REGION Network 1: Cân độc lập AGG5 Full
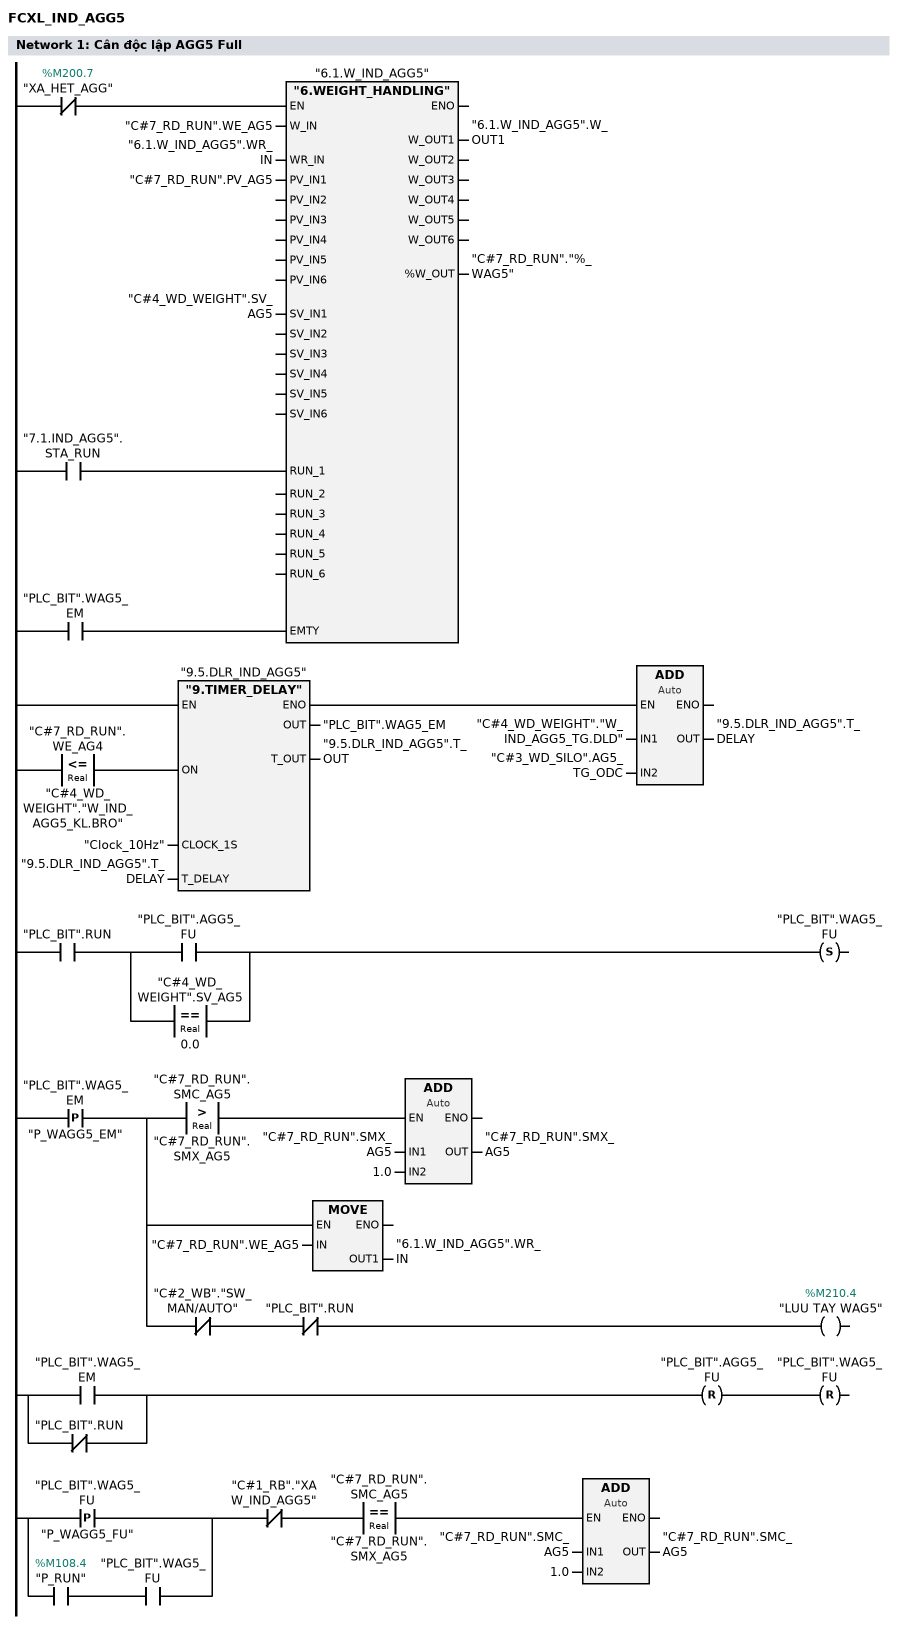
   RUNG wire#powerrail
      I_Contact( "XA_HET_AGG" )
      "6.1.W_IND_AGG5"(RUN_1 := wire#w1, EMTY := wire#w2, W_IN := "C#7_RD_RUN".WE_AG5, WR_IN := "6.1.W_IND_AGG5".WR_IN, PV_IN1 := "C#7_RD_RUN".PV_AG5, PV_IN2 :=, PV_IN3 :=, PV_IN4 :=, PV_IN5 :=, PV_IN6 :=, SV_IN1 := "C#4_WD_WEIGHT".SV_AG5, SV_IN2 :=, SV_IN3 :=, SV_IN4 :=, SV_IN5 :=, SV_IN6 :=, RUN_2 :=, RUN_3 :=, RUN_4 :=, RUN_5 :=, RUN_6 :=, W_OUT1 => "6.1.W_IND_AGG5".W_OUT1, W_OUT2 =>, W_OUT3 =>, W_OUT4 =>, W_OUT5 =>, W_OUT6 =>, "%W_OUT" => "C#7_RD_RUN"."%_WAG5")
   END_RUNG
   RUNG wire#powerrail
      Contact( "7.1.IND_AGG5".STA_RUN )
   END_RUNG wire#w1
   RUNG wire#powerrail
      Contact( "PLC_BIT".WAG5_EM )
   END_RUNG wire#w2
   RUNG wire#powerrail
      "9.5.DLR_IND_AGG5"(ON := wire#w3, CLOCK_1S := "Clock_10Hz", T_DELAY := "9.5.DLR_IND_AGG5".T_DELAY, OUT => "PLC_BIT".WAG5_EM, T_OUT => "9.5.DLR_IND_AGG5".T_OUT)
      Add(in1 := "C#4_WD_WEIGHT"."W_IND_AGG5_TG.DLD", in2 := "C#3_WD_SILO".AG5_TG_ODC, out => "9.5.DLR_IND_AGG5".T_DELAY)
   END_RUNG
   RUNG wire#powerrail
      { S7_Templates := "SrcType := Real" } LE_Contact(in1 := "C#7_RD_RUN".WE_AG4, in2 := "C#4_WD_WEIGHT"."W_IND_AGG5_KL.BRO")
   END_RUNG wire#w3
   RUNG wire#powerrail
      Contact( "PLC_BIT".RUN )
      wire#w4
      Contact( "PLC_BIT".AGG5_FU )
      wire#w5
      S_Coil( "PLC_BIT".WAG5_FU )
   END_RUNG
   RUNG wire#w4
      { S7_Templates := "SrcType := Real" } EQ_Contact(in1 := "C#4_WD_WEIGHT".SV_AG5, in2 := 0.0)
   END_RUNG wire#w5
   RUNG wire#powerrail
      P_Contact(operand := "PLC_BIT".WAG5_EM, bit := "P_WAGG5_EM")
      wire#w6
      { S7_Templates := "SrcType := Real" } GT_Contact(in1 := "C#7_RD_RUN".SMC_AG5, in2 := "C#7_RD_RUN".SMX_AG5)
      Add(in1 := "C#7_RD_RUN".SMX_AG5, in2 := 1.0, out => "C#7_RD_RUN".SMX_AG5)
   END_RUNG
   RUNG wire#w6
      Move(in := "C#7_RD_RUN".WE_AG5, out1 => "6.1.W_IND_AGG5".WR_IN)
   END_RUNG
   RUNG wire#w6
      I_Contact( "C#2_WB"."SW_MAN/AUTO" )
      I_Contact( "PLC_BIT".RUN )
      Coil( "LUU TAY WAG5" )
   END_RUNG
   RUNG wire#powerrail
      Contact( "PLC_BIT".WAG5_EM )
      wire#w7
      R_Coil( "PLC_BIT".AGG5_FU )
      R_Coil( "PLC_BIT".WAG5_FU )
   END_RUNG
   RUNG wire#powerrail
      I_Contact( "PLC_BIT".RUN )
   END_RUNG wire#w7
   RUNG wire#powerrail
      P_Contact(operand := "PLC_BIT".WAG5_FU, bit := "P_WAGG5_FU")
      wire#w8
      I_Contact( "C#1_RB"."XA W_IND_AGG5" )
      { S7_Templates := "SrcType := Real" } EQ_Contact(in1 := "C#7_RD_RUN".SMC_AG5, in2 := "C#7_RD_RUN".SMX_AG5)
      Add(in1 := "C#7_RD_RUN".SMC_AG5, in2 := 1.0, out => "C#7_RD_RUN".SMC_AG5)
   END_RUNG
   RUNG wire#powerrail
      Contact( "P_RUN" )
      Contact( "PLC_BIT".WAG5_FU )
   END_RUNG wire#w8
   // the same network as SCL:
   IF NOT "XA_HET_AGG" THEN
       "6.1.W_IND_AGG5"(W_IN := "C#7_RD_RUN".WE_AG5,   // "6.WEIGHT_HANDLING"
                        WR_IN := "6.1.W_IND_AGG5".WR_IN,
                        PV_IN1 := "C#7_RD_RUN".PV_AG5,
                        SV_IN1 := "C#4_WD_WEIGHT".SV_AG5,
                        RUN_1 := "7.1.IND_AGG5".STA_RUN,
                        EMTY := "PLC_BIT".WAG5_EM,
                        W_OUT1 => "6.1.W_IND_AGG5".W_OUT1,
                        "%W_OUT" => "C#7_RD_RUN"."%_WAG5");
   END_IF;
   "9.5.DLR_IND_AGG5"(ON := "C#7_RD_RUN".WE_AG4 <= "C#4_WD_WEIGHT"."W_IND_AGG5_KL.BRO",   // "9.TIMER_DELAY"
                      CLOCK_1S := "Clock_10Hz",
                      T_DELAY := "9.5.DLR_IND_AGG5".T_DELAY,
                      OUT => "PLC_BIT".WAG5_EM,
                      T_OUT => "9.5.DLR_IND_AGG5".T_OUT,
                      ENO => #_w1);
   IF #_w1 THEN
       "9.5.DLR_IND_AGG5".T_DELAY := "C#4_WD_WEIGHT"."W_IND_AGG5_TG.DLD" + "C#3_WD_SILO".AG5_TG_ODC;
   END_IF;
   IF "PLC_BIT".RUN AND ("PLC_BIT".AGG5_FU OR ("C#4_WD_WEIGHT".SV_AG5 = 0.0)) THEN
       "PLC_BIT".WAG5_FU := TRUE;
   END_IF;
   #_w2 := "PLC_BIT".WAG5_EM AND NOT "P_WAGG5_EM";   // rising edge of "PLC_BIT".WAG5_EM
   "P_WAGG5_EM" := "PLC_BIT".WAG5_EM;
   IF #_w2 AND ("C#7_RD_RUN".SMC_AG5 > "C#7_RD_RUN".SMX_AG5) THEN
       "C#7_RD_RUN".SMX_AG5 := "C#7_RD_RUN".SMX_AG5 + 1.0;
   END_IF;
   IF #_w2 THEN "6.1.W_IND_AGG5".WR_IN := "C#7_RD_RUN".WE_AG5; END_IF;
   "LUU TAY WAG5" := #_w2 AND NOT "C#2_WB"."SW_MAN/AUTO" AND NOT "PLC_BIT".RUN;
   IF "PLC_BIT".WAG5_EM OR NOT "PLC_BIT".RUN THEN
       "PLC_BIT".AGG5_FU := FALSE;
       "PLC_BIT".WAG5_FU := FALSE;
   END_IF;
   #_w3 := "PLC_BIT".WAG5_FU AND NOT "P_WAGG5_FU";   // rising edge of "PLC_BIT".WAG5_FU
   "P_WAGG5_FU" := "PLC_BIT".WAG5_FU;
   IF (#_w3 OR ("P_RUN" AND "PLC_BIT".WAG5_FU)) AND NOT "C#1_RB"."XA W_IND_AGG5" AND ("C#7_RD_RUN".SMC_AG5 = "C#7_RD_RUN".SMX_AG5) THEN
       "C#7_RD_RUN".SMC_AG5 := "C#7_RD_RUN".SMC_AG5 + 1.0;
   END_IF;
END_REGION
END_FUNCTION

FUNCTION "FCCA_IND_AGG5" : Void   // FC14, LAD
{ S7_Optimized_Access := 'TRUE' }
VERSION : 0.1
// stored: AutoNumber true, CodeModifiedDate 2026-01-15T16:25:54.5394757Z, CompileDate 2026-01-15T16:25:54.5786206Z, CreationDate 2026-01-15T16:24:02.4619467Z, HandleErrorsWithinBlock false, InterfaceModifiedDate 2026-01-11T04:47:10.3302964Z, IsConsistent true, IsIECCheckEnabled false, IsKnowHowProtected false, IsWriteProtected false, LibraryConformanceStatus Error: The block contains calls of single instances. Warning: The object contains access to global data blocks. Warning: The block contains direct access to inputs, outputs, bit memories, indirect access to the registry or indirect access to external memory areas that are unknown at the time of compilation., ModifiedDate 2026-01-15T16:25:54.5394757Z, ParameterModified 2026-01-11T04:47:10.3302964Z, PLCSimAdvancedSupport false, SetENOAutomatically False, StructureModified 2026-01-11T04:47:10.3302964Z, UDAEnableTagReadback false
BEGIN

REGION Network 1: Trạng thái cân AGG5
   // Đầu tiên nó sẽ đợi một khoảng thời gian gọi là Thời gian trễ cân, sau đó nó mới đủ điều kiện để cân
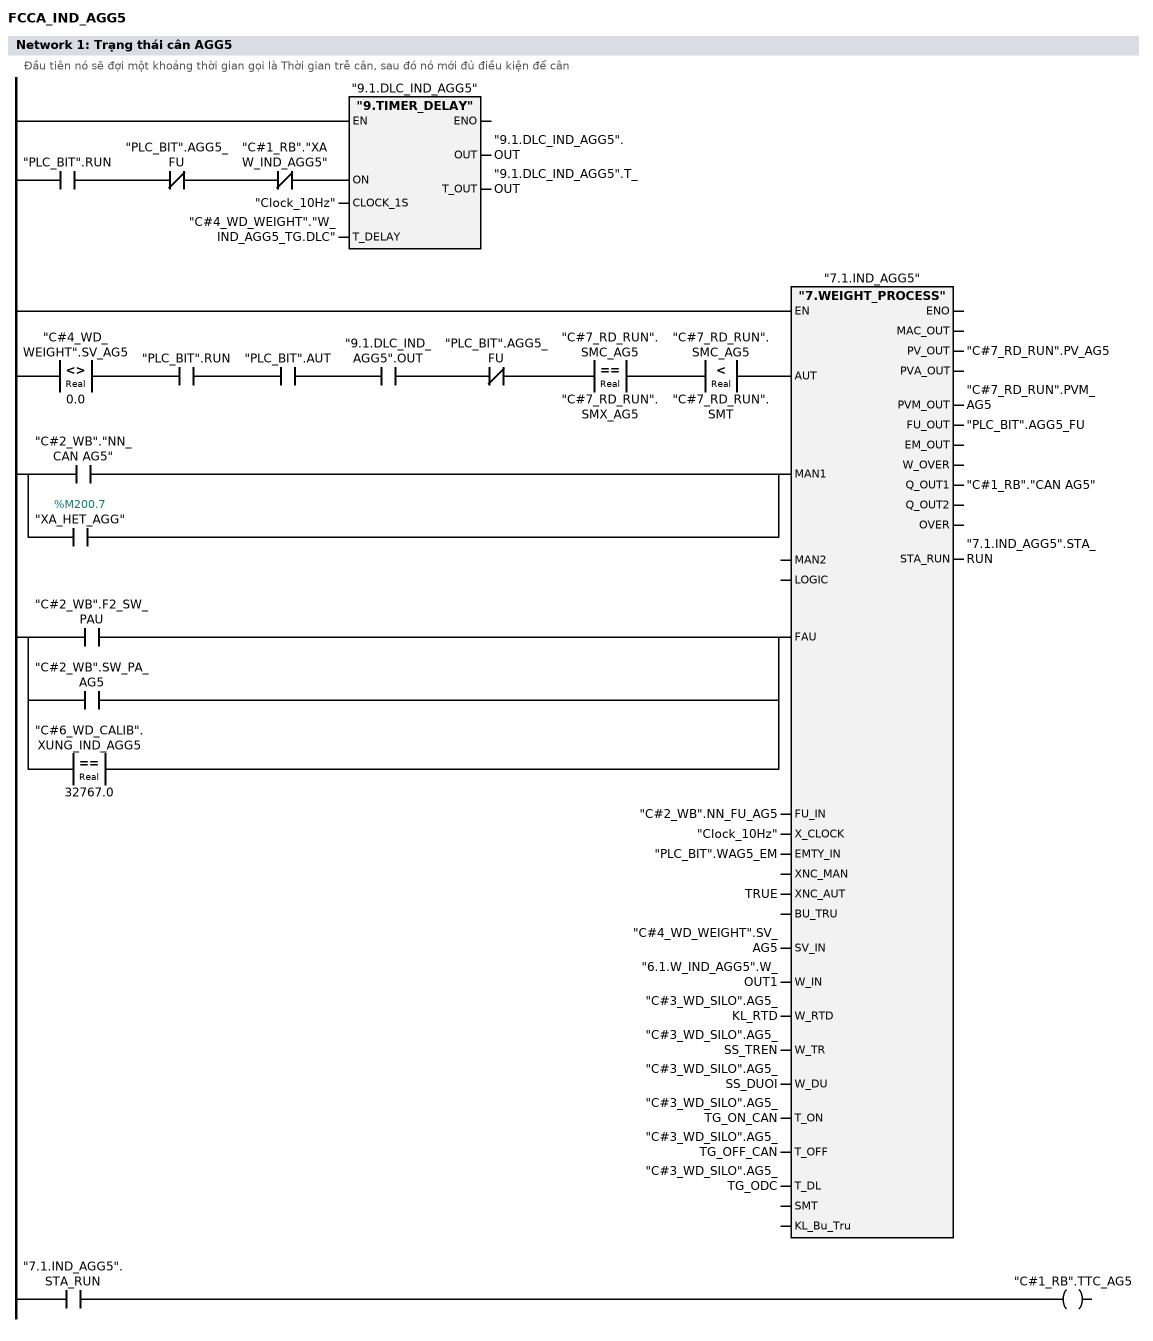
   RUNG wire#powerrail
      "9.1.DLC_IND_AGG5"(ON := wire#w1, CLOCK_1S := "Clock_10Hz", T_DELAY := "C#4_WD_WEIGHT"."W_IND_AGG5_TG.DLC", OUT => "9.1.DLC_IND_AGG5".OUT, T_OUT => "9.1.DLC_IND_AGG5".T_OUT)
   END_RUNG
   RUNG wire#powerrail
      Contact( "PLC_BIT".RUN )
      I_Contact( "PLC_BIT".AGG5_FU )
      I_Contact( "C#1_RB"."XA W_IND_AGG5" )
   END_RUNG wire#w1
   RUNG wire#powerrail
      "7.1.IND_AGG5"(AUT := wire#w2, MAN1 := wire#w3, FAU := wire#w4, MAN2 :=, LOGIC :=, FU_IN := "C#2_WB".NN_FU_AG5, X_CLOCK := "Clock_10Hz", EMTY_IN := "PLC_BIT".WAG5_EM, XNC_MAN :=, XNC_AUT := TRUE, BU_TRU :=, SV_IN := "C#4_WD_WEIGHT".SV_AG5, W_IN := "6.1.W_IND_AGG5".W_OUT1, W_RTD := "C#3_WD_SILO".AG5_KL_RTD, W_TR := "C#3_WD_SILO".AG5_SS_TREN, W_DU := "C#3_WD_SILO".AG5_SS_DUOI, T_ON := "C#3_WD_SILO".AG5_TG_ON_CAN, T_OFF := "C#3_WD_SILO".AG5_TG_OFF_CAN, T_DL := "C#3_WD_SILO".AG5_TG_ODC, SMT :=, KL_Bu_Tru :=, MAC_OUT =>, PV_OUT => "C#7_RD_RUN".PV_AG5, PVA_OUT =>, PVM_OUT => "C#7_RD_RUN".PVM_AG5, FU_OUT => "PLC_BIT".AGG5_FU, EM_OUT =>, W_OVER =>, Q_OUT1 => "C#1_RB"."CAN AG5", Q_OUT2 =>, OVER =>, STA_RUN => "7.1.IND_AGG5".STA_RUN)
   END_RUNG
   RUNG wire#powerrail
      { S7_Templates := "SrcType := Real" } NE_Contact(in1 := "C#4_WD_WEIGHT".SV_AG5, in2 := 0.0)
      Contact( "PLC_BIT".RUN )
      Contact( "PLC_BIT".AUT )
      Contact( "9.1.DLC_IND_AGG5".OUT )
      I_Contact( "PLC_BIT".AGG5_FU )
      { S7_Templates := "SrcType := Real" } EQ_Contact(in1 := "C#7_RD_RUN".SMC_AG5, in2 := "C#7_RD_RUN".SMX_AG5)
      { S7_Templates := "SrcType := Real" } LT_Contact(in1 := "C#7_RD_RUN".SMC_AG5, in2 := "C#7_RD_RUN".SMT)
   END_RUNG wire#w2
   RUNG wire#powerrail
      Contact( "C#2_WB"."NN_CAN AG5" )
   END_RUNG wire#w3
   RUNG wire#powerrail
      Contact( "XA_HET_AGG" )
   END_RUNG wire#w3
   RUNG wire#powerrail
      Contact( "C#2_WB".F2_SW_PAU )
   END_RUNG wire#w4
   RUNG wire#powerrail
      Contact( "C#2_WB".SW_PA_AG5 )
   END_RUNG wire#w4
   RUNG wire#powerrail
      { S7_Templates := "SrcType := Real" } EQ_Contact(in1 := "C#6_WD_CALIB".XUNG_IND_AGG5, in2 := 32767.0)
   END_RUNG wire#w4
   RUNG wire#powerrail
      Contact( "7.1.IND_AGG5".STA_RUN )
      Coil( "C#1_RB".TTC_AG5 )
   END_RUNG
   // the same network as SCL:
   "9.1.DLC_IND_AGG5"(ON := "PLC_BIT".RUN AND NOT "PLC_BIT".AGG5_FU AND NOT "C#1_RB"."XA W_IND_AGG5",   // "9.TIMER_DELAY"
                      CLOCK_1S := "Clock_10Hz",
                      T_DELAY := "C#4_WD_WEIGHT"."W_IND_AGG5_TG.DLC",
                      OUT => "9.1.DLC_IND_AGG5".OUT,
                      T_OUT => "9.1.DLC_IND_AGG5".T_OUT);
   "7.1.IND_AGG5"(AUT := ("C#4_WD_WEIGHT".SV_AG5 <> 0.0) AND "PLC_BIT".RUN AND "PLC_BIT".AUT AND "9.1.DLC_IND_AGG5".OUT AND NOT "PLC_BIT".AGG5_FU AND ("C#7_RD_RUN".SMC_AG5 = "C#7_RD_RUN".SMX_AG5) AND ("C#7_RD_RUN".SMC_AG5 < "C#7_RD_RUN".SMT),   // "7.WEIGHT_PROCESS"
                  MAN1 := "C#2_WB"."NN_CAN AG5" OR "XA_HET_AGG",
                  FAU := "C#2_WB".F2_SW_PAU OR "C#2_WB".SW_PA_AG5 OR ("C#6_WD_CALIB".XUNG_IND_AGG5 = 32767.0),
                  FU_IN := "C#2_WB".NN_FU_AG5,
                  X_CLOCK := "Clock_10Hz",
                  EMTY_IN := "PLC_BIT".WAG5_EM,
                  XNC_AUT := TRUE,
                  SV_IN := "C#4_WD_WEIGHT".SV_AG5,
                  W_IN := "6.1.W_IND_AGG5".W_OUT1,
                  W_RTD := "C#3_WD_SILO".AG5_KL_RTD,
                  W_TR := "C#3_WD_SILO".AG5_SS_TREN,
                  W_DU := "C#3_WD_SILO".AG5_SS_DUOI,
                  T_ON := "C#3_WD_SILO".AG5_TG_ON_CAN,
                  T_OFF := "C#3_WD_SILO".AG5_TG_OFF_CAN,
                  T_DL := "C#3_WD_SILO".AG5_TG_ODC,
                  PV_OUT => "C#7_RD_RUN".PV_AG5,
                  PVM_OUT => "C#7_RD_RUN".PVM_AG5,
                  FU_OUT => "PLC_BIT".AGG5_FU,
                  Q_OUT1 => "C#1_RB"."CAN AG5",
                  STA_RUN => "7.1.IND_AGG5".STA_RUN);
   "C#1_RB".TTC_AG5 := "7.1.IND_AGG5".STA_RUN;
END_REGION
END_FUNCTION

FUNCTION "FCXL_CCD_FD1" : Void   // FC10, LAD
{ S7_Optimized_Access := 'TRUE' }
VERSION : 0.1
// stored: AutoNumber true, CodeModifiedDate 2026-01-15T16:25:54.9008625Z, CompileDate 2026-01-15T16:25:54.9411388Z, CreationDate 2026-01-15T16:24:02.4619467Z, HandleErrorsWithinBlock false, InterfaceModifiedDate 2024-08-08T03:13:40.4539851Z, IsConsistent true, IsIECCheckEnabled false, IsKnowHowProtected false, IsWriteProtected false, LibraryConformanceStatus Error: The block contains calls of single instances. Warning: The object contains access to global data blocks. Warning: The block contains direct access to inputs, outputs, bit memories, indirect access to the registry or indirect access to external memory areas that are unknown at the time of compilation., ModifiedDate 2026-01-15T16:25:54.9008625Z, ParameterModified 2024-08-08T03:13:40.4539851Z, PLCSimAdvancedSupport false, SetENOAutomatically False, StructureModified 2024-08-08T03:13:40.4539851Z, UDAEnableTagReadback false
   VAR_TEMP   // added for the SCL form of the ladder/FBD networks
      _w1 : Bool;
      _w2 : Bool;
      _w3 : Bool;
   END_VAR
BEGIN

REGION Network 1: Cân CE/FD1 Full
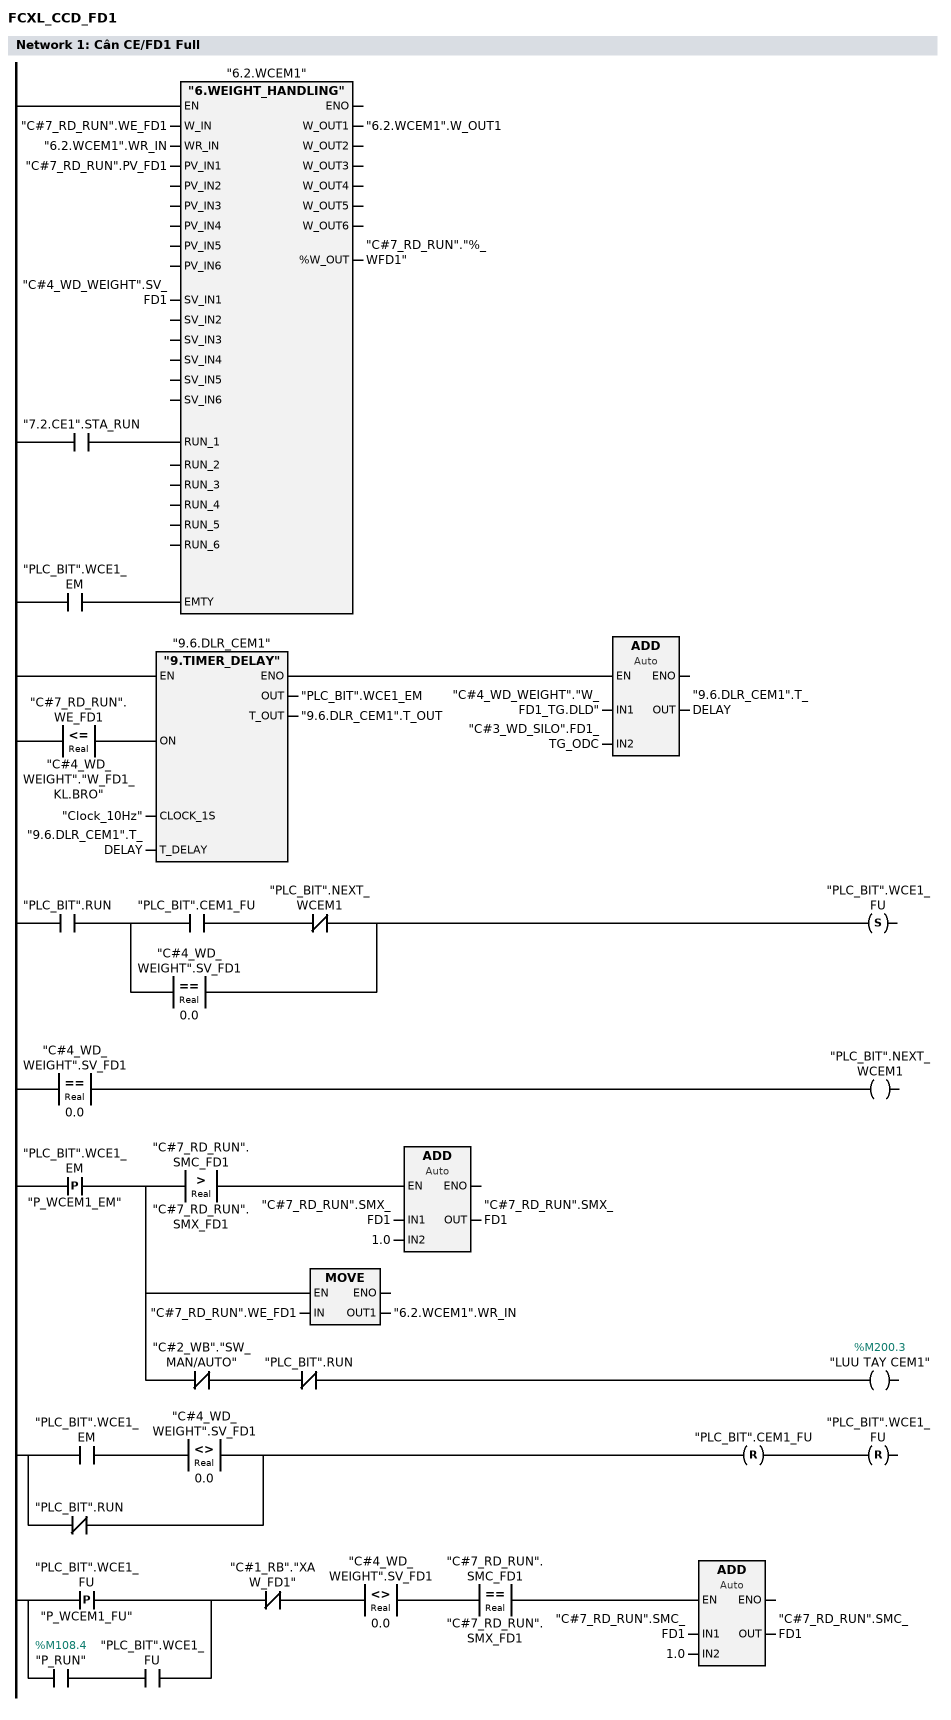
   RUNG wire#powerrail
      "6.2.WCEM1"(RUN_1 := wire#w1, EMTY := wire#w2, W_IN := "C#7_RD_RUN".WE_FD1, WR_IN := "6.2.WCEM1".WR_IN, PV_IN1 := "C#7_RD_RUN".PV_FD1, PV_IN2 :=, PV_IN3 :=, PV_IN4 :=, PV_IN5 :=, PV_IN6 :=, SV_IN1 := "C#4_WD_WEIGHT".SV_FD1, SV_IN2 :=, SV_IN3 :=, SV_IN4 :=, SV_IN5 :=, SV_IN6 :=, RUN_2 :=, RUN_3 :=, RUN_4 :=, RUN_5 :=, RUN_6 :=, W_OUT1 => "6.2.WCEM1".W_OUT1, W_OUT2 =>, W_OUT3 =>, W_OUT4 =>, W_OUT5 =>, W_OUT6 =>, "%W_OUT" => "C#7_RD_RUN"."%_WFD1")
   END_RUNG
   RUNG wire#powerrail
      Contact( "7.2.CE1".STA_RUN )
   END_RUNG wire#w1
   RUNG wire#powerrail
      Contact( "PLC_BIT".WCE1_EM )
   END_RUNG wire#w2
   RUNG wire#powerrail
      "9.6.DLR_CEM1"(ON := wire#w3, CLOCK_1S := "Clock_10Hz", T_DELAY := "9.6.DLR_CEM1".T_DELAY, OUT => "PLC_BIT".WCE1_EM, T_OUT => "9.6.DLR_CEM1".T_OUT)
      Add(in1 := "C#4_WD_WEIGHT"."W_FD1_TG.DLD", in2 := "C#3_WD_SILO".FD1_TG_ODC, out => "9.6.DLR_CEM1".T_DELAY)
   END_RUNG
   RUNG wire#powerrail
      { S7_Templates := "SrcType := Real" } LE_Contact(in1 := "C#7_RD_RUN".WE_FD1, in2 := "C#4_WD_WEIGHT"."W_FD1_KL.BRO")
   END_RUNG wire#w3
   RUNG wire#powerrail
      Contact( "PLC_BIT".RUN )
      wire#w4
      Contact( "PLC_BIT".CEM1_FU )
      I_Contact( "PLC_BIT".NEXT_WCEM1 )
      wire#w5
      S_Coil( "PLC_BIT".WCE1_FU )
   END_RUNG
   RUNG wire#w4
      { S7_Templates := "SrcType := Real" } EQ_Contact(in1 := "C#4_WD_WEIGHT".SV_FD1, in2 := 0.0)
   END_RUNG wire#w5
   RUNG wire#powerrail
      { S7_Templates := "SrcType := Real" } EQ_Contact(in1 := "C#4_WD_WEIGHT".SV_FD1, in2 := 0.0)
      Coil( "PLC_BIT".NEXT_WCEM1 )
   END_RUNG
   RUNG wire#powerrail
      P_Contact(operand := "PLC_BIT".WCE1_EM, bit := "P_WCEM1_EM")
      wire#w6
      { S7_Templates := "SrcType := Real" } GT_Contact(in1 := "C#7_RD_RUN".SMC_FD1, in2 := "C#7_RD_RUN".SMX_FD1)
      Add(in1 := "C#7_RD_RUN".SMX_FD1, in2 := 1.0, out => "C#7_RD_RUN".SMX_FD1)
   END_RUNG
   RUNG wire#w6
      Move(in := "C#7_RD_RUN".WE_FD1, out1 => "6.2.WCEM1".WR_IN)
   END_RUNG
   RUNG wire#w6
      I_Contact( "C#2_WB"."SW_MAN/AUTO" )
      I_Contact( "PLC_BIT".RUN )
      Coil( "LUU TAY CEM1" )
   END_RUNG
   RUNG wire#powerrail
      Contact( "PLC_BIT".WCE1_EM )
      { S7_Templates := "SrcType := Real" } NE_Contact(in1 := "C#4_WD_WEIGHT".SV_FD1, in2 := 0.0)
      wire#w7
      R_Coil( "PLC_BIT".CEM1_FU )
      R_Coil( "PLC_BIT".WCE1_FU )
   END_RUNG
   RUNG wire#powerrail
      I_Contact( "PLC_BIT".RUN )
   END_RUNG wire#w7
   RUNG wire#powerrail
      P_Contact(operand := "PLC_BIT".WCE1_FU, bit := "P_WCEM1_FU")
      wire#w8
      I_Contact( "C#1_RB"."XA W_FD1" )
      { S7_Templates := "SrcType := Real" } NE_Contact(in1 := "C#4_WD_WEIGHT".SV_FD1, in2 := 0.0)
      { S7_Templates := "SrcType := Real" } EQ_Contact(in1 := "C#7_RD_RUN".SMC_FD1, in2 := "C#7_RD_RUN".SMX_FD1)
      Add(in1 := "C#7_RD_RUN".SMC_FD1, in2 := 1.0, out => "C#7_RD_RUN".SMC_FD1)
   END_RUNG
   RUNG wire#powerrail
      Contact( "P_RUN" )
      Contact( "PLC_BIT".WCE1_FU )
   END_RUNG wire#w8
   // the same network as SCL:
   "6.2.WCEM1"(W_IN := "C#7_RD_RUN".WE_FD1,   // "6.WEIGHT_HANDLING"
               WR_IN := "6.2.WCEM1".WR_IN,
               PV_IN1 := "C#7_RD_RUN".PV_FD1,
               SV_IN1 := "C#4_WD_WEIGHT".SV_FD1,
               RUN_1 := "7.2.CE1".STA_RUN,
               EMTY := "PLC_BIT".WCE1_EM,
               W_OUT1 => "6.2.WCEM1".W_OUT1,
               "%W_OUT" => "C#7_RD_RUN"."%_WFD1");
   "9.6.DLR_CEM1"(ON := "C#7_RD_RUN".WE_FD1 <= "C#4_WD_WEIGHT"."W_FD1_KL.BRO",   // "9.TIMER_DELAY"
                  CLOCK_1S := "Clock_10Hz",
                  T_DELAY := "9.6.DLR_CEM1".T_DELAY,
                  OUT => "PLC_BIT".WCE1_EM,
                  T_OUT => "9.6.DLR_CEM1".T_OUT,
                  ENO => #_w1);
   IF #_w1 THEN "9.6.DLR_CEM1".T_DELAY := "C#4_WD_WEIGHT"."W_FD1_TG.DLD" + "C#3_WD_SILO".FD1_TG_ODC; END_IF;
   IF "PLC_BIT".RUN AND (("PLC_BIT".CEM1_FU AND NOT "PLC_BIT".NEXT_WCEM1) OR ("C#4_WD_WEIGHT".SV_FD1 = 0.0)) THEN
       "PLC_BIT".WCE1_FU := TRUE;
   END_IF;
   "PLC_BIT".NEXT_WCEM1 := "C#4_WD_WEIGHT".SV_FD1 = 0.0;
   #_w2 := "PLC_BIT".WCE1_EM AND NOT "P_WCEM1_EM";   // rising edge of "PLC_BIT".WCE1_EM
   "P_WCEM1_EM" := "PLC_BIT".WCE1_EM;
   IF #_w2 AND ("C#7_RD_RUN".SMC_FD1 > "C#7_RD_RUN".SMX_FD1) THEN
       "C#7_RD_RUN".SMX_FD1 := "C#7_RD_RUN".SMX_FD1 + 1.0;
   END_IF;
   IF #_w2 THEN "6.2.WCEM1".WR_IN := "C#7_RD_RUN".WE_FD1; END_IF;
   "LUU TAY CEM1" := #_w2 AND NOT "C#2_WB"."SW_MAN/AUTO" AND NOT "PLC_BIT".RUN;
   IF ("PLC_BIT".WCE1_EM AND ("C#4_WD_WEIGHT".SV_FD1 <> 0.0)) OR NOT "PLC_BIT".RUN THEN
       "PLC_BIT".CEM1_FU := FALSE;
       "PLC_BIT".WCE1_FU := FALSE;
   END_IF;
   #_w3 := "PLC_BIT".WCE1_FU AND NOT "P_WCEM1_FU";   // rising edge of "PLC_BIT".WCE1_FU
   "P_WCEM1_FU" := "PLC_BIT".WCE1_FU;
   IF (#_w3 OR ("P_RUN" AND "PLC_BIT".WCE1_FU)) AND NOT "C#1_RB"."XA W_FD1" AND ("C#4_WD_WEIGHT".SV_FD1 <> 0.0) AND ("C#7_RD_RUN".SMC_FD1 = "C#7_RD_RUN".SMX_FD1) THEN
       "C#7_RD_RUN".SMC_FD1 := "C#7_RD_RUN".SMC_FD1 + 1.0;
   END_IF;
END_REGION
END_FUNCTION

FUNCTION "FCCA_CCD_FD1" : Void   // FC12, LAD
{ S7_Optimized_Access := 'TRUE' }
VERSION : 0.1
// stored: AutoNumber true, CodeModifiedDate 2026-01-15T16:25:54.7244744Z, CompileDate 2026-01-15T16:25:54.7683501Z, CreationDate 2026-01-15T16:24:02.4619467Z, HandleErrorsWithinBlock false, InterfaceModifiedDate 2024-08-08T03:19:31.8063857Z, IsConsistent true, IsIECCheckEnabled false, IsKnowHowProtected false, IsWriteProtected false, LibraryConformanceStatus Error: The block contains calls of single instances. Warning: The object contains access to global data blocks. Warning: The block contains direct access to inputs, outputs, bit memories, indirect access to the registry or indirect access to external memory areas that are unknown at the time of compilation., ModifiedDate 2026-01-15T16:25:54.7244744Z, ParameterModified 2024-08-08T03:19:31.8063857Z, PLCSimAdvancedSupport false, SetENOAutomatically False, StructureModified 2024-08-08T03:19:31.8063857Z, UDAEnableTagReadback false
   VAR_TEMP   // added for the SCL form of the ladder/FBD networks
      _w1 : Bool;
   END_VAR
BEGIN

REGION Network 1: CAN XI MANG 1
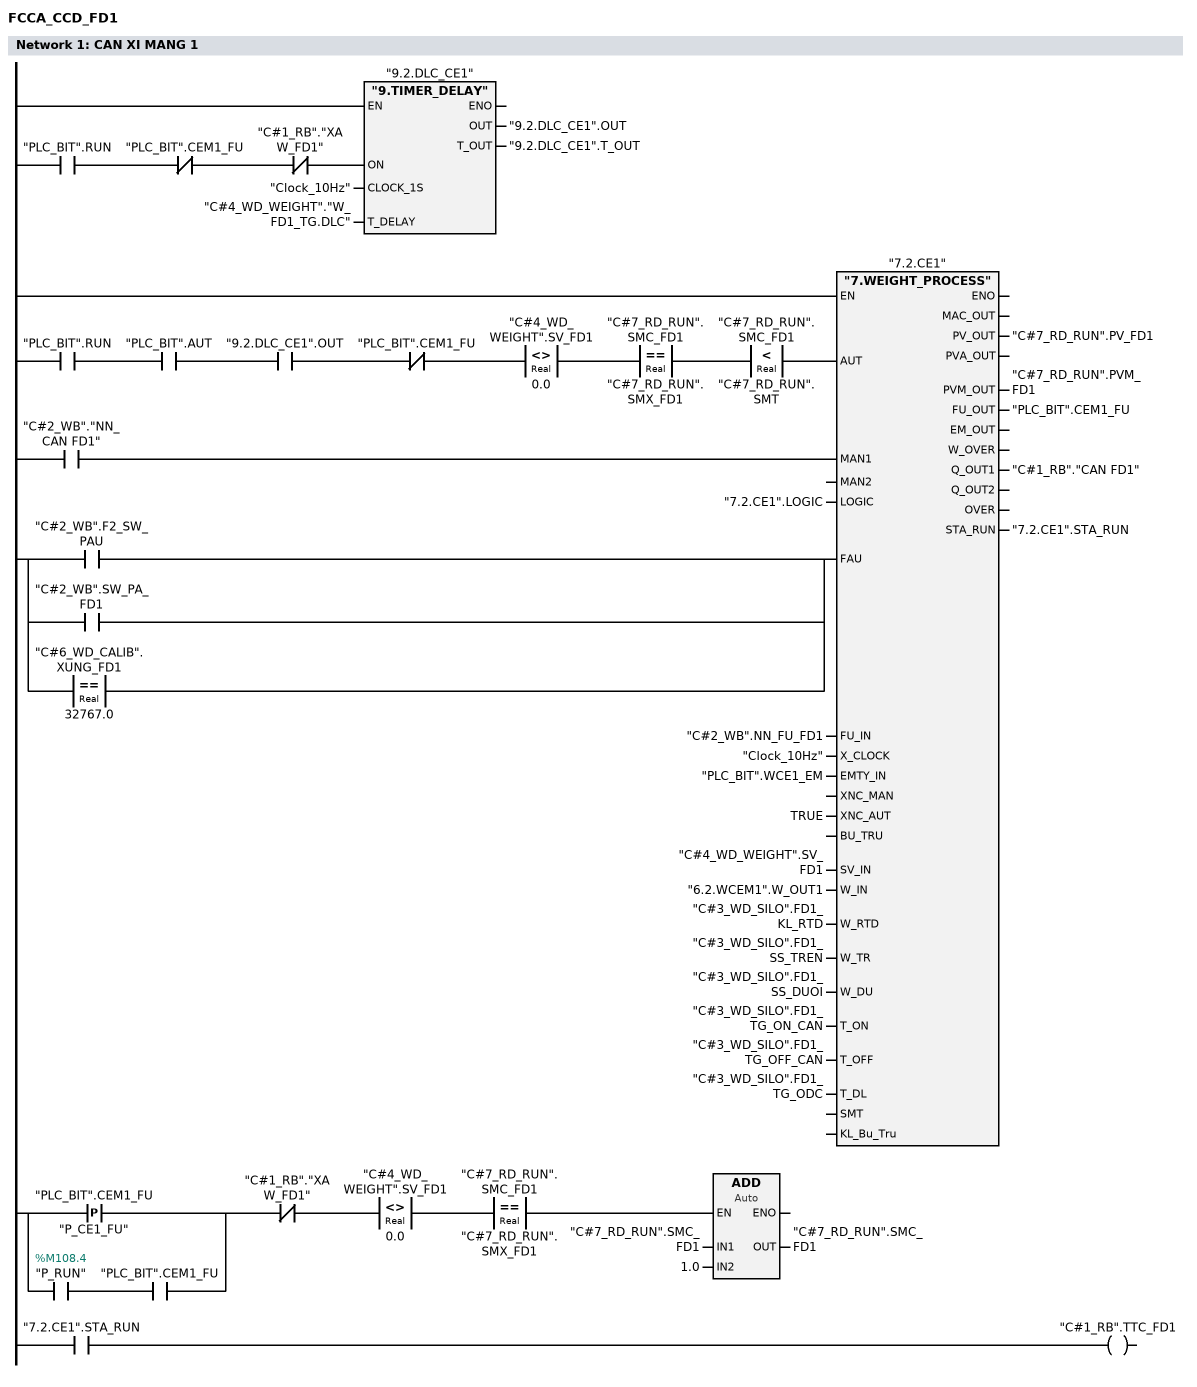
   RUNG wire#powerrail
      "9.2.DLC_CE1"(ON := wire#w1, CLOCK_1S := "Clock_10Hz", T_DELAY := "C#4_WD_WEIGHT"."W_FD1_TG.DLC", OUT => "9.2.DLC_CE1".OUT, T_OUT => "9.2.DLC_CE1".T_OUT)
   END_RUNG
   RUNG wire#powerrail
      Contact( "PLC_BIT".RUN )
      I_Contact( "PLC_BIT".CEM1_FU )
      I_Contact( "C#1_RB"."XA W_FD1" )
   END_RUNG wire#w1
   RUNG wire#powerrail
      "7.2.CE1"(AUT := wire#w2, MAN1 := wire#w3, FAU := wire#w4, MAN2 :=, LOGIC := "7.2.CE1".LOGIC, FU_IN := "C#2_WB".NN_FU_FD1, X_CLOCK := "Clock_10Hz", EMTY_IN := "PLC_BIT".WCE1_EM, XNC_MAN :=, XNC_AUT := TRUE, BU_TRU :=, SV_IN := "C#4_WD_WEIGHT".SV_FD1, W_IN := "6.2.WCEM1".W_OUT1, W_RTD := "C#3_WD_SILO".FD1_KL_RTD, W_TR := "C#3_WD_SILO".FD1_SS_TREN, W_DU := "C#3_WD_SILO".FD1_SS_DUOI, T_ON := "C#3_WD_SILO".FD1_TG_ON_CAN, T_OFF := "C#3_WD_SILO".FD1_TG_OFF_CAN, T_DL := "C#3_WD_SILO".FD1_TG_ODC, SMT :=, KL_Bu_Tru :=, MAC_OUT =>, PV_OUT => "C#7_RD_RUN".PV_FD1, PVA_OUT =>, PVM_OUT => "C#7_RD_RUN".PVM_FD1, FU_OUT => "PLC_BIT".CEM1_FU, EM_OUT =>, W_OVER =>, Q_OUT1 => "C#1_RB"."CAN FD1", Q_OUT2 =>, OVER =>, STA_RUN => "7.2.CE1".STA_RUN)
   END_RUNG
   RUNG wire#powerrail
      Contact( "PLC_BIT".RUN )
      Contact( "PLC_BIT".AUT )
      Contact( "9.2.DLC_CE1".OUT )
      I_Contact( "PLC_BIT".CEM1_FU )
      { S7_Templates := "SrcType := Real" } NE_Contact(in1 := "C#4_WD_WEIGHT".SV_FD1, in2 := 0.0)
      { S7_Templates := "SrcType := Real" } EQ_Contact(in1 := "C#7_RD_RUN".SMC_FD1, in2 := "C#7_RD_RUN".SMX_FD1)
      { S7_Templates := "SrcType := Real" } LT_Contact(in1 := "C#7_RD_RUN".SMC_FD1, in2 := "C#7_RD_RUN".SMT)
   END_RUNG wire#w2
   RUNG wire#powerrail
      Contact( "C#2_WB"."NN_CAN FD1" )
   END_RUNG wire#w3
   RUNG wire#powerrail
      Contact( "C#2_WB".F2_SW_PAU )
   END_RUNG wire#w4
   RUNG wire#powerrail
      Contact( "C#2_WB".SW_PA_FD1 )
   END_RUNG wire#w4
   RUNG wire#powerrail
      { S7_Templates := "SrcType := Real" } EQ_Contact(in1 := "C#6_WD_CALIB".XUNG_FD1, in2 := 32767.0)
   END_RUNG wire#w4
   RUNG wire#powerrail
      P_Contact(operand := "PLC_BIT".CEM1_FU, bit := "P_CE1_FU")
      wire#w5
      I_Contact( "C#1_RB"."XA W_FD1" )
      { S7_Templates := "SrcType := Real" } NE_Contact(in1 := "C#4_WD_WEIGHT".SV_FD1, in2 := 0.0)
      { S7_Templates := "SrcType := Real" } EQ_Contact(in1 := "C#7_RD_RUN".SMC_FD1, in2 := "C#7_RD_RUN".SMX_FD1)
      Add(in1 := "C#7_RD_RUN".SMC_FD1, in2 := 1.0, out => "C#7_RD_RUN".SMC_FD1)
   END_RUNG
   RUNG wire#powerrail
      Contact( "P_RUN" )
      Contact( "PLC_BIT".CEM1_FU )
   END_RUNG wire#w5
   RUNG wire#powerrail
      Contact( "7.2.CE1".STA_RUN )
      Coil( "C#1_RB".TTC_FD1 )
   END_RUNG
   // the same network as SCL:
   "9.2.DLC_CE1"(ON := "PLC_BIT".RUN AND NOT "PLC_BIT".CEM1_FU AND NOT "C#1_RB"."XA W_FD1",   // "9.TIMER_DELAY"
                 CLOCK_1S := "Clock_10Hz",
                 T_DELAY := "C#4_WD_WEIGHT"."W_FD1_TG.DLC",
                 OUT => "9.2.DLC_CE1".OUT,
                 T_OUT => "9.2.DLC_CE1".T_OUT);
   "7.2.CE1"(AUT := "PLC_BIT".RUN AND "PLC_BIT".AUT AND "9.2.DLC_CE1".OUT AND NOT "PLC_BIT".CEM1_FU AND ("C#4_WD_WEIGHT".SV_FD1 <> 0.0) AND ("C#7_RD_RUN".SMC_FD1 = "C#7_RD_RUN".SMX_FD1) AND ("C#7_RD_RUN".SMC_FD1 < "C#7_RD_RUN".SMT),   // "7.WEIGHT_PROCESS"
             MAN1 := "C#2_WB"."NN_CAN FD1",
             LOGIC := "7.2.CE1".LOGIC,
             FAU := "C#2_WB".F2_SW_PAU OR "C#2_WB".SW_PA_FD1 OR ("C#6_WD_CALIB".XUNG_FD1 = 32767.0),
             FU_IN := "C#2_WB".NN_FU_FD1,
             X_CLOCK := "Clock_10Hz",
             EMTY_IN := "PLC_BIT".WCE1_EM,
             XNC_AUT := TRUE,
             SV_IN := "C#4_WD_WEIGHT".SV_FD1,
             W_IN := "6.2.WCEM1".W_OUT1,
             W_RTD := "C#3_WD_SILO".FD1_KL_RTD,
             W_TR := "C#3_WD_SILO".FD1_SS_TREN,
             W_DU := "C#3_WD_SILO".FD1_SS_DUOI,
             T_ON := "C#3_WD_SILO".FD1_TG_ON_CAN,
             T_OFF := "C#3_WD_SILO".FD1_TG_OFF_CAN,
             T_DL := "C#3_WD_SILO".FD1_TG_ODC,
             PV_OUT => "C#7_RD_RUN".PV_FD1,
             PVM_OUT => "C#7_RD_RUN".PVM_FD1,
             FU_OUT => "PLC_BIT".CEM1_FU,
             Q_OUT1 => "C#1_RB"."CAN FD1",
             STA_RUN => "7.2.CE1".STA_RUN);
   #_w1 := "PLC_BIT".CEM1_FU AND NOT "P_CE1_FU";   // rising edge of "PLC_BIT".CEM1_FU
   "P_CE1_FU" := "PLC_BIT".CEM1_FU;
   IF (#_w1 OR ("P_RUN" AND "PLC_BIT".CEM1_FU)) AND NOT "C#1_RB"."XA W_FD1" AND ("C#4_WD_WEIGHT".SV_FD1 <> 0.0) AND ("C#7_RD_RUN".SMC_FD1 = "C#7_RD_RUN".SMX_FD1) THEN
       "C#7_RD_RUN".SMC_FD1 := "C#7_RD_RUN".SMC_FD1 + 1.0;
   END_IF;
   "C#1_RB".TTC_FD1 := "7.2.CE1".STA_RUN;
END_REGION
END_FUNCTION

FUNCTION "FCXL_CCD_AP1" : Void   // FC15, LAD
{ S7_Optimized_Access := 'TRUE' }
VERSION : 0.1
// stored: AutoNumber true, CodeModifiedDate 2026-01-15T16:25:54.4516816Z, CompileDate 2026-01-15T16:25:54.494478Z, CreationDate 2026-01-15T16:24:02.4619467Z, HandleErrorsWithinBlock false, InterfaceModifiedDate 2024-08-08T03:23:40.7447783Z, IsConsistent true, IsIECCheckEnabled false, IsKnowHowProtected false, IsWriteProtected false, LibraryConformanceStatus Error: The block contains calls of single instances. Warning: The object contains access to global data blocks. Warning: The block contains direct access to inputs, outputs, bit memories, indirect access to the registry or indirect access to external memory areas that are unknown at the time of compilation., ModifiedDate 2026-01-15T16:25:54.4516816Z, ParameterModified 2024-08-08T03:23:40.7447783Z, PLCSimAdvancedSupport false, SetENOAutomatically False, StructureModified 2024-08-08T03:23:40.7447783Z, UDAEnableTagReadback false
   VAR_TEMP   // added for the SCL form of the ladder/FBD networks
      _w1 : Bool;
      _w2 : Bool;
      _w3 : Bool;
   END_VAR
BEGIN

REGION Network 1: Weigh Asphalt Tank 1 Full - Cảm biến báo bể nhựa 1 đầy
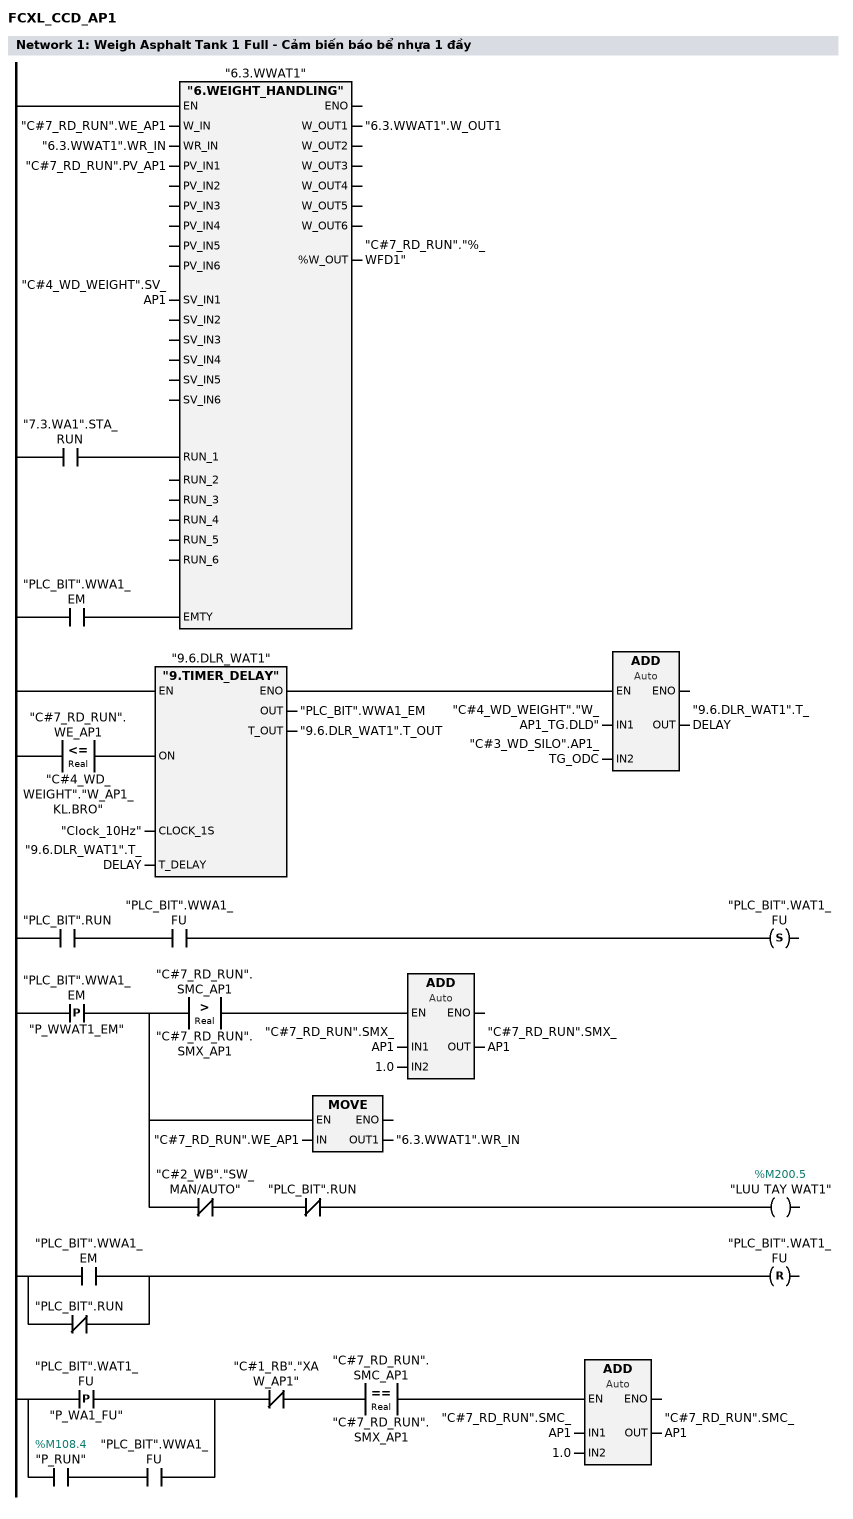
   RUNG wire#powerrail
      "6.3.WWAT1"(RUN_1 := wire#w1, EMTY := wire#w2, W_IN := "C#7_RD_RUN".WE_AP1, WR_IN := "6.3.WWAT1".WR_IN, PV_IN1 := "C#7_RD_RUN".PV_AP1, PV_IN2 :=, PV_IN3 :=, PV_IN4 :=, PV_IN5 :=, PV_IN6 :=, SV_IN1 := "C#4_WD_WEIGHT".SV_AP1, SV_IN2 :=, SV_IN3 :=, SV_IN4 :=, SV_IN5 :=, SV_IN6 :=, RUN_2 :=, RUN_3 :=, RUN_4 :=, RUN_5 :=, RUN_6 :=, W_OUT1 => "6.3.WWAT1".W_OUT1, W_OUT2 =>, W_OUT3 =>, W_OUT4 =>, W_OUT5 =>, W_OUT6 =>, "%W_OUT" => "C#7_RD_RUN"."%_WFD1")
   END_RUNG
   RUNG wire#powerrail
      Contact( "7.3.WA1".STA_RUN )
   END_RUNG wire#w1
   RUNG wire#powerrail
      Contact( "PLC_BIT".WWA1_EM )
   END_RUNG wire#w2
   RUNG wire#powerrail
      "9.6.DLR_WAT1"(ON := wire#w3, CLOCK_1S := "Clock_10Hz", T_DELAY := "9.6.DLR_WAT1".T_DELAY, OUT => "PLC_BIT".WWA1_EM, T_OUT => "9.6.DLR_WAT1".T_OUT)
      Add(in1 := "C#4_WD_WEIGHT"."W_AP1_TG.DLD", in2 := "C#3_WD_SILO".AP1_TG_ODC, out => "9.6.DLR_WAT1".T_DELAY)
   END_RUNG
   RUNG wire#powerrail
      { S7_Templates := "SrcType := Real" } LE_Contact(in1 := "C#7_RD_RUN".WE_AP1, in2 := "C#4_WD_WEIGHT"."W_AP1_KL.BRO")
   END_RUNG wire#w3
   RUNG wire#powerrail
      Contact( "PLC_BIT".RUN )
      Contact( "PLC_BIT".WWA1_FU )
      S_Coil( "PLC_BIT".WAT1_FU )
   END_RUNG
   RUNG wire#powerrail
      P_Contact(operand := "PLC_BIT".WWA1_EM, bit := "P_WWAT1_EM")
      wire#w4
      { S7_Templates := "SrcType := Real" } GT_Contact(in1 := "C#7_RD_RUN".SMC_AP1, in2 := "C#7_RD_RUN".SMX_AP1)
      Add(in1 := "C#7_RD_RUN".SMX_AP1, in2 := 1.0, out => "C#7_RD_RUN".SMX_AP1)
   END_RUNG
   RUNG wire#w4
      Move(in := "C#7_RD_RUN".WE_AP1, out1 => "6.3.WWAT1".WR_IN)
   END_RUNG
   RUNG wire#w4
      I_Contact( "C#2_WB"."SW_MAN/AUTO" )
      I_Contact( "PLC_BIT".RUN )
      Coil( "LUU TAY WAT1" )
   END_RUNG
   RUNG wire#powerrail
      Contact( "PLC_BIT".WWA1_EM )
      wire#w5
      R_Coil( "PLC_BIT".WAT1_FU )
   END_RUNG
   RUNG wire#powerrail
      I_Contact( "PLC_BIT".RUN )
   END_RUNG wire#w5
   RUNG wire#powerrail
      P_Contact(operand := "PLC_BIT".WAT1_FU, bit := "P_WA1_FU")
      wire#w6
      I_Contact( "C#1_RB"."XA W_AP1" )
      { S7_Templates := "SrcType := Real" } EQ_Contact(in1 := "C#7_RD_RUN".SMC_AP1, in2 := "C#7_RD_RUN".SMX_AP1)
      Add(in1 := "C#7_RD_RUN".SMC_AP1, in2 := 1.0, out => "C#7_RD_RUN".SMC_AP1)
   END_RUNG
   RUNG wire#powerrail
      Contact( "P_RUN" )
      Contact( "PLC_BIT".WWA1_FU )
   END_RUNG wire#w6
   // the same network as SCL:
   "6.3.WWAT1"(W_IN := "C#7_RD_RUN".WE_AP1,   // "6.WEIGHT_HANDLING"
               WR_IN := "6.3.WWAT1".WR_IN,
               PV_IN1 := "C#7_RD_RUN".PV_AP1,
               SV_IN1 := "C#4_WD_WEIGHT".SV_AP1,
               RUN_1 := "7.3.WA1".STA_RUN,
               EMTY := "PLC_BIT".WWA1_EM,
               W_OUT1 => "6.3.WWAT1".W_OUT1,
               "%W_OUT" => "C#7_RD_RUN"."%_WFD1");
   "9.6.DLR_WAT1"(ON := "C#7_RD_RUN".WE_AP1 <= "C#4_WD_WEIGHT"."W_AP1_KL.BRO",   // "9.TIMER_DELAY"
                  CLOCK_1S := "Clock_10Hz",
                  T_DELAY := "9.6.DLR_WAT1".T_DELAY,
                  OUT => "PLC_BIT".WWA1_EM,
                  T_OUT => "9.6.DLR_WAT1".T_OUT,
                  ENO => #_w1);
   IF #_w1 THEN "9.6.DLR_WAT1".T_DELAY := "C#4_WD_WEIGHT"."W_AP1_TG.DLD" + "C#3_WD_SILO".AP1_TG_ODC; END_IF;
   IF "PLC_BIT".RUN AND "PLC_BIT".WWA1_FU THEN "PLC_BIT".WAT1_FU := TRUE; END_IF;
   #_w2 := "PLC_BIT".WWA1_EM AND NOT "P_WWAT1_EM";   // rising edge of "PLC_BIT".WWA1_EM
   "P_WWAT1_EM" := "PLC_BIT".WWA1_EM;
   IF #_w2 AND ("C#7_RD_RUN".SMC_AP1 > "C#7_RD_RUN".SMX_AP1) THEN
       "C#7_RD_RUN".SMX_AP1 := "C#7_RD_RUN".SMX_AP1 + 1.0;
   END_IF;
   IF #_w2 THEN "6.3.WWAT1".WR_IN := "C#7_RD_RUN".WE_AP1; END_IF;
   "LUU TAY WAT1" := #_w2 AND NOT "C#2_WB"."SW_MAN/AUTO" AND NOT "PLC_BIT".RUN;
   IF "PLC_BIT".WWA1_EM OR NOT "PLC_BIT".RUN THEN "PLC_BIT".WAT1_FU := FALSE; END_IF;
   #_w3 := "PLC_BIT".WAT1_FU AND NOT "P_WA1_FU";   // rising edge of "PLC_BIT".WAT1_FU
   "P_WA1_FU" := "PLC_BIT".WAT1_FU;
   IF (#_w3 OR ("P_RUN" AND "PLC_BIT".WWA1_FU)) AND NOT "C#1_RB"."XA W_AP1" AND ("C#7_RD_RUN".SMC_AP1 = "C#7_RD_RUN".SMX_AP1) THEN
       "C#7_RD_RUN".SMC_AP1 := "C#7_RD_RUN".SMC_AP1 + 1.0;
   END_IF;
END_REGION
END_FUNCTION

FUNCTION "FCCA_CCD_AP1" : Void   // FC16, LAD
{ S7_Optimized_Access := 'TRUE' }
VERSION : 0.1
// stored: AutoNumber true, CodeModifiedDate 2026-01-15T16:25:54.3671983Z, CompileDate 2026-01-15T16:25:54.4076417Z, CreationDate 2026-01-15T16:24:02.4619467Z, HandleErrorsWithinBlock false, InterfaceModifiedDate 2024-08-08T03:24:33.8704482Z, IsConsistent true, IsIECCheckEnabled false, IsKnowHowProtected false, IsWriteProtected false, LibraryConformanceStatus Error: The block contains calls of single instances. Warning: The object contains access to global data blocks. Warning: The block contains direct access to inputs, outputs, bit memories, indirect access to the registry or indirect access to external memory areas that are unknown at the time of compilation., ModifiedDate 2026-01-15T16:25:54.3671983Z, ParameterModified 2024-08-08T03:24:33.8704482Z, PLCSimAdvancedSupport false, SetENOAutomatically False, StructureModified 2024-08-08T03:24:33.8704482Z, UDAEnableTagReadback false
BEGIN

REGION Network 1: Trạng thái cân Nước 1 hoặc AP1
   // Đầu tiên nó sẽ đợi một khoảng thời gian gọi là Thời gian trễ cân, sau đó nó mới đủ điều kiện để cân
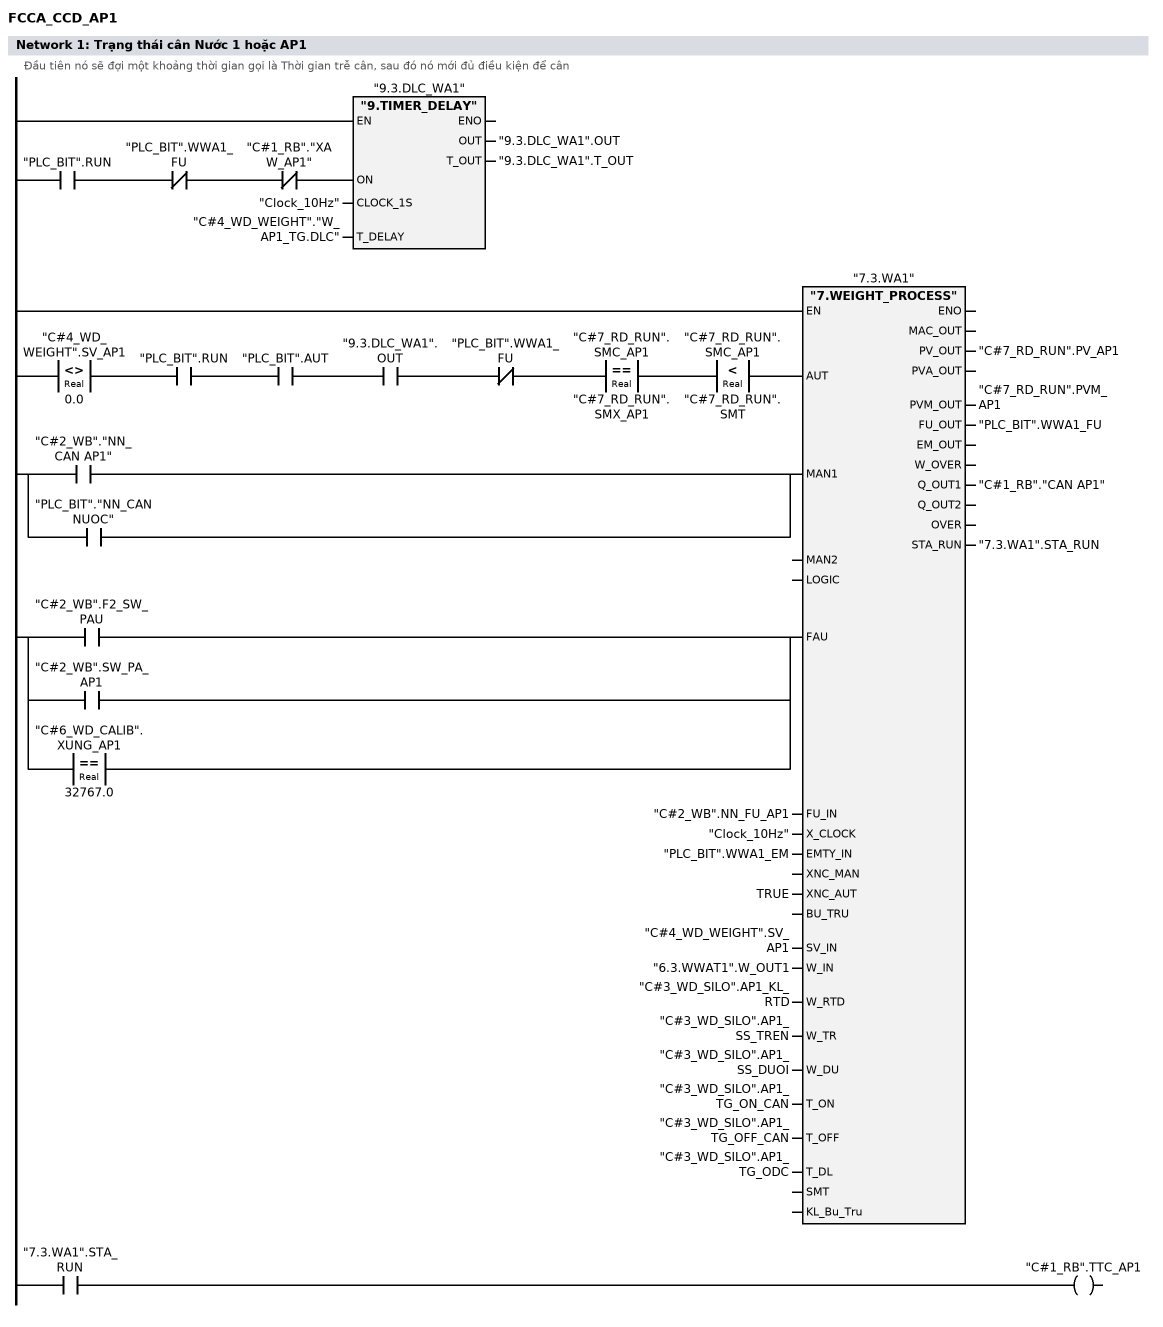
   RUNG wire#powerrail
      "9.3.DLC_WA1"(ON := wire#w1, CLOCK_1S := "Clock_10Hz", T_DELAY := "C#4_WD_WEIGHT"."W_AP1_TG.DLC", OUT => "9.3.DLC_WA1".OUT, T_OUT => "9.3.DLC_WA1".T_OUT)
   END_RUNG
   RUNG wire#powerrail
      Contact( "PLC_BIT".RUN )
      I_Contact( "PLC_BIT".WWA1_FU )
      I_Contact( "C#1_RB"."XA W_AP1" )
   END_RUNG wire#w1
   RUNG wire#powerrail
      "7.3.WA1"(AUT := wire#w2, MAN1 := wire#w3, FAU := wire#w4, MAN2 :=, LOGIC :=, FU_IN := "C#2_WB".NN_FU_AP1, X_CLOCK := "Clock_10Hz", EMTY_IN := "PLC_BIT".WWA1_EM, XNC_MAN :=, XNC_AUT := TRUE, BU_TRU :=, SV_IN := "C#4_WD_WEIGHT".SV_AP1, W_IN := "6.3.WWAT1".W_OUT1, W_RTD := "C#3_WD_SILO".AP1_KL_RTD, W_TR := "C#3_WD_SILO".AP1_SS_TREN, W_DU := "C#3_WD_SILO".AP1_SS_DUOI, T_ON := "C#3_WD_SILO".AP1_TG_ON_CAN, T_OFF := "C#3_WD_SILO".AP1_TG_OFF_CAN, T_DL := "C#3_WD_SILO".AP1_TG_ODC, SMT :=, KL_Bu_Tru :=, MAC_OUT =>, PV_OUT => "C#7_RD_RUN".PV_AP1, PVA_OUT =>, PVM_OUT => "C#7_RD_RUN".PVM_AP1, FU_OUT => "PLC_BIT".WWA1_FU, EM_OUT =>, W_OVER =>, Q_OUT1 => "C#1_RB"."CAN AP1", Q_OUT2 =>, OVER =>, STA_RUN => "7.3.WA1".STA_RUN)
   END_RUNG
   RUNG wire#powerrail
      { S7_Templates := "SrcType := Real" } NE_Contact(in1 := "C#4_WD_WEIGHT".SV_AP1, in2 := 0.0)
      Contact( "PLC_BIT".RUN )
      Contact( "PLC_BIT".AUT )
      Contact( "9.3.DLC_WA1".OUT )
      I_Contact( "PLC_BIT".WWA1_FU )
      { S7_Templates := "SrcType := Real" } EQ_Contact(in1 := "C#7_RD_RUN".SMC_AP1, in2 := "C#7_RD_RUN".SMX_AP1)
      { S7_Templates := "SrcType := Real" } LT_Contact(in1 := "C#7_RD_RUN".SMC_AP1, in2 := "C#7_RD_RUN".SMT)
   END_RUNG wire#w2
   RUNG wire#powerrail
      Contact( "C#2_WB"."NN_CAN AP1" )
   END_RUNG wire#w3
   RUNG wire#powerrail
      Contact( "PLC_BIT"."NN_CAN NUOC" )
   END_RUNG wire#w3
   RUNG wire#powerrail
      Contact( "C#2_WB".F2_SW_PAU )
   END_RUNG wire#w4
   RUNG wire#powerrail
      Contact( "C#2_WB".SW_PA_AP1 )
   END_RUNG wire#w4
   RUNG wire#powerrail
      { S7_Templates := "SrcType := Real" } EQ_Contact(in1 := "C#6_WD_CALIB".XUNG_AP1, in2 := 32767.0)
   END_RUNG wire#w4
   RUNG wire#powerrail
      Contact( "7.3.WA1".STA_RUN )
      Coil( "C#1_RB".TTC_AP1 )
   END_RUNG
   // the same network as SCL:
   "9.3.DLC_WA1"(ON := "PLC_BIT".RUN AND NOT "PLC_BIT".WWA1_FU AND NOT "C#1_RB"."XA W_AP1",   // "9.TIMER_DELAY"
                 CLOCK_1S := "Clock_10Hz",
                 T_DELAY := "C#4_WD_WEIGHT"."W_AP1_TG.DLC",
                 OUT => "9.3.DLC_WA1".OUT,
                 T_OUT => "9.3.DLC_WA1".T_OUT);
   "7.3.WA1"(AUT := ("C#4_WD_WEIGHT".SV_AP1 <> 0.0) AND "PLC_BIT".RUN AND "PLC_BIT".AUT AND "9.3.DLC_WA1".OUT AND NOT "PLC_BIT".WWA1_FU AND ("C#7_RD_RUN".SMC_AP1 = "C#7_RD_RUN".SMX_AP1) AND ("C#7_RD_RUN".SMC_AP1 < "C#7_RD_RUN".SMT),   // "7.WEIGHT_PROCESS"
             MAN1 := "C#2_WB"."NN_CAN AP1" OR "PLC_BIT"."NN_CAN NUOC",
             FAU := "C#2_WB".F2_SW_PAU OR "C#2_WB".SW_PA_AP1 OR ("C#6_WD_CALIB".XUNG_AP1 = 32767.0),
             FU_IN := "C#2_WB".NN_FU_AP1,
             X_CLOCK := "Clock_10Hz",
             EMTY_IN := "PLC_BIT".WWA1_EM,
             XNC_AUT := TRUE,
             SV_IN := "C#4_WD_WEIGHT".SV_AP1,
             W_IN := "6.3.WWAT1".W_OUT1,
             W_RTD := "C#3_WD_SILO".AP1_KL_RTD,
             W_TR := "C#3_WD_SILO".AP1_SS_TREN,
             W_DU := "C#3_WD_SILO".AP1_SS_DUOI,
             T_ON := "C#3_WD_SILO".AP1_TG_ON_CAN,
             T_OFF := "C#3_WD_SILO".AP1_TG_OFF_CAN,
             T_DL := "C#3_WD_SILO".AP1_TG_ODC,
             PV_OUT => "C#7_RD_RUN".PV_AP1,
             PVM_OUT => "C#7_RD_RUN".PVM_AP1,
             FU_OUT => "PLC_BIT".WWA1_FU,
             Q_OUT1 => "C#1_RB"."CAN AP1",
             STA_RUN => "7.3.WA1".STA_RUN);
   "C#1_RB".TTC_AP1 := "7.3.WA1".STA_RUN;
END_REGION
END_FUNCTION

FUNCTION "FCXL_CCD_SB1" : Void   // FC17, LAD
{ S7_Optimized_Access := 'TRUE' }
VERSION : 0.1
// stored: AutoNumber true, CodeModifiedDate 2026-01-15T16:25:52.9899247Z, CompileDate 2026-01-15T16:25:53.1527483Z, CreationDate 2026-01-15T16:24:02.4619467Z, HandleErrorsWithinBlock false, InterfaceModifiedDate 2024-08-08T03:53:18.695573Z, IsConsistent true, IsIECCheckEnabled false, IsKnowHowProtected false, IsWriteProtected false, LibraryConformanceStatus Error: The block contains calls of single instances. Warning: The object contains access to global data blocks. Warning: The block contains direct access to inputs, outputs, bit memories, indirect access to the registry or indirect access to external memory areas that are unknown at the time of compilation., ModifiedDate 2026-01-15T16:25:52.9899247Z, ParameterModified 2024-08-08T03:53:18.695573Z, PLCSimAdvancedSupport false, SetENOAutomatically False, StructureModified 2024-08-08T03:53:18.695573Z, UDAEnableTagReadback false
   VAR_TEMP   // added for the SCL form of the ladder/FBD networks
      _w1 : Bool;
      _w2 : Bool;
      _w3 : Bool;
   END_VAR
BEGIN

REGION Network 1: Cân phụ gia 1 Full
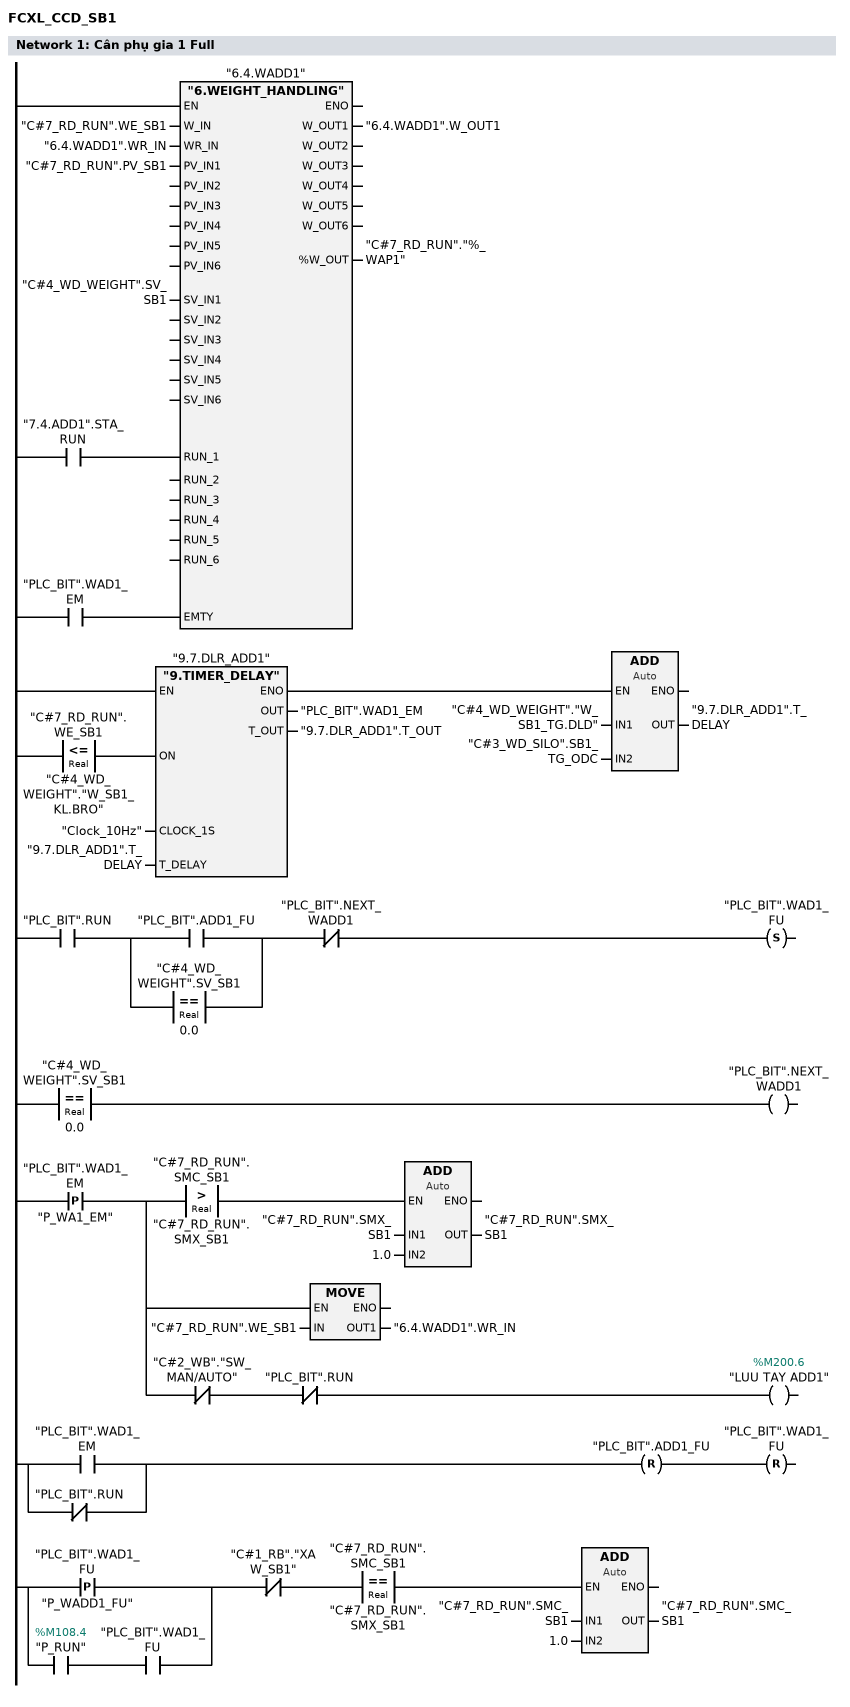
   RUNG wire#powerrail
      "6.4.WADD1"(RUN_1 := wire#w1, EMTY := wire#w2, W_IN := "C#7_RD_RUN".WE_SB1, WR_IN := "6.4.WADD1".WR_IN, PV_IN1 := "C#7_RD_RUN".PV_SB1, PV_IN2 :=, PV_IN3 :=, PV_IN4 :=, PV_IN5 :=, PV_IN6 :=, SV_IN1 := "C#4_WD_WEIGHT".SV_SB1, SV_IN2 :=, SV_IN3 :=, SV_IN4 :=, SV_IN5 :=, SV_IN6 :=, RUN_2 :=, RUN_3 :=, RUN_4 :=, RUN_5 :=, RUN_6 :=, W_OUT1 => "6.4.WADD1".W_OUT1, W_OUT2 =>, W_OUT3 =>, W_OUT4 =>, W_OUT5 =>, W_OUT6 =>, "%W_OUT" => "C#7_RD_RUN"."%_WAP1")
   END_RUNG
   RUNG wire#powerrail
      Contact( "7.4.ADD1".STA_RUN )
   END_RUNG wire#w1
   RUNG wire#powerrail
      Contact( "PLC_BIT".WAD1_EM )
   END_RUNG wire#w2
   RUNG wire#powerrail
      "9.7.DLR_ADD1"(ON := wire#w3, CLOCK_1S := "Clock_10Hz", T_DELAY := "9.7.DLR_ADD1".T_DELAY, OUT => "PLC_BIT".WAD1_EM, T_OUT => "9.7.DLR_ADD1".T_OUT)
      Add(in1 := "C#4_WD_WEIGHT"."W_SB1_TG.DLD", in2 := "C#3_WD_SILO".SB1_TG_ODC, out => "9.7.DLR_ADD1".T_DELAY)
   END_RUNG
   RUNG wire#powerrail
      { S7_Templates := "SrcType := Real" } LE_Contact(in1 := "C#7_RD_RUN".WE_SB1, in2 := "C#4_WD_WEIGHT"."W_SB1_KL.BRO")
   END_RUNG wire#w3
   RUNG wire#powerrail
      Contact( "PLC_BIT".RUN )
      wire#w4
      Contact( "PLC_BIT".ADD1_FU )
      wire#w5
      I_Contact( "PLC_BIT".NEXT_WADD1 )
      S_Coil( "PLC_BIT".WAD1_FU )
   END_RUNG
   RUNG wire#w4
      { S7_Templates := "SrcType := Real" } EQ_Contact(in1 := "C#4_WD_WEIGHT".SV_SB1, in2 := 0.0)
   END_RUNG wire#w5
   RUNG wire#powerrail
      { S7_Templates := "SrcType := Real" } EQ_Contact(in1 := "C#4_WD_WEIGHT".SV_SB1, in2 := 0.0)
      Coil( "PLC_BIT".NEXT_WADD1 )
   END_RUNG
   RUNG wire#powerrail
      P_Contact(operand := "PLC_BIT".WAD1_EM, bit := "P_WA1_EM")
      wire#w6
      { S7_Templates := "SrcType := Real" } GT_Contact(in1 := "C#7_RD_RUN".SMC_SB1, in2 := "C#7_RD_RUN".SMX_SB1)
      Add(in1 := "C#7_RD_RUN".SMX_SB1, in2 := 1.0, out => "C#7_RD_RUN".SMX_SB1)
   END_RUNG
   RUNG wire#w6
      Move(in := "C#7_RD_RUN".WE_SB1, out1 => "6.4.WADD1".WR_IN)
   END_RUNG
   RUNG wire#w6
      I_Contact( "C#2_WB"."SW_MAN/AUTO" )
      I_Contact( "PLC_BIT".RUN )
      Coil( "LUU TAY ADD1" )
   END_RUNG
   RUNG wire#powerrail
      Contact( "PLC_BIT".WAD1_EM )
      wire#w7
      R_Coil( "PLC_BIT".ADD1_FU )
      R_Coil( "PLC_BIT".WAD1_FU )
   END_RUNG
   RUNG wire#powerrail
      I_Contact( "PLC_BIT".RUN )
   END_RUNG wire#w7
   RUNG wire#powerrail
      P_Contact(operand := "PLC_BIT".WAD1_FU, bit := "P_WADD1_FU")
      wire#w8
      I_Contact( "C#1_RB"."XA W_SB1" )
      { S7_Templates := "SrcType := Real" } EQ_Contact(in1 := "C#7_RD_RUN".SMC_SB1, in2 := "C#7_RD_RUN".SMX_SB1)
      Add(in1 := "C#7_RD_RUN".SMC_SB1, in2 := 1.0, out => "C#7_RD_RUN".SMC_SB1)
   END_RUNG
   RUNG wire#powerrail
      Contact( "P_RUN" )
      Contact( "PLC_BIT".WAD1_FU )
   END_RUNG wire#w8
   // the same network as SCL:
   "6.4.WADD1"(W_IN := "C#7_RD_RUN".WE_SB1,   // "6.WEIGHT_HANDLING"
               WR_IN := "6.4.WADD1".WR_IN,
               PV_IN1 := "C#7_RD_RUN".PV_SB1,
               SV_IN1 := "C#4_WD_WEIGHT".SV_SB1,
               RUN_1 := "7.4.ADD1".STA_RUN,
               EMTY := "PLC_BIT".WAD1_EM,
               W_OUT1 => "6.4.WADD1".W_OUT1,
               "%W_OUT" => "C#7_RD_RUN"."%_WAP1");
   "9.7.DLR_ADD1"(ON := "C#7_RD_RUN".WE_SB1 <= "C#4_WD_WEIGHT"."W_SB1_KL.BRO",   // "9.TIMER_DELAY"
                  CLOCK_1S := "Clock_10Hz",
                  T_DELAY := "9.7.DLR_ADD1".T_DELAY,
                  OUT => "PLC_BIT".WAD1_EM,
                  T_OUT => "9.7.DLR_ADD1".T_OUT,
                  ENO => #_w1);
   IF #_w1 THEN "9.7.DLR_ADD1".T_DELAY := "C#4_WD_WEIGHT"."W_SB1_TG.DLD" + "C#3_WD_SILO".SB1_TG_ODC; END_IF;
   IF "PLC_BIT".RUN AND ("PLC_BIT".ADD1_FU OR ("C#4_WD_WEIGHT".SV_SB1 = 0.0)) AND NOT "PLC_BIT".NEXT_WADD1 THEN
       "PLC_BIT".WAD1_FU := TRUE;
   END_IF;
   "PLC_BIT".NEXT_WADD1 := "C#4_WD_WEIGHT".SV_SB1 = 0.0;
   #_w2 := "PLC_BIT".WAD1_EM AND NOT "P_WA1_EM";   // rising edge of "PLC_BIT".WAD1_EM
   "P_WA1_EM" := "PLC_BIT".WAD1_EM;
   IF #_w2 AND ("C#7_RD_RUN".SMC_SB1 > "C#7_RD_RUN".SMX_SB1) THEN
       "C#7_RD_RUN".SMX_SB1 := "C#7_RD_RUN".SMX_SB1 + 1.0;
   END_IF;
   IF #_w2 THEN "6.4.WADD1".WR_IN := "C#7_RD_RUN".WE_SB1; END_IF;
   "LUU TAY ADD1" := #_w2 AND NOT "C#2_WB"."SW_MAN/AUTO" AND NOT "PLC_BIT".RUN;
   IF "PLC_BIT".WAD1_EM OR NOT "PLC_BIT".RUN THEN
       "PLC_BIT".ADD1_FU := FALSE;
       "PLC_BIT".WAD1_FU := FALSE;
   END_IF;
   #_w3 := "PLC_BIT".WAD1_FU AND NOT "P_WADD1_FU";   // rising edge of "PLC_BIT".WAD1_FU
   "P_WADD1_FU" := "PLC_BIT".WAD1_FU;
   IF (#_w3 OR ("P_RUN" AND "PLC_BIT".WAD1_FU)) AND NOT "C#1_RB"."XA W_SB1" AND ("C#7_RD_RUN".SMC_SB1 = "C#7_RD_RUN".SMX_SB1) THEN
       "C#7_RD_RUN".SMC_SB1 := "C#7_RD_RUN".SMC_SB1 + 1.0;
   END_IF;
END_REGION
END_FUNCTION

FUNCTION "FCCA_CCD_SB1" : Void   // FC18, LAD
{ S7_Optimized_Access := 'TRUE' }
VERSION : 0.1
// stored: AutoNumber true, CodeModifiedDate 2026-01-15T16:25:53.9559646Z, CompileDate 2026-01-15T16:25:53.9939929Z, CreationDate 2026-01-15T16:24:02.4619467Z, HandleErrorsWithinBlock false, InterfaceModifiedDate 2024-08-08T03:53:53.300462Z, IsConsistent true, IsIECCheckEnabled false, IsKnowHowProtected false, IsWriteProtected false, LibraryConformanceStatus Error: The block contains calls of single instances. Warning: The object contains access to global data blocks. Warning: The block contains direct access to inputs, outputs, bit memories, indirect access to the registry or indirect access to external memory areas that are unknown at the time of compilation., ModifiedDate 2026-01-15T16:25:53.9559646Z, ParameterModified 2024-08-08T03:53:53.300462Z, PLCSimAdvancedSupport false, SetENOAutomatically False, StructureModified 2024-08-08T03:53:53.300462Z, UDAEnableTagReadback false
BEGIN

REGION Network 1: CAN PHU GIA 1
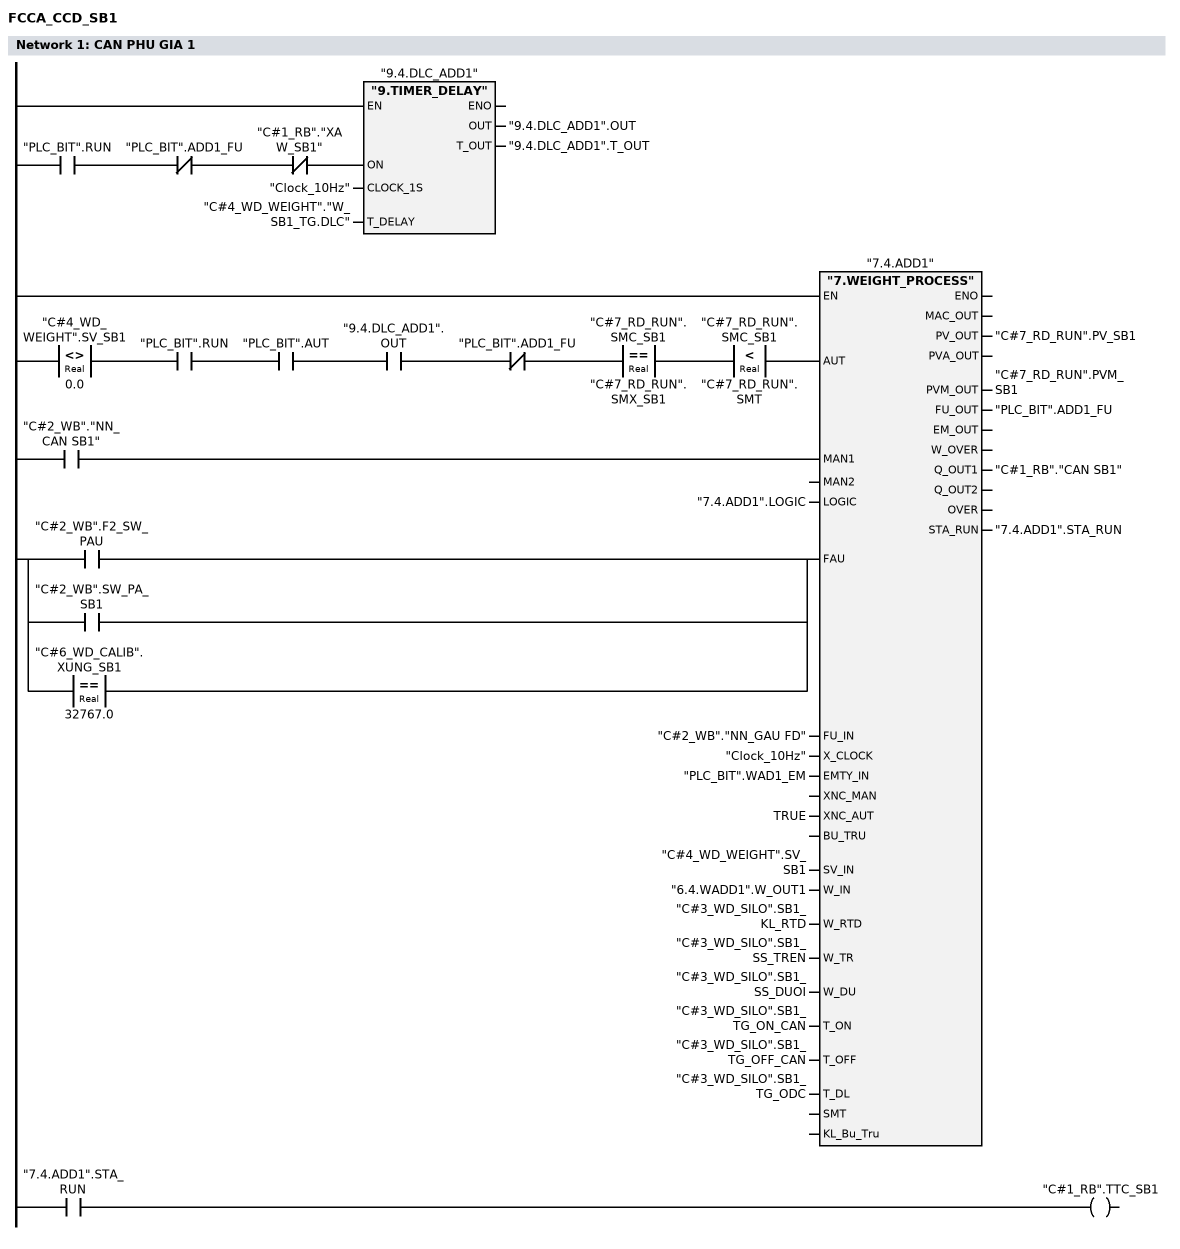
   RUNG wire#powerrail
      "9.4.DLC_ADD1"(ON := wire#w1, CLOCK_1S := "Clock_10Hz", T_DELAY := "C#4_WD_WEIGHT"."W_SB1_TG.DLC", OUT => "9.4.DLC_ADD1".OUT, T_OUT => "9.4.DLC_ADD1".T_OUT)
   END_RUNG
   RUNG wire#powerrail
      Contact( "PLC_BIT".RUN )
      I_Contact( "PLC_BIT".ADD1_FU )
      I_Contact( "C#1_RB"."XA W_SB1" )
   END_RUNG wire#w1
   RUNG wire#powerrail
      "7.4.ADD1"(AUT := wire#w2, MAN1 := wire#w3, FAU := wire#w4, MAN2 :=, LOGIC := "7.4.ADD1".LOGIC, FU_IN := "C#2_WB"."NN_GAU FD", X_CLOCK := "Clock_10Hz", EMTY_IN := "PLC_BIT".WAD1_EM, XNC_MAN :=, XNC_AUT := TRUE, BU_TRU :=, SV_IN := "C#4_WD_WEIGHT".SV_SB1, W_IN := "6.4.WADD1".W_OUT1, W_RTD := "C#3_WD_SILO".SB1_KL_RTD, W_TR := "C#3_WD_SILO".SB1_SS_TREN, W_DU := "C#3_WD_SILO".SB1_SS_DUOI, T_ON := "C#3_WD_SILO".SB1_TG_ON_CAN, T_OFF := "C#3_WD_SILO".SB1_TG_OFF_CAN, T_DL := "C#3_WD_SILO".SB1_TG_ODC, SMT :=, KL_Bu_Tru :=, MAC_OUT =>, PV_OUT => "C#7_RD_RUN".PV_SB1, PVA_OUT =>, PVM_OUT => "C#7_RD_RUN".PVM_SB1, FU_OUT => "PLC_BIT".ADD1_FU, EM_OUT =>, W_OVER =>, Q_OUT1 => "C#1_RB"."CAN SB1", Q_OUT2 =>, OVER =>, STA_RUN => "7.4.ADD1".STA_RUN)
   END_RUNG
   RUNG wire#powerrail
      { S7_Templates := "SrcType := Real" } NE_Contact(in1 := "C#4_WD_WEIGHT".SV_SB1, in2 := 0.0)
      Contact( "PLC_BIT".RUN )
      Contact( "PLC_BIT".AUT )
      Contact( "9.4.DLC_ADD1".OUT )
      I_Contact( "PLC_BIT".ADD1_FU )
      { S7_Templates := "SrcType := Real" } EQ_Contact(in1 := "C#7_RD_RUN".SMC_SB1, in2 := "C#7_RD_RUN".SMX_SB1)
      { S7_Templates := "SrcType := Real" } LT_Contact(in1 := "C#7_RD_RUN".SMC_SB1, in2 := "C#7_RD_RUN".SMT)
   END_RUNG wire#w2
   RUNG wire#powerrail
      Contact( "C#2_WB"."NN_CAN SB1" )
   END_RUNG wire#w3
   RUNG wire#powerrail
      Contact( "C#2_WB".F2_SW_PAU )
   END_RUNG wire#w4
   RUNG wire#powerrail
      Contact( "C#2_WB".SW_PA_SB1 )
   END_RUNG wire#w4
   RUNG wire#powerrail
      { S7_Templates := "SrcType := Real" } EQ_Contact(in1 := "C#6_WD_CALIB".XUNG_SB1, in2 := 32767.0)
   END_RUNG wire#w4
   RUNG wire#powerrail
      Contact( "7.4.ADD1".STA_RUN )
      Coil( "C#1_RB".TTC_SB1 )
   END_RUNG
   // the same network as SCL:
   "9.4.DLC_ADD1"(ON := "PLC_BIT".RUN AND NOT "PLC_BIT".ADD1_FU AND NOT "C#1_RB"."XA W_SB1",   // "9.TIMER_DELAY"
                  CLOCK_1S := "Clock_10Hz",
                  T_DELAY := "C#4_WD_WEIGHT"."W_SB1_TG.DLC",
                  OUT => "9.4.DLC_ADD1".OUT,
                  T_OUT => "9.4.DLC_ADD1".T_OUT);
   "7.4.ADD1"(AUT := ("C#4_WD_WEIGHT".SV_SB1 <> 0.0) AND "PLC_BIT".RUN AND "PLC_BIT".AUT AND "9.4.DLC_ADD1".OUT AND NOT "PLC_BIT".ADD1_FU AND ("C#7_RD_RUN".SMC_SB1 = "C#7_RD_RUN".SMX_SB1) AND ("C#7_RD_RUN".SMC_SB1 < "C#7_RD_RUN".SMT),   // "7.WEIGHT_PROCESS"
              MAN1 := "C#2_WB"."NN_CAN SB1",
              LOGIC := "7.4.ADD1".LOGIC,
              FAU := "C#2_WB".F2_SW_PAU OR "C#2_WB".SW_PA_SB1 OR ("C#6_WD_CALIB".XUNG_SB1 = 32767.0),
              FU_IN := "C#2_WB"."NN_GAU FD",
              X_CLOCK := "Clock_10Hz",
              EMTY_IN := "PLC_BIT".WAD1_EM,
              XNC_AUT := TRUE,
              SV_IN := "C#4_WD_WEIGHT".SV_SB1,
              W_IN := "6.4.WADD1".W_OUT1,
              W_RTD := "C#3_WD_SILO".SB1_KL_RTD,
              W_TR := "C#3_WD_SILO".SB1_SS_TREN,
              W_DU := "C#3_WD_SILO".SB1_SS_DUOI,
              T_ON := "C#3_WD_SILO".SB1_TG_ON_CAN,
              T_OFF := "C#3_WD_SILO".SB1_TG_OFF_CAN,
              T_DL := "C#3_WD_SILO".SB1_TG_ODC,
              PV_OUT => "C#7_RD_RUN".PV_SB1,
              PVM_OUT => "C#7_RD_RUN".PVM_SB1,
              FU_OUT => "PLC_BIT".ADD1_FU,
              Q_OUT1 => "C#1_RB"."CAN SB1",
              STA_RUN => "7.4.ADD1".STA_RUN);
   "C#1_RB".TTC_SB1 := "7.4.ADD1".STA_RUN;
END_REGION
END_FUNCTION

FUNCTION "5. QUA TRINH NAP LIEU" : Void   // FC5, LAD
{ S7_Optimized_Access := 'TRUE' }
VERSION : 0.1
// stored: AutoNumber true, CodeModifiedDate 2026-01-15T16:25:52.514227Z, CompileDate 2026-01-15T16:25:52.5840608Z, CreationDate 2026-01-15T16:22:49.8270549Z, HandleErrorsWithinBlock false, InterfaceModifiedDate 2023-12-12T15:54:48.677177Z, IsConsistent true, IsIECCheckEnabled false, IsKnowHowProtected false, IsWriteProtected false, LibraryConformanceStatus Warning: The object contains access to global data blocks. Warning: The block contains direct access to inputs, outputs, bit memories, indirect access to the registry or indirect access to external memory areas that are unknown at the time of compilation., ModifiedDate 2026-01-15T16:25:52.514227Z, ParameterModified 2023-12-12T15:54:48.677177Z, PLCSimAdvancedSupport false, SetENOAutomatically False, StructureModified 2023-12-12T15:54:48.677177Z, UDAEnableTagReadback false
   VAR_OUTPUT
      XA_PTG : Bool;
      XA_CEM1 : Bool;
      XA_CEM2 : Bool;
      XA_WAT1 : Bool;
      XA_WAT2 : Bool;
      XA_ADD1 : Bool;
      XA_ADD2 : Bool;
   END_VAR
BEGIN

REGION Network 1: Van xả phễu chờ
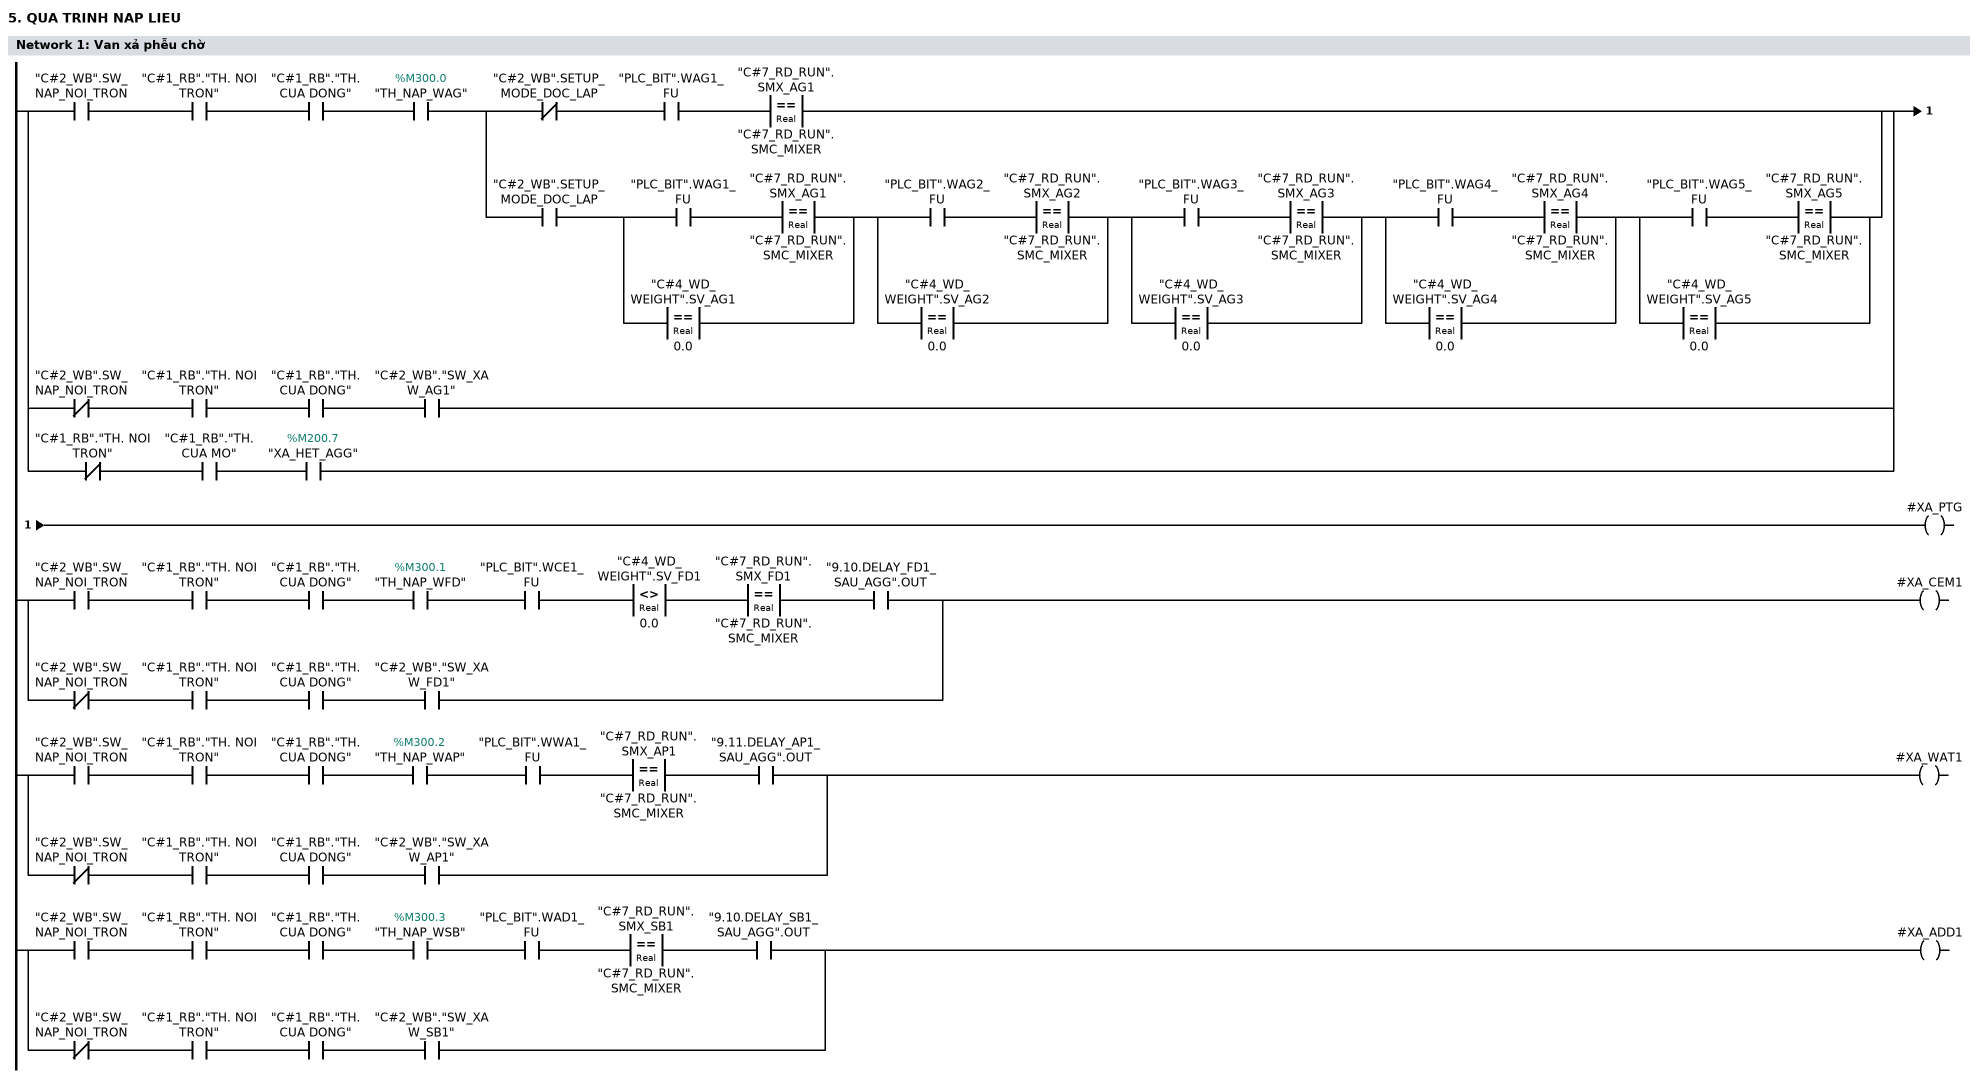
   RUNG wire#powerrail
      Contact( "C#2_WB".SW_NAP_NOI_TRON )
      Contact( "C#1_RB"."TH. NOI TRON" )
      Contact( "C#1_RB"."TH. CUA DONG" )
      Contact( "TH_NAP_WAG" )
      wire#w1
      I_Contact( "C#2_WB".SETUP_MODE_DOC_LAP )
      Contact( "PLC_BIT".WAG1_FU )
      { S7_Templates := "SrcType := Real" } EQ_Contact(in1 := "C#7_RD_RUN".SMX_AG1, in2 := "C#7_RD_RUN".SMC_MIXER)
      wire#w2
      Coil( #XA_PTG )
   END_RUNG
   RUNG wire#w1
      Contact( "C#2_WB".SETUP_MODE_DOC_LAP )
      wire#w3
      Contact( "PLC_BIT".WAG1_FU )
      { S7_Templates := "SrcType := Real" } EQ_Contact(in1 := "C#7_RD_RUN".SMX_AG1, in2 := "C#7_RD_RUN".SMC_MIXER)
      wire#w4
      Contact( "PLC_BIT".WAG2_FU )
      { S7_Templates := "SrcType := Real" } EQ_Contact(in1 := "C#7_RD_RUN".SMX_AG2, in2 := "C#7_RD_RUN".SMC_MIXER)
      wire#w5
      Contact( "PLC_BIT".WAG3_FU )
      { S7_Templates := "SrcType := Real" } EQ_Contact(in1 := "C#7_RD_RUN".SMX_AG3, in2 := "C#7_RD_RUN".SMC_MIXER)
      wire#w6
      Contact( "PLC_BIT".WAG4_FU )
      { S7_Templates := "SrcType := Real" } EQ_Contact(in1 := "C#7_RD_RUN".SMX_AG4, in2 := "C#7_RD_RUN".SMC_MIXER)
      wire#w7
      Contact( "PLC_BIT".WAG5_FU )
      { S7_Templates := "SrcType := Real" } EQ_Contact(in1 := "C#7_RD_RUN".SMX_AG5, in2 := "C#7_RD_RUN".SMC_MIXER)
   END_RUNG wire#w2
   RUNG wire#w3
      { S7_Templates := "SrcType := Real" } EQ_Contact(in1 := "C#4_WD_WEIGHT".SV_AG1, in2 := 0.0)
   END_RUNG wire#w4
   RUNG wire#w4
      { S7_Templates := "SrcType := Real" } EQ_Contact(in1 := "C#4_WD_WEIGHT".SV_AG2, in2 := 0.0)
   END_RUNG wire#w5
   RUNG wire#w5
      { S7_Templates := "SrcType := Real" } EQ_Contact(in1 := "C#4_WD_WEIGHT".SV_AG3, in2 := 0.0)
   END_RUNG wire#w6
   RUNG wire#w6
      { S7_Templates := "SrcType := Real" } EQ_Contact(in1 := "C#4_WD_WEIGHT".SV_AG4, in2 := 0.0)
   END_RUNG wire#w7
   RUNG wire#w7
      { S7_Templates := "SrcType := Real" } EQ_Contact(in1 := "C#4_WD_WEIGHT".SV_AG5, in2 := 0.0)
   END_RUNG wire#w2
   RUNG wire#powerrail
      I_Contact( "C#2_WB".SW_NAP_NOI_TRON )
      Contact( "C#1_RB"."TH. NOI TRON" )
      Contact( "C#1_RB"."TH. CUA DONG" )
      Contact( "C#2_WB"."SW_XA W_AG1" )
   END_RUNG wire#w2
   RUNG wire#powerrail
      I_Contact( "C#1_RB"."TH. NOI TRON" )
      Contact( "C#1_RB"."TH. CUA MO" )
      Contact( "XA_HET_AGG" )
   END_RUNG wire#w2
   RUNG wire#powerrail
      Contact( "C#2_WB".SW_NAP_NOI_TRON )
      Contact( "C#1_RB"."TH. NOI TRON" )
      Contact( "C#1_RB"."TH. CUA DONG" )
      Contact( "TH_NAP_WFD" )
      Contact( "PLC_BIT".WCE1_FU )
      { S7_Templates := "SrcType := Real" } NE_Contact(in1 := "C#4_WD_WEIGHT".SV_FD1, in2 := 0.0)
      { S7_Templates := "SrcType := Real" } EQ_Contact(in1 := "C#7_RD_RUN".SMX_FD1, in2 := "C#7_RD_RUN".SMC_MIXER)
      Contact( "9.10.DELAY_FD1_SAU_AGG".OUT )
      wire#w8
      Coil( #XA_CEM1 )
   END_RUNG
   RUNG wire#powerrail
      I_Contact( "C#2_WB".SW_NAP_NOI_TRON )
      Contact( "C#1_RB"."TH. NOI TRON" )
      Contact( "C#1_RB"."TH. CUA DONG" )
      Contact( "C#2_WB"."SW_XA W_FD1" )
   END_RUNG wire#w8
   RUNG wire#powerrail
      Contact( "C#2_WB".SW_NAP_NOI_TRON )
      Contact( "C#1_RB"."TH. NOI TRON" )
      Contact( "C#1_RB"."TH. CUA DONG" )
      Contact( "TH_NAP_WAP" )
      Contact( "PLC_BIT".WWA1_FU )
      { S7_Templates := "SrcType := Real" } EQ_Contact(in1 := "C#7_RD_RUN".SMX_AP1, in2 := "C#7_RD_RUN".SMC_MIXER)
      Contact( "9.11.DELAY_AP1_SAU_AGG".OUT )
      wire#w9
      Coil( #XA_WAT1 )
   END_RUNG
   RUNG wire#powerrail
      I_Contact( "C#2_WB".SW_NAP_NOI_TRON )
      Contact( "C#1_RB"."TH. NOI TRON" )
      Contact( "C#1_RB"."TH. CUA DONG" )
      Contact( "C#2_WB"."SW_XA W_AP1" )
   END_RUNG wire#w9
   RUNG wire#powerrail
      Contact( "C#2_WB".SW_NAP_NOI_TRON )
      Contact( "C#1_RB"."TH. NOI TRON" )
      Contact( "C#1_RB"."TH. CUA DONG" )
      Contact( "TH_NAP_WSB" )
      Contact( "PLC_BIT".WAD1_FU )
      { S7_Templates := "SrcType := Real" } EQ_Contact(in1 := "C#7_RD_RUN".SMX_SB1, in2 := "C#7_RD_RUN".SMC_MIXER)
      Contact( "9.10.DELAY_SB1_SAU_AGG".OUT )
      wire#w10
      Coil( #XA_ADD1 )
   END_RUNG
   RUNG wire#powerrail
      I_Contact( "C#2_WB".SW_NAP_NOI_TRON )
      Contact( "C#1_RB"."TH. NOI TRON" )
      Contact( "C#1_RB"."TH. CUA DONG" )
      Contact( "C#2_WB"."SW_XA W_SB1" )
   END_RUNG wire#w10
   // the same network as SCL:
   #XA_PTG := ("C#2_WB".SW_NAP_NOI_TRON AND "C#1_RB"."TH. NOI TRON" AND "C#1_RB"."TH. CUA DONG" AND "TH_NAP_WAG" AND ((NOT "C#2_WB".SETUP_MODE_DOC_LAP AND "PLC_BIT".WAG1_FU AND ("C#7_RD_RUN".SMX_AG1 = "C#7_RD_RUN".SMC_MIXER)) OR ("C#2_WB".SETUP_MODE_DOC_LAP AND (("PLC_BIT".WAG1_FU AND ("C#7_RD_RUN".SMX_AG1 = "C#7_RD_RUN".SMC_MIXER)) OR ("C#4_WD_WEIGHT".SV_AG1 = 0.0)) AND (("PLC_BIT".WAG2_FU AND ("C#7_RD_RUN".SMX_AG2 = "C#7_RD_RUN".SMC_MIXER)) OR ("C#4_WD_WEIGHT".SV_AG2 = 0.0)) AND (("PLC_BIT".WAG3_FU AND ("C#7_RD_RUN".SMX_AG3 = "C#7_RD_RUN".SMC_MIXER)) OR ("C#4_WD_WEIGHT".SV_AG3 = 0.0)) AND (("PLC_BIT".WAG4_FU AND ("C#7_RD_RUN".SMX_AG4 = "C#7_RD_RUN".SMC_MIXER)) OR ("C#4_WD_WEIGHT".SV_AG4 = 0.0)) AND (("PLC_BIT".WAG5_FU AND ("C#7_RD_RUN".SMX_AG5 = "C#7_RD_RUN".SMC_MIXER)) OR ("C#4_WD_WEIGHT".SV_AG5 = 0.0))))) OR (NOT "C#2_WB".SW_NAP_NOI_TRON AND "C#1_RB"."TH. NOI TRON" AND "C#1_RB"."TH. CUA DONG" AND "C#2_WB"."SW_XA W_AG1") OR (NOT "C#1_RB"."TH. NOI TRON" AND "C#1_RB"."TH. CUA MO" AND "XA_HET_AGG");
   #XA_CEM1 := ("C#2_WB".SW_NAP_NOI_TRON AND "C#1_RB"."TH. NOI TRON" AND "C#1_RB"."TH. CUA DONG" AND "TH_NAP_WFD" AND "PLC_BIT".WCE1_FU AND ("C#4_WD_WEIGHT".SV_FD1 <> 0.0) AND ("C#7_RD_RUN".SMX_FD1 = "C#7_RD_RUN".SMC_MIXER) AND "9.10.DELAY_FD1_SAU_AGG".OUT) OR (NOT "C#2_WB".SW_NAP_NOI_TRON AND "C#1_RB"."TH. NOI TRON" AND "C#1_RB"."TH. CUA DONG" AND "C#2_WB"."SW_XA W_FD1");
   #XA_WAT1 := ("C#2_WB".SW_NAP_NOI_TRON AND "C#1_RB"."TH. NOI TRON" AND "C#1_RB"."TH. CUA DONG" AND "TH_NAP_WAP" AND "PLC_BIT".WWA1_FU AND ("C#7_RD_RUN".SMX_AP1 = "C#7_RD_RUN".SMC_MIXER) AND "9.11.DELAY_AP1_SAU_AGG".OUT) OR (NOT "C#2_WB".SW_NAP_NOI_TRON AND "C#1_RB"."TH. NOI TRON" AND "C#1_RB"."TH. CUA DONG" AND "C#2_WB"."SW_XA W_AP1");
   #XA_ADD1 := ("C#2_WB".SW_NAP_NOI_TRON AND "C#1_RB"."TH. NOI TRON" AND "C#1_RB"."TH. CUA DONG" AND "TH_NAP_WSB" AND "PLC_BIT".WAD1_FU AND ("C#7_RD_RUN".SMX_SB1 = "C#7_RD_RUN".SMC_MIXER) AND "9.10.DELAY_SB1_SAU_AGG".OUT) OR (NOT "C#2_WB".SW_NAP_NOI_TRON AND "C#1_RB"."TH. NOI TRON" AND "C#1_RB"."TH. CUA DONG" AND "C#2_WB"."SW_XA W_SB1");
END_REGION
END_FUNCTION

FUNCTION "7. SAVE_REPORT" : Void   // FC7, LAD
{ S7_Optimized_Access := 'TRUE' }
VERSION : 0.1
// stored: AutoNumber false, CodeModifiedDate 2026-01-15T16:25:53.2342694Z, CompileDate 2026-01-15T16:25:53.2888298Z, CreationDate 2026-01-15T16:22:49.8270549Z, HandleErrorsWithinBlock false, InterfaceModifiedDate 2023-12-15T06:44:57.8941631Z, IsConsistent true, IsIECCheckEnabled false, IsKnowHowProtected false, IsWriteProtected false, LibraryConformanceStatus Warning: The object contains access to global data blocks. Warning: The block contains direct access to inputs, outputs, bit memories, indirect access to the registry or indirect access to external memory areas that are unknown at the time of compilation., ModifiedDate 2026-01-15T16:25:53.2342694Z, ParameterModified 2023-12-15T06:44:57.8941631Z, PLCSimAdvancedSupport false, SetENOAutomatically False, StructureModified 2023-12-15T06:44:57.8941631Z, UDAEnableTagReadback false
   VAR_TEMP   // added for the SCL form of the ladder/FBD networks
      _w1 : Bool;
   END_VAR
BEGIN

REGION Network 1: Lưu dữ liệu Cốt liệu
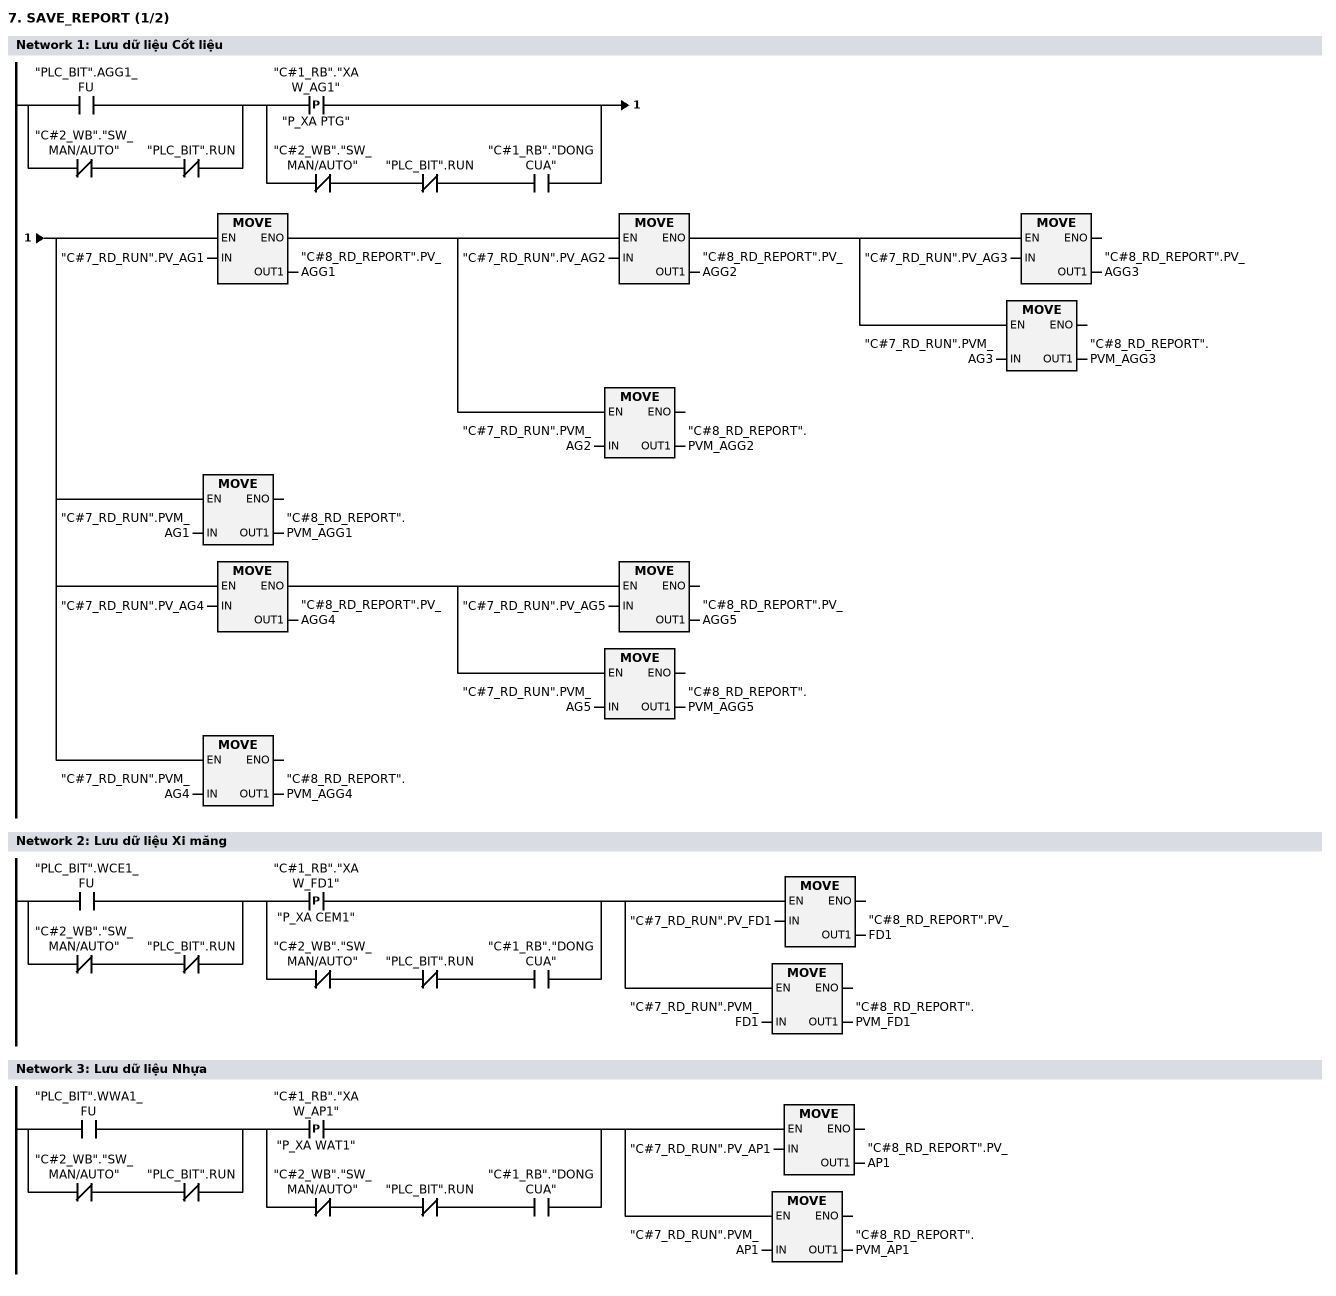
   RUNG wire#powerrail
      Contact( "PLC_BIT".AGG1_FU )
      wire#w1
      P_Contact(operand := "C#1_RB"."XA W_AG1", bit := "P_XA PTG")
      wire#w2
      Move(in := "C#7_RD_RUN".PV_AG1, out1 => "C#8_RD_REPORT".PV_AGG1)
      wire#w3
      Move(in := "C#7_RD_RUN".PV_AG2, out1 => "C#8_RD_REPORT".PV_AGG2)
      wire#w4
      Move(in := "C#7_RD_RUN".PV_AG3, out1 => "C#8_RD_REPORT".PV_AGG3)
   END_RUNG
   RUNG wire#powerrail
      I_Contact( "C#2_WB"."SW_MAN/AUTO" )
      I_Contact( "PLC_BIT".RUN )
   END_RUNG wire#w1
   RUNG wire#w1
      I_Contact( "C#2_WB"."SW_MAN/AUTO" )
      I_Contact( "PLC_BIT".RUN )
      Contact( "C#1_RB"."DONG CUA" )
   END_RUNG wire#w2
   RUNG wire#w4
      Move(in := "C#7_RD_RUN".PVM_AG3, out1 => "C#8_RD_REPORT".PVM_AGG3)
   END_RUNG
   RUNG wire#w3
      Move(in := "C#7_RD_RUN".PVM_AG2, out1 => "C#8_RD_REPORT".PVM_AGG2)
   END_RUNG
   RUNG wire#w2
      Move(in := "C#7_RD_RUN".PVM_AG1, out1 => "C#8_RD_REPORT".PVM_AGG1)
   END_RUNG
   RUNG wire#w2
      Move(in := "C#7_RD_RUN".PV_AG4, out1 => "C#8_RD_REPORT".PV_AGG4)
      wire#w5
      Move(in := "C#7_RD_RUN".PV_AG5, out1 => "C#8_RD_REPORT".PV_AGG5)
   END_RUNG
   RUNG wire#w5
      Move(in := "C#7_RD_RUN".PVM_AG5, out1 => "C#8_RD_REPORT".PVM_AGG5)
   END_RUNG
   RUNG wire#w2
      Move(in := "C#7_RD_RUN".PVM_AG4, out1 => "C#8_RD_REPORT".PVM_AGG4)
   END_RUNG
   // the same network as SCL:
   #_w1 := ("PLC_BIT".AGG1_FU OR (NOT "C#2_WB"."SW_MAN/AUTO" AND NOT "PLC_BIT".RUN)) AND "C#1_RB"."XA W_AG1" AND NOT "P_XA PTG";   // rising edge of "C#1_RB"."XA W_AG1"
   "P_XA PTG" := "C#1_RB"."XA W_AG1";
   IF #_w1 OR (("PLC_BIT".AGG1_FU OR (NOT "C#2_WB"."SW_MAN/AUTO" AND NOT "PLC_BIT".RUN)) AND NOT "C#2_WB"."SW_MAN/AUTO" AND NOT "PLC_BIT".RUN AND "C#1_RB"."DONG CUA") THEN
       "C#8_RD_REPORT".PV_AGG1 := "C#7_RD_RUN".PV_AG1;
       "C#8_RD_REPORT".PV_AGG2 := "C#7_RD_RUN".PV_AG2;
       "C#8_RD_REPORT".PV_AGG3 := "C#7_RD_RUN".PV_AG3;
       "C#8_RD_REPORT".PVM_AGG3 := "C#7_RD_RUN".PVM_AG3;
       "C#8_RD_REPORT".PVM_AGG2 := "C#7_RD_RUN".PVM_AG2;
       "C#8_RD_REPORT".PVM_AGG1 := "C#7_RD_RUN".PVM_AG1;
       "C#8_RD_REPORT".PV_AGG4 := "C#7_RD_RUN".PV_AG4;
       "C#8_RD_REPORT".PV_AGG5 := "C#7_RD_RUN".PV_AG5;
       "C#8_RD_REPORT".PVM_AGG5 := "C#7_RD_RUN".PVM_AG5;
       "C#8_RD_REPORT".PVM_AGG4 := "C#7_RD_RUN".PVM_AG4;
   END_IF;
END_REGION

REGION Network 2: Lưu dữ liệu Xi măng
   RUNG wire#powerrail
      Contact( "PLC_BIT".WCE1_FU )
      wire#w1
      P_Contact(operand := "C#1_RB"."XA W_FD1", bit := "P_XA CEM1")
      wire#w2
      Move(in := "C#7_RD_RUN".PV_FD1, out1 => "C#8_RD_REPORT".PV_FD1)
   END_RUNG
   RUNG wire#powerrail
      I_Contact( "C#2_WB"."SW_MAN/AUTO" )
      I_Contact( "PLC_BIT".RUN )
   END_RUNG wire#w1
   RUNG wire#w1
      I_Contact( "C#2_WB"."SW_MAN/AUTO" )
      I_Contact( "PLC_BIT".RUN )
      Contact( "C#1_RB"."DONG CUA" )
   END_RUNG wire#w2
   RUNG wire#w2
      Move(in := "C#7_RD_RUN".PVM_FD1, out1 => "C#8_RD_REPORT".PVM_FD1)
   END_RUNG
   // the same network as SCL:
   #_w1 := ("PLC_BIT".WCE1_FU OR (NOT "C#2_WB"."SW_MAN/AUTO" AND NOT "PLC_BIT".RUN)) AND "C#1_RB"."XA W_FD1" AND NOT "P_XA CEM1";   // rising edge of "C#1_RB"."XA W_FD1"
   "P_XA CEM1" := "C#1_RB"."XA W_FD1";
   IF #_w1 OR (("PLC_BIT".WCE1_FU OR (NOT "C#2_WB"."SW_MAN/AUTO" AND NOT "PLC_BIT".RUN)) AND NOT "C#2_WB"."SW_MAN/AUTO" AND NOT "PLC_BIT".RUN AND "C#1_RB"."DONG CUA") THEN
       "C#8_RD_REPORT".PV_FD1 := "C#7_RD_RUN".PV_FD1;
       "C#8_RD_REPORT".PVM_FD1 := "C#7_RD_RUN".PVM_FD1;
   END_IF;
END_REGION

REGION Network 3: Lưu dữ liệu Nhựa
   RUNG wire#powerrail
      Contact( "PLC_BIT".WWA1_FU )
      wire#w1
      P_Contact(operand := "C#1_RB"."XA W_AP1", bit := "P_XA WAT1")
      wire#w2
      Move(in := "C#7_RD_RUN".PV_AP1, out1 => "C#8_RD_REPORT".PV_AP1)
   END_RUNG
   RUNG wire#powerrail
      I_Contact( "C#2_WB"."SW_MAN/AUTO" )
      I_Contact( "PLC_BIT".RUN )
   END_RUNG wire#w1
   RUNG wire#w1
      I_Contact( "C#2_WB"."SW_MAN/AUTO" )
      I_Contact( "PLC_BIT".RUN )
      Contact( "C#1_RB"."DONG CUA" )
   END_RUNG wire#w2
   RUNG wire#w2
      Move(in := "C#7_RD_RUN".PVM_AP1, out1 => "C#8_RD_REPORT".PVM_AP1)
   END_RUNG
   // the same network as SCL:
   #_w1 := ("PLC_BIT".WWA1_FU OR (NOT "C#2_WB"."SW_MAN/AUTO" AND NOT "PLC_BIT".RUN)) AND "C#1_RB"."XA W_AP1" AND NOT "P_XA WAT1";   // rising edge of "C#1_RB"."XA W_AP1"
   "P_XA WAT1" := "C#1_RB"."XA W_AP1";
   IF #_w1 OR (("PLC_BIT".WWA1_FU OR (NOT "C#2_WB"."SW_MAN/AUTO" AND NOT "PLC_BIT".RUN)) AND NOT "C#2_WB"."SW_MAN/AUTO" AND NOT "PLC_BIT".RUN AND "C#1_RB"."DONG CUA") THEN
       "C#8_RD_REPORT".PV_AP1 := "C#7_RD_RUN".PV_AP1;
       "C#8_RD_REPORT".PVM_AP1 := "C#7_RD_RUN".PVM_AP1;
   END_IF;
END_REGION

REGION Network 4: Lưu dữ liệu Phụ gia SBS
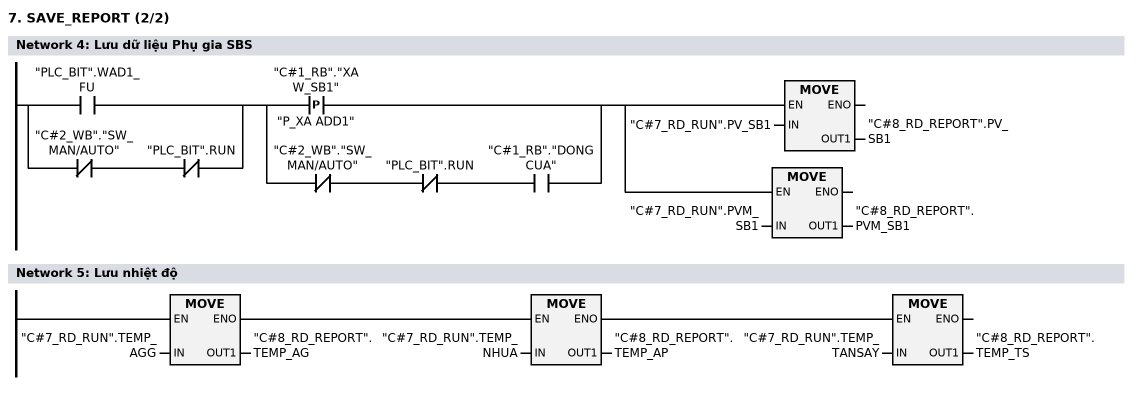
   RUNG wire#powerrail
      Contact( "PLC_BIT".WAD1_FU )
      wire#w1
      P_Contact(operand := "C#1_RB"."XA W_SB1", bit := "P_XA ADD1")
      wire#w2
      Move(in := "C#7_RD_RUN".PV_SB1, out1 => "C#8_RD_REPORT".PV_SB1)
   END_RUNG
   RUNG wire#powerrail
      I_Contact( "C#2_WB"."SW_MAN/AUTO" )
      I_Contact( "PLC_BIT".RUN )
   END_RUNG wire#w1
   RUNG wire#w1
      I_Contact( "C#2_WB"."SW_MAN/AUTO" )
      I_Contact( "PLC_BIT".RUN )
      Contact( "C#1_RB"."DONG CUA" )
   END_RUNG wire#w2
   RUNG wire#w2
      Move(in := "C#7_RD_RUN".PVM_SB1, out1 => "C#8_RD_REPORT".PVM_SB1)
   END_RUNG
   // the same network as SCL:
   #_w1 := ("PLC_BIT".WAD1_FU OR (NOT "C#2_WB"."SW_MAN/AUTO" AND NOT "PLC_BIT".RUN)) AND "C#1_RB"."XA W_SB1" AND NOT "P_XA ADD1";   // rising edge of "C#1_RB"."XA W_SB1"
   "P_XA ADD1" := "C#1_RB"."XA W_SB1";
   IF #_w1 OR (("PLC_BIT".WAD1_FU OR (NOT "C#2_WB"."SW_MAN/AUTO" AND NOT "PLC_BIT".RUN)) AND NOT "C#2_WB"."SW_MAN/AUTO" AND NOT "PLC_BIT".RUN AND "C#1_RB"."DONG CUA") THEN
       "C#8_RD_REPORT".PV_SB1 := "C#7_RD_RUN".PV_SB1;
       "C#8_RD_REPORT".PVM_SB1 := "C#7_RD_RUN".PVM_SB1;
   END_IF;
END_REGION

REGION Network 5: Lưu nhiệt độ
   RUNG wire#powerrail
      Move(in := "C#7_RD_RUN".TEMP_AGG, out1 => "C#8_RD_REPORT".TEMP_AG)
      Move(in := "C#7_RD_RUN".TEMP_NHUA, out1 => "C#8_RD_REPORT".TEMP_AP)
      Move(in := "C#7_RD_RUN".TEMP_TANSAY, out1 => "C#8_RD_REPORT".TEMP_TS)
   END_RUNG
   // the same network as SCL:
   "C#8_RD_REPORT".TEMP_AG := "C#7_RD_RUN".TEMP_AGG;
   "C#8_RD_REPORT".TEMP_AP := "C#7_RD_RUN".TEMP_NHUA;
   "C#8_RD_REPORT".TEMP_TS := "C#7_RD_RUN".TEMP_TANSAY;
END_REGION
END_FUNCTION

ORGANIZATION_BLOCK "Main"   // OB123, LAD, ProgramCycle
TITLE = "Main Program Sweep (Cycle)"
{ S7_Optimized_Access := 'TRUE' }
VERSION : 0.1
// stored: AutoNumber true, CodeModifiedDate 2026-01-15T16:25:55.6274482Z, CompileDate 2026-01-15T16:25:55.6406611Z, ConstantName OB_Main, CreationDate 2026-01-15T16:14:49.4586784Z, EventClass Program cycle, HandleErrorsWithinBlock false, InterfaceModifiedDate 2026-01-15T16:25:47.5430699Z, IsConsistent true, IsIECCheckEnabled false, IsKnowHowProtected false, IsWriteProtected false, ModifiedDate 2026-01-15T16:25:55.6274482Z, ParameterModified 2008-07-21T16:55:08.419547Z, PLCSimAdvancedSupport false, PriorityNumber 1, ProcessImagePartNumber 65535, SetENOAutomatically False, StructureModified 2008-07-21T16:55:08.419547Z
   VAR_INPUT
      Initial_Call : Bool;   // Initial call of this OB
      Remanence : Bool;   // =True, if remanent data are available
   END_VAR
BEGIN
END_ORGANIZATION_BLOCK

FUNCTION_BLOCK "10.TIMER_CLOCK"   // FB10, LAD
{ S7_Optimized_Access := 'TRUE' }
VERSION : 0.1
// stored: AutoNumber false, CodeModifiedDate 2025-08-27T17:13:37.9521369Z, CompileDate 2026-01-15T16:25:53.3373579Z, CreationDate 2026-01-15T16:22:49.8270549Z, DownloadWithoutReinit false, HandleErrorsWithinBlock false, InterfaceModifiedDate 2023-08-14T08:08:19.3737097Z, IsConsistent true, IsIECCheckEnabled false, IsKnowHowProtected false, IsRetainMemResEnabled false, IsWriteProtected false, LibraryConformanceStatus The object is library-conformant., MemoryReserve 100, ModifiedDate 2025-08-27T17:13:37.9521369Z, ParameterModified 2022-05-24T16:04:05.0982286Z, PLCSimAdvancedSupport false, SetENOAutomatically False, StructureModified 2023-08-14T08:08:19.3737097Z, UDAEnableTagReadback false
   VAR_INPUT
      ON : Bool;
      CLOCK_1S : Bool;
      T_ON : Real;
      T_OFF : Real;
   END_VAR
   VAR_OUTPUT
      OUT : Bool;
   END_VAR
   VAR RETAIN
      TON : Real;
      TOFF : Real;
   END_VAR
   VAR
      CLK1 : Bool;
   END_VAR
   VAR_TEMP   // added for the SCL form of the ladder/FBD networks
      _w1 : Bool;
   END_VAR
BEGIN

REGION Network 1
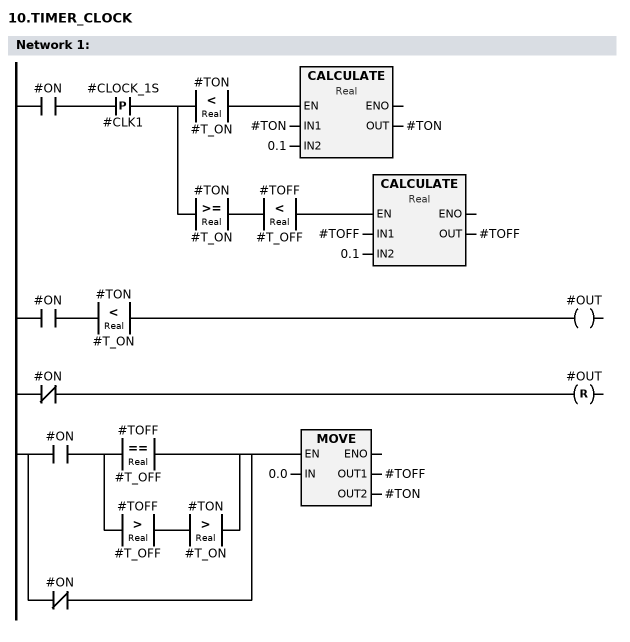
   RUNG wire#powerrail
      Contact( #ON )
      P_Contact(operand := #CLOCK_1S, bit := #CLK1)
      wire#w1
      { S7_Templates := "SrcType := Real" } LT_Contact(in1 := #TON, in2 := #T_ON)
      { S7_Templates := "SrcType := Real"; S7_Expression := "IN1+IN2" } Calculate(in1 := #TON, in2 := 0.1, out => #TON)
   END_RUNG
   RUNG wire#w1
      { S7_Templates := "SrcType := Real" } GE_Contact(in1 := #TON, in2 := #T_ON)
      { S7_Templates := "SrcType := Real" } LT_Contact(in1 := #TOFF, in2 := #T_OFF)
      { S7_Templates := "SrcType := Real"; S7_Expression := "IN1+IN2" } Calculate(in1 := #TOFF, in2 := 0.1, out => #TOFF)
   END_RUNG
   RUNG wire#powerrail
      Contact( #ON )
      { S7_Templates := "SrcType := Real" } LT_Contact(in1 := #TON, in2 := #T_ON)
      Coil( #OUT )
   END_RUNG
   RUNG wire#powerrail
      I_Contact( #ON )
      R_Coil( #OUT )
   END_RUNG
   RUNG wire#powerrail
      Contact( #ON )
      wire#w2
      { S7_Templates := "SrcType := Real" } EQ_Contact(in1 := #TOFF, in2 := #T_OFF)
      wire#w3
      Move(in := 0.0, out1 => #TOFF, out2 => #TON)
   END_RUNG
   RUNG wire#w2
      { S7_Templates := "SrcType := Real" } GT_Contact(in1 := #TOFF, in2 := #T_OFF)
      { S7_Templates := "SrcType := Real" } GT_Contact(in1 := #TON, in2 := #T_ON)
   END_RUNG wire#w3
   RUNG wire#powerrail
      I_Contact( #ON )
   END_RUNG wire#w3
   // the same network as SCL:
   #_w1 := #ON AND #CLOCK_1S AND NOT #CLK1;   // rising edge of #CLOCK_1S
   #CLK1 := #CLOCK_1S;
   IF #_w1 AND (#TON < #T_ON) THEN #TON := #TON+0.1; END_IF;
   IF #_w1 AND (#TON >= #T_ON) AND (#TOFF < #T_OFF) THEN #TOFF := #TOFF+0.1; END_IF;
   #OUT := #ON AND (#TON < #T_ON);
   IF NOT #ON THEN #OUT := FALSE; END_IF;
   IF (#ON AND ((#TOFF = #T_OFF) OR ((#TOFF > #T_OFF) AND (#TON > #T_ON)))) OR NOT #ON THEN
       #TOFF := 0.0;
       #TON := 0.0;
   END_IF;
END_REGION
END_FUNCTION_BLOCK

FUNCTION_BLOCK "11. LOGIC CAN"   // FB11, LAD
{ S7_Optimized_Access := 'TRUE' }
VERSION : 0.1
// stored: AutoNumber true, CodeModifiedDate 2025-08-27T17:14:05.4937984Z, CompileDate 2026-01-15T16:25:55.4686185Z, CreationDate 2026-01-15T16:22:49.8270549Z, DownloadWithoutReinit false, HandleErrorsWithinBlock false, InterfaceModifiedDate 2023-12-21T19:23:23.4270206Z, IsConsistent true, IsIECCheckEnabled false, IsKnowHowProtected false, IsRetainMemResEnabled false, IsWriteProtected false, LibraryConformanceStatus The object is library-conformant., MemoryReserve 100, ModifiedDate 2025-08-27T17:14:05.4937984Z, ParameterModified 2023-12-21T19:23:23.4270206Z, PLCSimAdvancedSupport false, SetENOAutomatically False, StructureModified 2023-12-21T19:23:23.4270206Z, UDAEnableTagReadback false
   VAR_INPUT
      LOGIC_1 : Real;
      LOGIC_2 : Real;
      LOGIC_3 : Real;
      "THC_1.1" : Bool;
      "THC_1.2" : Bool;
      "THC_2.1" : Bool;
      "THC_2.2" : Bool;
      "THC_3.1" : Bool;
      "THC_3.2" : Bool;
      "THC_4.1" : Bool;
      "THC_4.2" : Bool;
      "THC_5.1" : Bool;
      "THC_5.2" : Bool;
      "THC_6.1" : Bool;
      "THC_6.2" : Bool;
   END_VAR
   VAR_OUTPUT
      "OUT_LGOIC_1.1" : Bool;
      "OUT_LGOIC_1.2" : Bool;
      "OUT_LGOIC_2.1" : Bool;
      "OUT_LGOIC_2.2" : Bool;
      "OUT_LGOIC_3.1" : Bool;
      "OUT_LGOIC_3.2" : Bool;
      "OUT_LGOIC_4.1" : Bool;
      "OUT_LGOIC_4.2" : Bool;
      "OUT_LGOIC_5.1" : Bool;
      "OUT_LGOIC_5.2" : Bool;
      "OUT_LGOIC_6.1" : Bool;
      "OUT_LGOIC_6.2" : Bool;
   END_VAR
BEGIN

REGION Network 1: OUT1
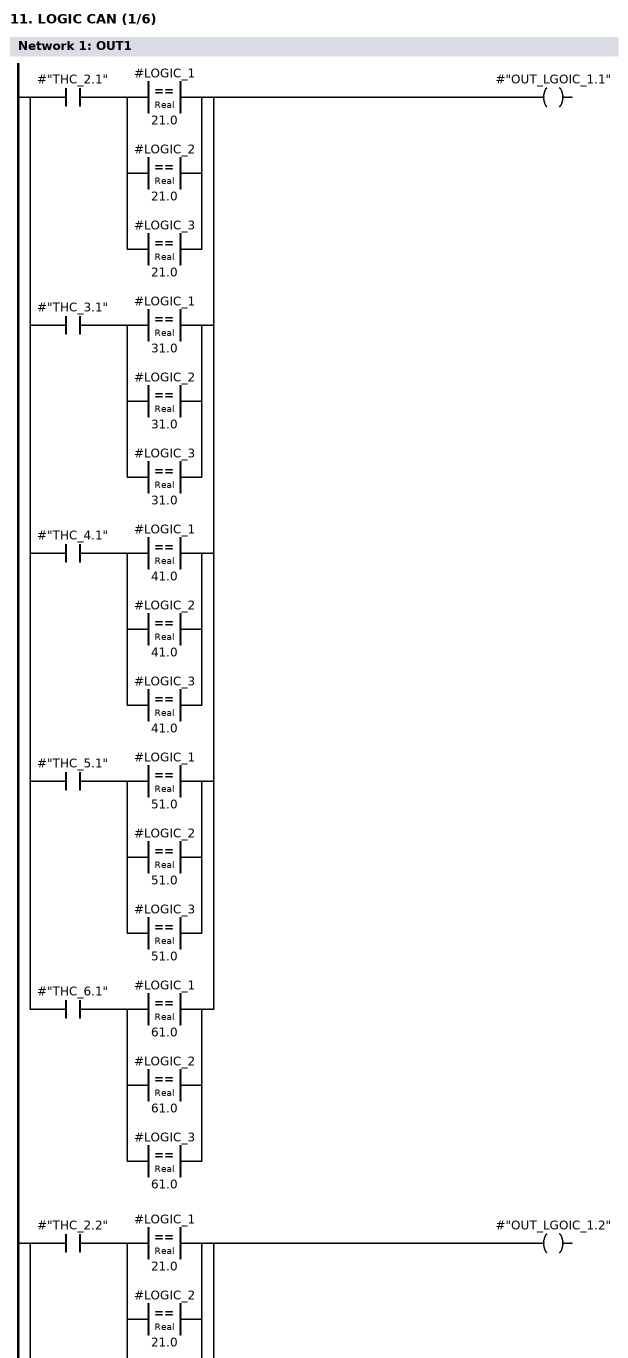
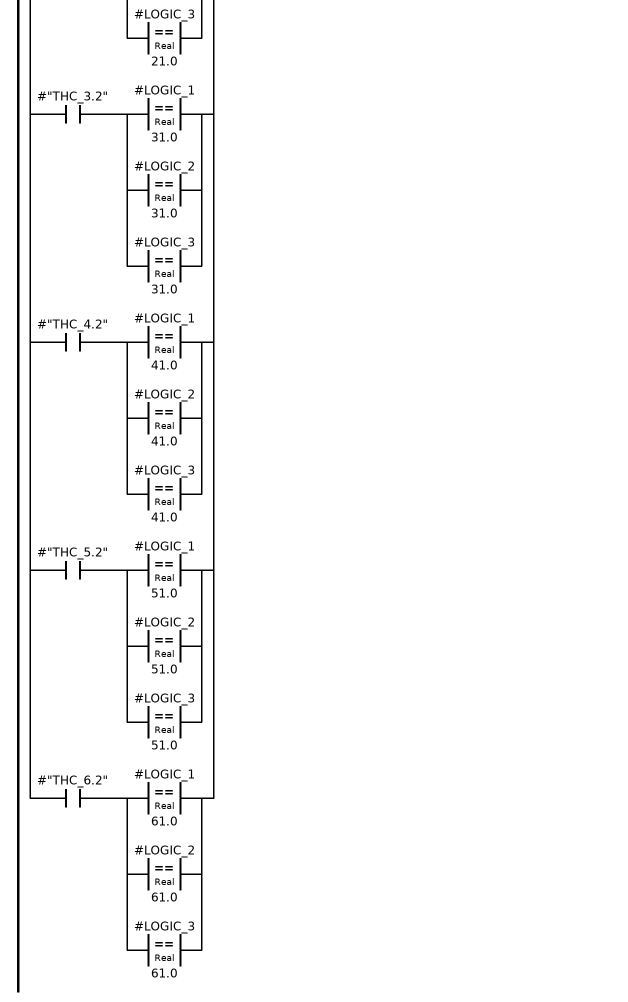
   RUNG wire#powerrail
      Contact( #"THC_2.1" )
      wire#w1
      { S7_Templates := "SrcType := Real" } EQ_Contact(in1 := #LOGIC_1, in2 := 21.0)
      wire#w2
      Coil( #"OUT_LGOIC_1.1" )
   END_RUNG
   RUNG wire#w1
      { S7_Templates := "SrcType := Real" } EQ_Contact(in1 := #LOGIC_2, in2 := 21.0)
   END_RUNG wire#w2
   RUNG wire#w1
      { S7_Templates := "SrcType := Real" } EQ_Contact(in1 := #LOGIC_3, in2 := 21.0)
   END_RUNG wire#w2
   RUNG wire#powerrail
      Contact( #"THC_3.1" )
      wire#w3
      { S7_Templates := "SrcType := Real" } EQ_Contact(in1 := #LOGIC_1, in2 := 31.0)
   END_RUNG wire#w2
   RUNG wire#w3
      { S7_Templates := "SrcType := Real" } EQ_Contact(in1 := #LOGIC_2, in2 := 31.0)
   END_RUNG wire#w2
   RUNG wire#w3
      { S7_Templates := "SrcType := Real" } EQ_Contact(in1 := #LOGIC_3, in2 := 31.0)
   END_RUNG wire#w2
   RUNG wire#powerrail
      Contact( #"THC_4.1" )
      wire#w4
      { S7_Templates := "SrcType := Real" } EQ_Contact(in1 := #LOGIC_1, in2 := 41.0)
   END_RUNG wire#w2
   RUNG wire#w4
      { S7_Templates := "SrcType := Real" } EQ_Contact(in1 := #LOGIC_2, in2 := 41.0)
   END_RUNG wire#w2
   RUNG wire#w4
      { S7_Templates := "SrcType := Real" } EQ_Contact(in1 := #LOGIC_3, in2 := 41.0)
   END_RUNG wire#w2
   RUNG wire#powerrail
      Contact( #"THC_5.1" )
      wire#w5
      { S7_Templates := "SrcType := Real" } EQ_Contact(in1 := #LOGIC_1, in2 := 51.0)
   END_RUNG wire#w2
   RUNG wire#w5
      { S7_Templates := "SrcType := Real" } EQ_Contact(in1 := #LOGIC_2, in2 := 51.0)
   END_RUNG wire#w2
   RUNG wire#w5
      { S7_Templates := "SrcType := Real" } EQ_Contact(in1 := #LOGIC_3, in2 := 51.0)
   END_RUNG wire#w2
   RUNG wire#powerrail
      Contact( #"THC_6.1" )
      wire#w6
      { S7_Templates := "SrcType := Real" } EQ_Contact(in1 := #LOGIC_1, in2 := 61.0)
   END_RUNG wire#w2
   RUNG wire#w6
      { S7_Templates := "SrcType := Real" } EQ_Contact(in1 := #LOGIC_2, in2 := 61.0)
   END_RUNG wire#w2
   RUNG wire#w6
      { S7_Templates := "SrcType := Real" } EQ_Contact(in1 := #LOGIC_3, in2 := 61.0)
   END_RUNG wire#w2
   RUNG wire#powerrail
      Contact( #"THC_2.2" )
      wire#w7
      { S7_Templates := "SrcType := Real" } EQ_Contact(in1 := #LOGIC_1, in2 := 21.0)
      wire#w8
      Coil( #"OUT_LGOIC_1.2" )
   END_RUNG
   RUNG wire#w7
      { S7_Templates := "SrcType := Real" } EQ_Contact(in1 := #LOGIC_2, in2 := 21.0)
   END_RUNG wire#w8
   RUNG wire#w7
      { S7_Templates := "SrcType := Real" } EQ_Contact(in1 := #LOGIC_3, in2 := 21.0)
   END_RUNG wire#w8
   RUNG wire#powerrail
      Contact( #"THC_3.2" )
      wire#w9
      { S7_Templates := "SrcType := Real" } EQ_Contact(in1 := #LOGIC_1, in2 := 31.0)
   END_RUNG wire#w8
   RUNG wire#w9
      { S7_Templates := "SrcType := Real" } EQ_Contact(in1 := #LOGIC_2, in2 := 31.0)
   END_RUNG wire#w8
   RUNG wire#w9
      { S7_Templates := "SrcType := Real" } EQ_Contact(in1 := #LOGIC_3, in2 := 31.0)
   END_RUNG wire#w8
   RUNG wire#powerrail
      Contact( #"THC_4.2" )
      wire#w10
      { S7_Templates := "SrcType := Real" } EQ_Contact(in1 := #LOGIC_1, in2 := 41.0)
   END_RUNG wire#w8
   RUNG wire#w10
      { S7_Templates := "SrcType := Real" } EQ_Contact(in1 := #LOGIC_2, in2 := 41.0)
   END_RUNG wire#w8
   RUNG wire#w10
      { S7_Templates := "SrcType := Real" } EQ_Contact(in1 := #LOGIC_3, in2 := 41.0)
   END_RUNG wire#w8
   RUNG wire#powerrail
      Contact( #"THC_5.2" )
      wire#w11
      { S7_Templates := "SrcType := Real" } EQ_Contact(in1 := #LOGIC_1, in2 := 51.0)
   END_RUNG wire#w8
   RUNG wire#w11
      { S7_Templates := "SrcType := Real" } EQ_Contact(in1 := #LOGIC_2, in2 := 51.0)
   END_RUNG wire#w8
   RUNG wire#w11
      { S7_Templates := "SrcType := Real" } EQ_Contact(in1 := #LOGIC_3, in2 := 51.0)
   END_RUNG wire#w8
   RUNG wire#powerrail
      Contact( #"THC_6.2" )
      wire#w12
      { S7_Templates := "SrcType := Real" } EQ_Contact(in1 := #LOGIC_1, in2 := 61.0)
   END_RUNG wire#w8
   RUNG wire#w12
      { S7_Templates := "SrcType := Real" } EQ_Contact(in1 := #LOGIC_2, in2 := 61.0)
   END_RUNG wire#w8
   RUNG wire#w12
      { S7_Templates := "SrcType := Real" } EQ_Contact(in1 := #LOGIC_3, in2 := 61.0)
   END_RUNG wire#w8
   // the same network as SCL:
   #"OUT_LGOIC_1.1" := (#"THC_2.1" AND ((#LOGIC_1 = 21.0) OR (#LOGIC_2 = 21.0) OR (#LOGIC_3 = 21.0))) OR (#"THC_3.1" AND ((#LOGIC_1 = 31.0) OR (#LOGIC_2 = 31.0) OR (#LOGIC_3 = 31.0))) OR (#"THC_4.1" AND ((#LOGIC_1 = 41.0) OR (#LOGIC_2 = 41.0) OR (#LOGIC_3 = 41.0))) OR (#"THC_5.1" AND ((#LOGIC_1 = 51.0) OR (#LOGIC_2 = 51.0) OR (#LOGIC_3 = 51.0))) OR (#"THC_6.1" AND ((#LOGIC_1 = 61.0) OR (#LOGIC_2 = 61.0) OR (#LOGIC_3 = 61.0)));
   #"OUT_LGOIC_1.2" := (#"THC_2.2" AND ((#LOGIC_1 = 21.0) OR (#LOGIC_2 = 21.0) OR (#LOGIC_3 = 21.0))) OR (#"THC_3.2" AND ((#LOGIC_1 = 31.0) OR (#LOGIC_2 = 31.0) OR (#LOGIC_3 = 31.0))) OR (#"THC_4.2" AND ((#LOGIC_1 = 41.0) OR (#LOGIC_2 = 41.0) OR (#LOGIC_3 = 41.0))) OR (#"THC_5.2" AND ((#LOGIC_1 = 51.0) OR (#LOGIC_2 = 51.0) OR (#LOGIC_3 = 51.0))) OR (#"THC_6.2" AND ((#LOGIC_1 = 61.0) OR (#LOGIC_2 = 61.0) OR (#LOGIC_3 = 61.0)));
END_REGION

REGION Network 2: OUT2
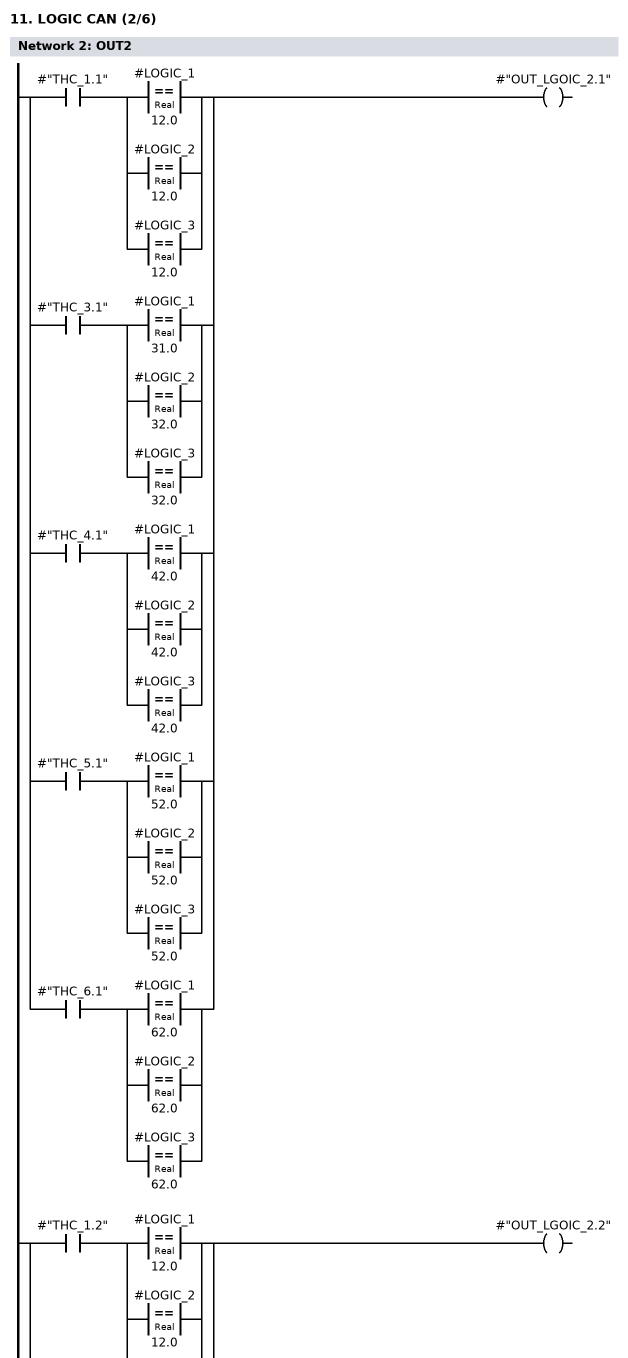
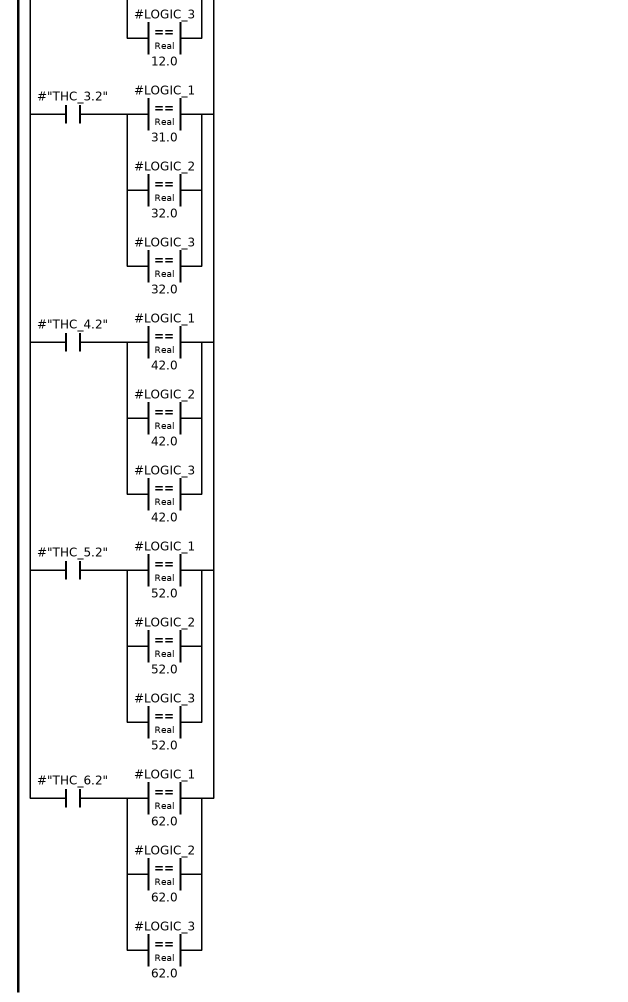
   RUNG wire#powerrail
      Contact( #"THC_1.1" )
      wire#w1
      { S7_Templates := "SrcType := Real" } EQ_Contact(in1 := #LOGIC_1, in2 := 12.0)
      wire#w2
      Coil( #"OUT_LGOIC_2.1" )
   END_RUNG
   RUNG wire#w1
      { S7_Templates := "SrcType := Real" } EQ_Contact(in1 := #LOGIC_2, in2 := 12.0)
   END_RUNG wire#w2
   RUNG wire#w1
      { S7_Templates := "SrcType := Real" } EQ_Contact(in1 := #LOGIC_3, in2 := 12.0)
   END_RUNG wire#w2
   RUNG wire#powerrail
      Contact( #"THC_3.1" )
      wire#w3
      { S7_Templates := "SrcType := Real" } EQ_Contact(in1 := #LOGIC_1, in2 := 31.0)
   END_RUNG wire#w2
   RUNG wire#w3
      { S7_Templates := "SrcType := Real" } EQ_Contact(in1 := #LOGIC_2, in2 := 32.0)
   END_RUNG wire#w2
   RUNG wire#w3
      { S7_Templates := "SrcType := Real" } EQ_Contact(in1 := #LOGIC_3, in2 := 32.0)
   END_RUNG wire#w2
   RUNG wire#powerrail
      Contact( #"THC_4.1" )
      wire#w4
      { S7_Templates := "SrcType := Real" } EQ_Contact(in1 := #LOGIC_1, in2 := 42.0)
   END_RUNG wire#w2
   RUNG wire#w4
      { S7_Templates := "SrcType := Real" } EQ_Contact(in1 := #LOGIC_2, in2 := 42.0)
   END_RUNG wire#w2
   RUNG wire#w4
      { S7_Templates := "SrcType := Real" } EQ_Contact(in1 := #LOGIC_3, in2 := 42.0)
   END_RUNG wire#w2
   RUNG wire#powerrail
      Contact( #"THC_5.1" )
      wire#w5
      { S7_Templates := "SrcType := Real" } EQ_Contact(in1 := #LOGIC_1, in2 := 52.0)
   END_RUNG wire#w2
   RUNG wire#w5
      { S7_Templates := "SrcType := Real" } EQ_Contact(in1 := #LOGIC_2, in2 := 52.0)
   END_RUNG wire#w2
   RUNG wire#w5
      { S7_Templates := "SrcType := Real" } EQ_Contact(in1 := #LOGIC_3, in2 := 52.0)
   END_RUNG wire#w2
   RUNG wire#powerrail
      Contact( #"THC_6.1" )
      wire#w6
      { S7_Templates := "SrcType := Real" } EQ_Contact(in1 := #LOGIC_1, in2 := 62.0)
   END_RUNG wire#w2
   RUNG wire#w6
      { S7_Templates := "SrcType := Real" } EQ_Contact(in1 := #LOGIC_2, in2 := 62.0)
   END_RUNG wire#w2
   RUNG wire#w6
      { S7_Templates := "SrcType := Real" } EQ_Contact(in1 := #LOGIC_3, in2 := 62.0)
   END_RUNG wire#w2
   RUNG wire#powerrail
      Contact( #"THC_1.2" )
      wire#w7
      { S7_Templates := "SrcType := Real" } EQ_Contact(in1 := #LOGIC_1, in2 := 12.0)
      wire#w8
      Coil( #"OUT_LGOIC_2.2" )
   END_RUNG
   RUNG wire#w7
      { S7_Templates := "SrcType := Real" } EQ_Contact(in1 := #LOGIC_2, in2 := 12.0)
   END_RUNG wire#w8
   RUNG wire#w7
      { S7_Templates := "SrcType := Real" } EQ_Contact(in1 := #LOGIC_3, in2 := 12.0)
   END_RUNG wire#w8
   RUNG wire#powerrail
      Contact( #"THC_3.2" )
      wire#w9
      { S7_Templates := "SrcType := Real" } EQ_Contact(in1 := #LOGIC_1, in2 := 31.0)
   END_RUNG wire#w8
   RUNG wire#w9
      { S7_Templates := "SrcType := Real" } EQ_Contact(in1 := #LOGIC_2, in2 := 32.0)
   END_RUNG wire#w8
   RUNG wire#w9
      { S7_Templates := "SrcType := Real" } EQ_Contact(in1 := #LOGIC_3, in2 := 32.0)
   END_RUNG wire#w8
   RUNG wire#powerrail
      Contact( #"THC_4.2" )
      wire#w10
      { S7_Templates := "SrcType := Real" } EQ_Contact(in1 := #LOGIC_1, in2 := 42.0)
   END_RUNG wire#w8
   RUNG wire#w10
      { S7_Templates := "SrcType := Real" } EQ_Contact(in1 := #LOGIC_2, in2 := 42.0)
   END_RUNG wire#w8
   RUNG wire#w10
      { S7_Templates := "SrcType := Real" } EQ_Contact(in1 := #LOGIC_3, in2 := 42.0)
   END_RUNG wire#w8
   RUNG wire#powerrail
      Contact( #"THC_5.2" )
      wire#w11
      { S7_Templates := "SrcType := Real" } EQ_Contact(in1 := #LOGIC_1, in2 := 52.0)
   END_RUNG wire#w8
   RUNG wire#w11
      { S7_Templates := "SrcType := Real" } EQ_Contact(in1 := #LOGIC_2, in2 := 52.0)
   END_RUNG wire#w8
   RUNG wire#w11
      { S7_Templates := "SrcType := Real" } EQ_Contact(in1 := #LOGIC_3, in2 := 52.0)
   END_RUNG wire#w8
   RUNG wire#powerrail
      Contact( #"THC_6.2" )
      wire#w12
      { S7_Templates := "SrcType := Real" } EQ_Contact(in1 := #LOGIC_1, in2 := 62.0)
   END_RUNG wire#w8
   RUNG wire#w12
      { S7_Templates := "SrcType := Real" } EQ_Contact(in1 := #LOGIC_2, in2 := 62.0)
   END_RUNG wire#w8
   RUNG wire#w12
      { S7_Templates := "SrcType := Real" } EQ_Contact(in1 := #LOGIC_3, in2 := 62.0)
   END_RUNG wire#w8
   // the same network as SCL:
   #"OUT_LGOIC_2.1" := (#"THC_1.1" AND ((#LOGIC_1 = 12.0) OR (#LOGIC_2 = 12.0) OR (#LOGIC_3 = 12.0))) OR (#"THC_3.1" AND ((#LOGIC_1 = 31.0) OR (#LOGIC_2 = 32.0) OR (#LOGIC_3 = 32.0))) OR (#"THC_4.1" AND ((#LOGIC_1 = 42.0) OR (#LOGIC_2 = 42.0) OR (#LOGIC_3 = 42.0))) OR (#"THC_5.1" AND ((#LOGIC_1 = 52.0) OR (#LOGIC_2 = 52.0) OR (#LOGIC_3 = 52.0))) OR (#"THC_6.1" AND ((#LOGIC_1 = 62.0) OR (#LOGIC_2 = 62.0) OR (#LOGIC_3 = 62.0)));
   #"OUT_LGOIC_2.2" := (#"THC_1.2" AND ((#LOGIC_1 = 12.0) OR (#LOGIC_2 = 12.0) OR (#LOGIC_3 = 12.0))) OR (#"THC_3.2" AND ((#LOGIC_1 = 31.0) OR (#LOGIC_2 = 32.0) OR (#LOGIC_3 = 32.0))) OR (#"THC_4.2" AND ((#LOGIC_1 = 42.0) OR (#LOGIC_2 = 42.0) OR (#LOGIC_3 = 42.0))) OR (#"THC_5.2" AND ((#LOGIC_1 = 52.0) OR (#LOGIC_2 = 52.0) OR (#LOGIC_3 = 52.0))) OR (#"THC_6.2" AND ((#LOGIC_1 = 62.0) OR (#LOGIC_2 = 62.0) OR (#LOGIC_3 = 62.0)));
END_REGION

REGION Network 3: OUT3
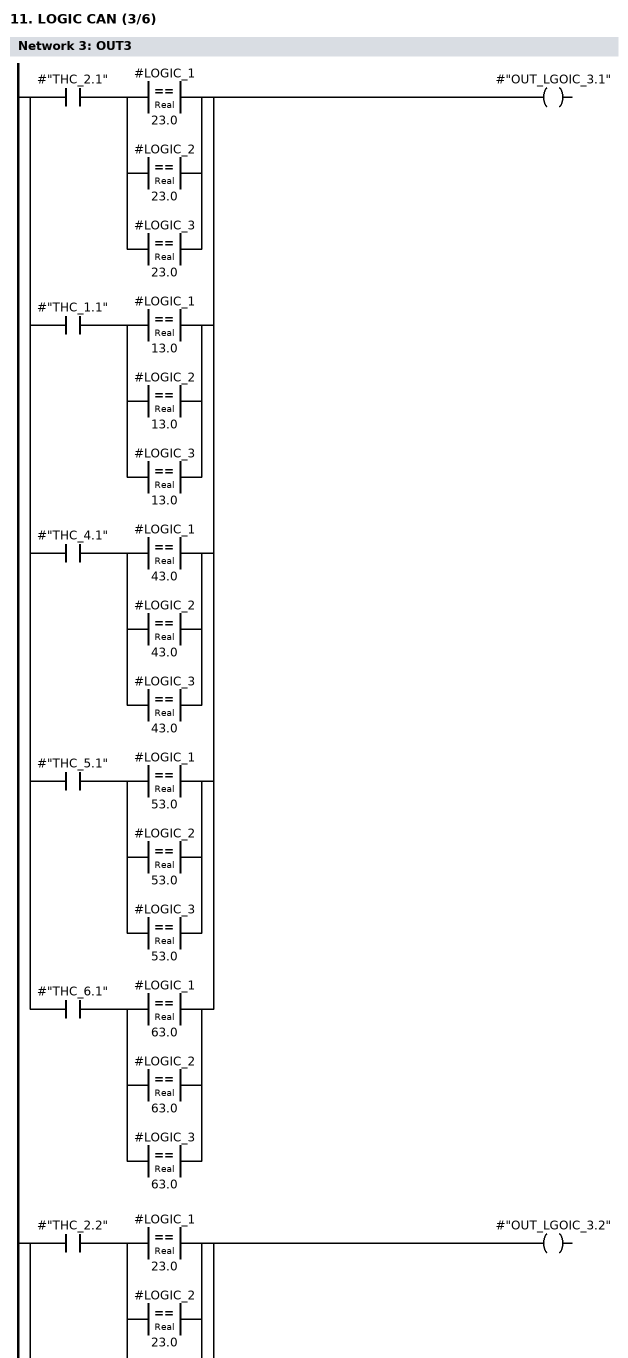
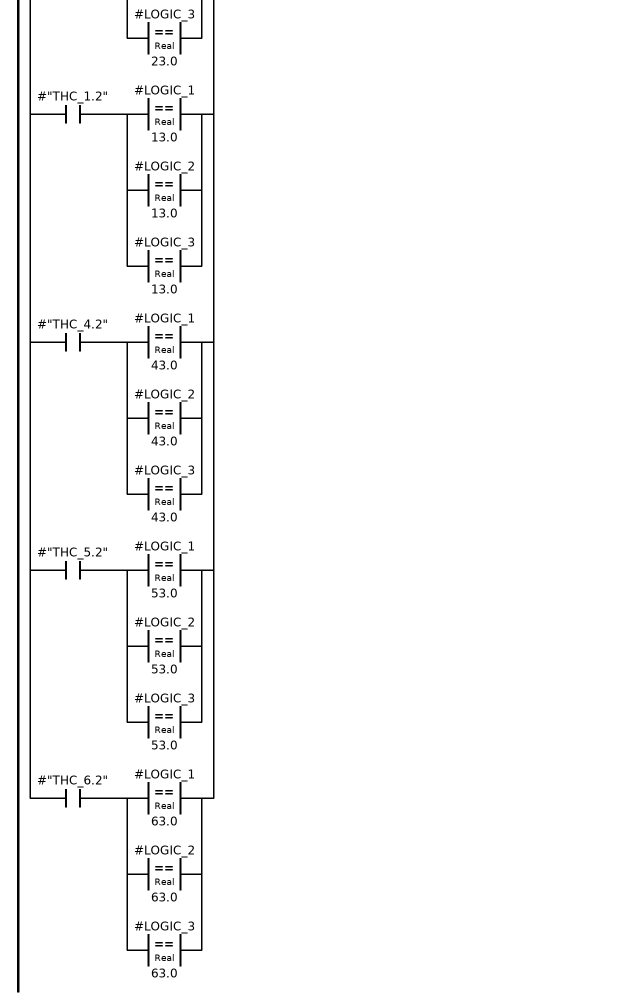
   RUNG wire#powerrail
      Contact( #"THC_2.1" )
      wire#w1
      { S7_Templates := "SrcType := Real" } EQ_Contact(in1 := #LOGIC_1, in2 := 23.0)
      wire#w2
      Coil( #"OUT_LGOIC_3.1" )
   END_RUNG
   RUNG wire#w1
      { S7_Templates := "SrcType := Real" } EQ_Contact(in1 := #LOGIC_2, in2 := 23.0)
   END_RUNG wire#w2
   RUNG wire#w1
      { S7_Templates := "SrcType := Real" } EQ_Contact(in1 := #LOGIC_3, in2 := 23.0)
   END_RUNG wire#w2
   RUNG wire#powerrail
      Contact( #"THC_1.1" )
      wire#w3
      { S7_Templates := "SrcType := Real" } EQ_Contact(in1 := #LOGIC_1, in2 := 13.0)
   END_RUNG wire#w2
   RUNG wire#w3
      { S7_Templates := "SrcType := Real" } EQ_Contact(in1 := #LOGIC_2, in2 := 13.0)
   END_RUNG wire#w2
   RUNG wire#w3
      { S7_Templates := "SrcType := Real" } EQ_Contact(in1 := #LOGIC_3, in2 := 13.0)
   END_RUNG wire#w2
   RUNG wire#powerrail
      Contact( #"THC_4.1" )
      wire#w4
      { S7_Templates := "SrcType := Real" } EQ_Contact(in1 := #LOGIC_1, in2 := 43.0)
   END_RUNG wire#w2
   RUNG wire#w4
      { S7_Templates := "SrcType := Real" } EQ_Contact(in1 := #LOGIC_2, in2 := 43.0)
   END_RUNG wire#w2
   RUNG wire#w4
      { S7_Templates := "SrcType := Real" } EQ_Contact(in1 := #LOGIC_3, in2 := 43.0)
   END_RUNG wire#w2
   RUNG wire#powerrail
      Contact( #"THC_5.1" )
      wire#w5
      { S7_Templates := "SrcType := Real" } EQ_Contact(in1 := #LOGIC_1, in2 := 53.0)
   END_RUNG wire#w2
   RUNG wire#w5
      { S7_Templates := "SrcType := Real" } EQ_Contact(in1 := #LOGIC_2, in2 := 53.0)
   END_RUNG wire#w2
   RUNG wire#w5
      { S7_Templates := "SrcType := Real" } EQ_Contact(in1 := #LOGIC_3, in2 := 53.0)
   END_RUNG wire#w2
   RUNG wire#powerrail
      Contact( #"THC_6.1" )
      wire#w6
      { S7_Templates := "SrcType := Real" } EQ_Contact(in1 := #LOGIC_1, in2 := 63.0)
   END_RUNG wire#w2
   RUNG wire#w6
      { S7_Templates := "SrcType := Real" } EQ_Contact(in1 := #LOGIC_2, in2 := 63.0)
   END_RUNG wire#w2
   RUNG wire#w6
      { S7_Templates := "SrcType := Real" } EQ_Contact(in1 := #LOGIC_3, in2 := 63.0)
   END_RUNG wire#w2
   RUNG wire#powerrail
      Contact( #"THC_2.2" )
      wire#w7
      { S7_Templates := "SrcType := Real" } EQ_Contact(in1 := #LOGIC_1, in2 := 23.0)
      wire#w8
      Coil( #"OUT_LGOIC_3.2" )
   END_RUNG
   RUNG wire#w7
      { S7_Templates := "SrcType := Real" } EQ_Contact(in1 := #LOGIC_2, in2 := 23.0)
   END_RUNG wire#w8
   RUNG wire#w7
      { S7_Templates := "SrcType := Real" } EQ_Contact(in1 := #LOGIC_3, in2 := 23.0)
   END_RUNG wire#w8
   RUNG wire#powerrail
      Contact( #"THC_1.2" )
      wire#w9
      { S7_Templates := "SrcType := Real" } EQ_Contact(in1 := #LOGIC_1, in2 := 13.0)
   END_RUNG wire#w8
   RUNG wire#w9
      { S7_Templates := "SrcType := Real" } EQ_Contact(in1 := #LOGIC_2, in2 := 13.0)
   END_RUNG wire#w8
   RUNG wire#w9
      { S7_Templates := "SrcType := Real" } EQ_Contact(in1 := #LOGIC_3, in2 := 13.0)
   END_RUNG wire#w8
   RUNG wire#powerrail
      Contact( #"THC_4.2" )
      wire#w10
      { S7_Templates := "SrcType := Real" } EQ_Contact(in1 := #LOGIC_1, in2 := 43.0)
   END_RUNG wire#w8
   RUNG wire#w10
      { S7_Templates := "SrcType := Real" } EQ_Contact(in1 := #LOGIC_2, in2 := 43.0)
   END_RUNG wire#w8
   RUNG wire#w10
      { S7_Templates := "SrcType := Real" } EQ_Contact(in1 := #LOGIC_3, in2 := 43.0)
   END_RUNG wire#w8
   RUNG wire#powerrail
      Contact( #"THC_5.2" )
      wire#w11
      { S7_Templates := "SrcType := Real" } EQ_Contact(in1 := #LOGIC_1, in2 := 53.0)
   END_RUNG wire#w8
   RUNG wire#w11
      { S7_Templates := "SrcType := Real" } EQ_Contact(in1 := #LOGIC_2, in2 := 53.0)
   END_RUNG wire#w8
   RUNG wire#w11
      { S7_Templates := "SrcType := Real" } EQ_Contact(in1 := #LOGIC_3, in2 := 53.0)
   END_RUNG wire#w8
   RUNG wire#powerrail
      Contact( #"THC_6.2" )
      wire#w12
      { S7_Templates := "SrcType := Real" } EQ_Contact(in1 := #LOGIC_1, in2 := 63.0)
   END_RUNG wire#w8
   RUNG wire#w12
      { S7_Templates := "SrcType := Real" } EQ_Contact(in1 := #LOGIC_2, in2 := 63.0)
   END_RUNG wire#w8
   RUNG wire#w12
      { S7_Templates := "SrcType := Real" } EQ_Contact(in1 := #LOGIC_3, in2 := 63.0)
   END_RUNG wire#w8
   // the same network as SCL:
   #"OUT_LGOIC_3.1" := (#"THC_2.1" AND ((#LOGIC_1 = 23.0) OR (#LOGIC_2 = 23.0) OR (#LOGIC_3 = 23.0))) OR (#"THC_1.1" AND ((#LOGIC_1 = 13.0) OR (#LOGIC_2 = 13.0) OR (#LOGIC_3 = 13.0))) OR (#"THC_4.1" AND ((#LOGIC_1 = 43.0) OR (#LOGIC_2 = 43.0) OR (#LOGIC_3 = 43.0))) OR (#"THC_5.1" AND ((#LOGIC_1 = 53.0) OR (#LOGIC_2 = 53.0) OR (#LOGIC_3 = 53.0))) OR (#"THC_6.1" AND ((#LOGIC_1 = 63.0) OR (#LOGIC_2 = 63.0) OR (#LOGIC_3 = 63.0)));
   #"OUT_LGOIC_3.2" := (#"THC_2.2" AND ((#LOGIC_1 = 23.0) OR (#LOGIC_2 = 23.0) OR (#LOGIC_3 = 23.0))) OR (#"THC_1.2" AND ((#LOGIC_1 = 13.0) OR (#LOGIC_2 = 13.0) OR (#LOGIC_3 = 13.0))) OR (#"THC_4.2" AND ((#LOGIC_1 = 43.0) OR (#LOGIC_2 = 43.0) OR (#LOGIC_3 = 43.0))) OR (#"THC_5.2" AND ((#LOGIC_1 = 53.0) OR (#LOGIC_2 = 53.0) OR (#LOGIC_3 = 53.0))) OR (#"THC_6.2" AND ((#LOGIC_1 = 63.0) OR (#LOGIC_2 = 63.0) OR (#LOGIC_3 = 63.0)));
END_REGION

REGION Network 4: OUT4
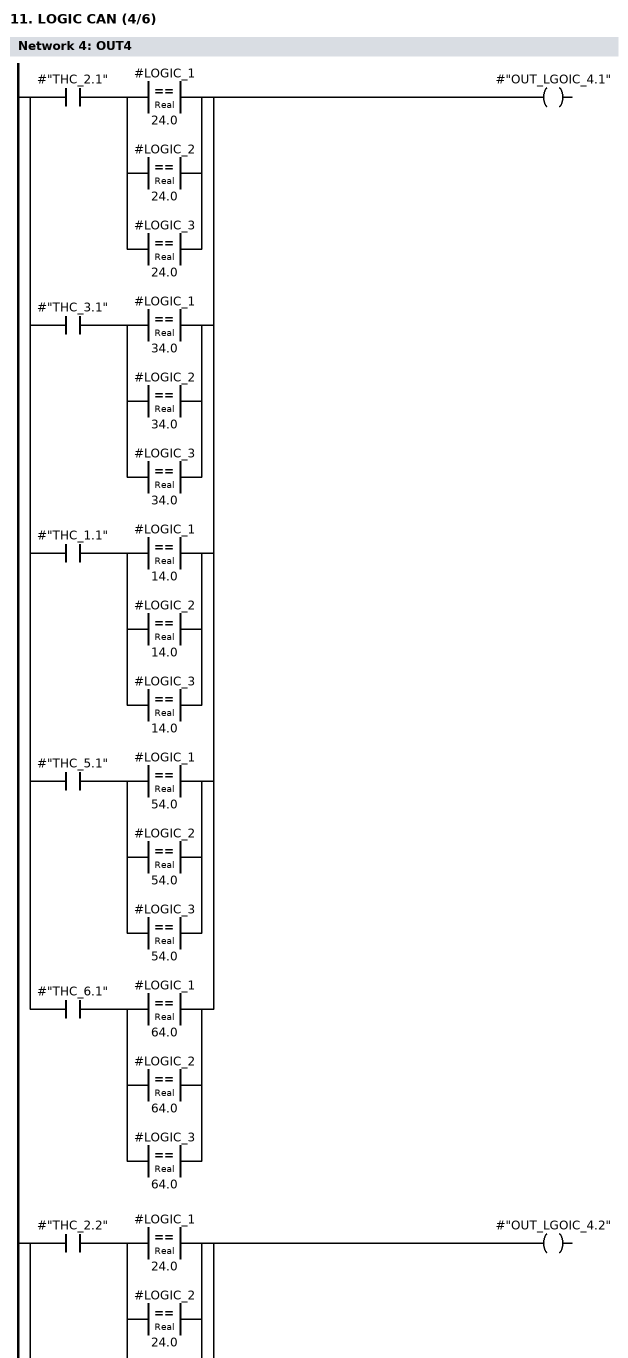
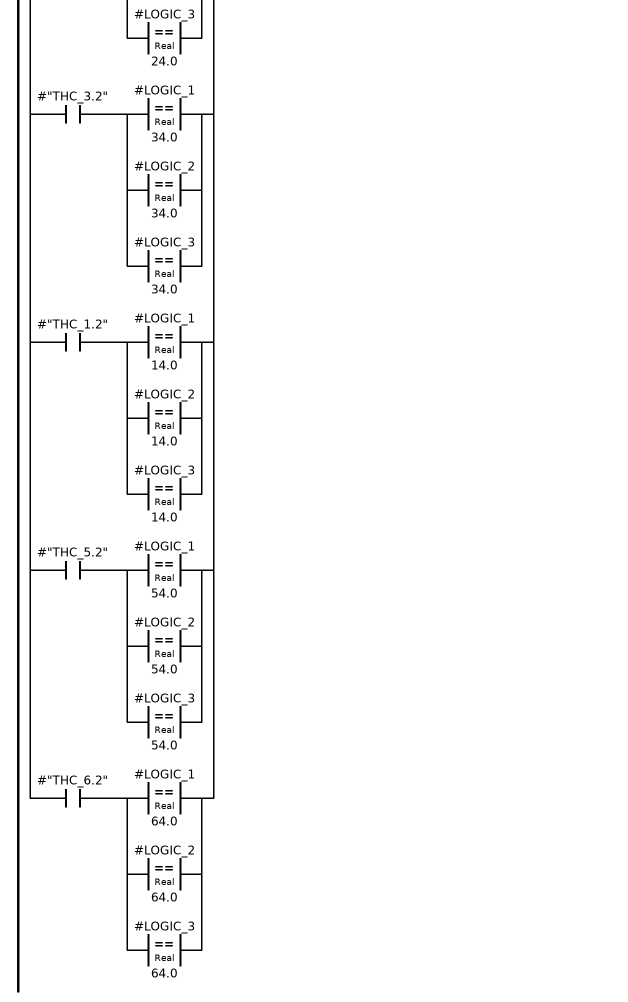
   RUNG wire#powerrail
      Contact( #"THC_2.1" )
      wire#w1
      { S7_Templates := "SrcType := Real" } EQ_Contact(in1 := #LOGIC_1, in2 := 24.0)
      wire#w2
      Coil( #"OUT_LGOIC_4.1" )
   END_RUNG
   RUNG wire#w1
      { S7_Templates := "SrcType := Real" } EQ_Contact(in1 := #LOGIC_2, in2 := 24.0)
   END_RUNG wire#w2
   RUNG wire#w1
      { S7_Templates := "SrcType := Real" } EQ_Contact(in1 := #LOGIC_3, in2 := 24.0)
   END_RUNG wire#w2
   RUNG wire#powerrail
      Contact( #"THC_3.1" )
      wire#w3
      { S7_Templates := "SrcType := Real" } EQ_Contact(in1 := #LOGIC_1, in2 := 34.0)
   END_RUNG wire#w2
   RUNG wire#w3
      { S7_Templates := "SrcType := Real" } EQ_Contact(in1 := #LOGIC_2, in2 := 34.0)
   END_RUNG wire#w2
   RUNG wire#w3
      { S7_Templates := "SrcType := Real" } EQ_Contact(in1 := #LOGIC_3, in2 := 34.0)
   END_RUNG wire#w2
   RUNG wire#powerrail
      Contact( #"THC_1.1" )
      wire#w4
      { S7_Templates := "SrcType := Real" } EQ_Contact(in1 := #LOGIC_1, in2 := 14.0)
   END_RUNG wire#w2
   RUNG wire#w4
      { S7_Templates := "SrcType := Real" } EQ_Contact(in1 := #LOGIC_2, in2 := 14.0)
   END_RUNG wire#w2
   RUNG wire#w4
      { S7_Templates := "SrcType := Real" } EQ_Contact(in1 := #LOGIC_3, in2 := 14.0)
   END_RUNG wire#w2
   RUNG wire#powerrail
      Contact( #"THC_5.1" )
      wire#w5
      { S7_Templates := "SrcType := Real" } EQ_Contact(in1 := #LOGIC_1, in2 := 54.0)
   END_RUNG wire#w2
   RUNG wire#w5
      { S7_Templates := "SrcType := Real" } EQ_Contact(in1 := #LOGIC_2, in2 := 54.0)
   END_RUNG wire#w2
   RUNG wire#w5
      { S7_Templates := "SrcType := Real" } EQ_Contact(in1 := #LOGIC_3, in2 := 54.0)
   END_RUNG wire#w2
   RUNG wire#powerrail
      Contact( #"THC_6.1" )
      wire#w6
      { S7_Templates := "SrcType := Real" } EQ_Contact(in1 := #LOGIC_1, in2 := 64.0)
   END_RUNG wire#w2
   RUNG wire#w6
      { S7_Templates := "SrcType := Real" } EQ_Contact(in1 := #LOGIC_2, in2 := 64.0)
   END_RUNG wire#w2
   RUNG wire#w6
      { S7_Templates := "SrcType := Real" } EQ_Contact(in1 := #LOGIC_3, in2 := 64.0)
   END_RUNG wire#w2
   RUNG wire#powerrail
      Contact( #"THC_2.2" )
      wire#w7
      { S7_Templates := "SrcType := Real" } EQ_Contact(in1 := #LOGIC_1, in2 := 24.0)
      wire#w8
      Coil( #"OUT_LGOIC_4.2" )
   END_RUNG
   RUNG wire#w7
      { S7_Templates := "SrcType := Real" } EQ_Contact(in1 := #LOGIC_2, in2 := 24.0)
   END_RUNG wire#w8
   RUNG wire#w7
      { S7_Templates := "SrcType := Real" } EQ_Contact(in1 := #LOGIC_3, in2 := 24.0)
   END_RUNG wire#w8
   RUNG wire#powerrail
      Contact( #"THC_3.2" )
      wire#w9
      { S7_Templates := "SrcType := Real" } EQ_Contact(in1 := #LOGIC_1, in2 := 34.0)
   END_RUNG wire#w8
   RUNG wire#w9
      { S7_Templates := "SrcType := Real" } EQ_Contact(in1 := #LOGIC_2, in2 := 34.0)
   END_RUNG wire#w8
   RUNG wire#w9
      { S7_Templates := "SrcType := Real" } EQ_Contact(in1 := #LOGIC_3, in2 := 34.0)
   END_RUNG wire#w8
   RUNG wire#powerrail
      Contact( #"THC_1.2" )
      wire#w10
      { S7_Templates := "SrcType := Real" } EQ_Contact(in1 := #LOGIC_1, in2 := 14.0)
   END_RUNG wire#w8
   RUNG wire#w10
      { S7_Templates := "SrcType := Real" } EQ_Contact(in1 := #LOGIC_2, in2 := 14.0)
   END_RUNG wire#w8
   RUNG wire#w10
      { S7_Templates := "SrcType := Real" } EQ_Contact(in1 := #LOGIC_3, in2 := 14.0)
   END_RUNG wire#w8
   RUNG wire#powerrail
      Contact( #"THC_5.2" )
      wire#w11
      { S7_Templates := "SrcType := Real" } EQ_Contact(in1 := #LOGIC_1, in2 := 54.0)
   END_RUNG wire#w8
   RUNG wire#w11
      { S7_Templates := "SrcType := Real" } EQ_Contact(in1 := #LOGIC_2, in2 := 54.0)
   END_RUNG wire#w8
   RUNG wire#w11
      { S7_Templates := "SrcType := Real" } EQ_Contact(in1 := #LOGIC_3, in2 := 54.0)
   END_RUNG wire#w8
   RUNG wire#powerrail
      Contact( #"THC_6.2" )
      wire#w12
      { S7_Templates := "SrcType := Real" } EQ_Contact(in1 := #LOGIC_1, in2 := 64.0)
   END_RUNG wire#w8
   RUNG wire#w12
      { S7_Templates := "SrcType := Real" } EQ_Contact(in1 := #LOGIC_2, in2 := 64.0)
   END_RUNG wire#w8
   RUNG wire#w12
      { S7_Templates := "SrcType := Real" } EQ_Contact(in1 := #LOGIC_3, in2 := 64.0)
   END_RUNG wire#w8
   // the same network as SCL:
   #"OUT_LGOIC_4.1" := (#"THC_2.1" AND ((#LOGIC_1 = 24.0) OR (#LOGIC_2 = 24.0) OR (#LOGIC_3 = 24.0))) OR (#"THC_3.1" AND ((#LOGIC_1 = 34.0) OR (#LOGIC_2 = 34.0) OR (#LOGIC_3 = 34.0))) OR (#"THC_1.1" AND ((#LOGIC_1 = 14.0) OR (#LOGIC_2 = 14.0) OR (#LOGIC_3 = 14.0))) OR (#"THC_5.1" AND ((#LOGIC_1 = 54.0) OR (#LOGIC_2 = 54.0) OR (#LOGIC_3 = 54.0))) OR (#"THC_6.1" AND ((#LOGIC_1 = 64.0) OR (#LOGIC_2 = 64.0) OR (#LOGIC_3 = 64.0)));
   #"OUT_LGOIC_4.2" := (#"THC_2.2" AND ((#LOGIC_1 = 24.0) OR (#LOGIC_2 = 24.0) OR (#LOGIC_3 = 24.0))) OR (#"THC_3.2" AND ((#LOGIC_1 = 34.0) OR (#LOGIC_2 = 34.0) OR (#LOGIC_3 = 34.0))) OR (#"THC_1.2" AND ((#LOGIC_1 = 14.0) OR (#LOGIC_2 = 14.0) OR (#LOGIC_3 = 14.0))) OR (#"THC_5.2" AND ((#LOGIC_1 = 54.0) OR (#LOGIC_2 = 54.0) OR (#LOGIC_3 = 54.0))) OR (#"THC_6.2" AND ((#LOGIC_1 = 64.0) OR (#LOGIC_2 = 64.0) OR (#LOGIC_3 = 64.0)));
END_REGION

REGION Network 5: OUT5
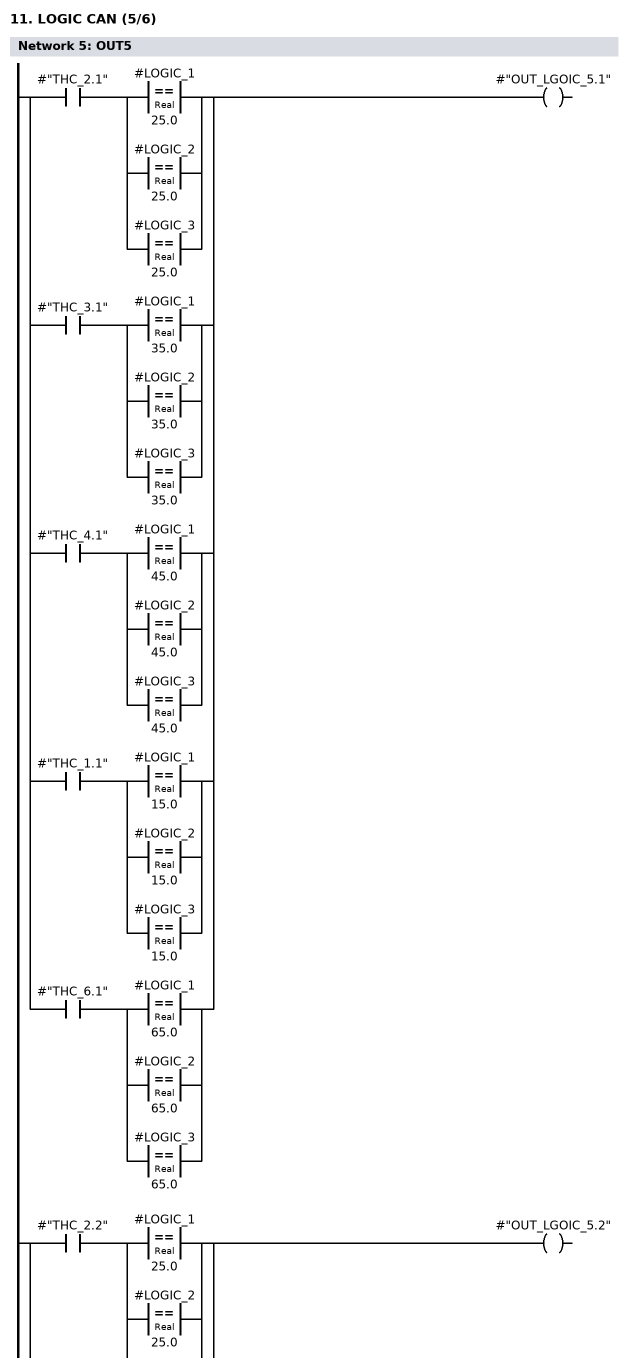
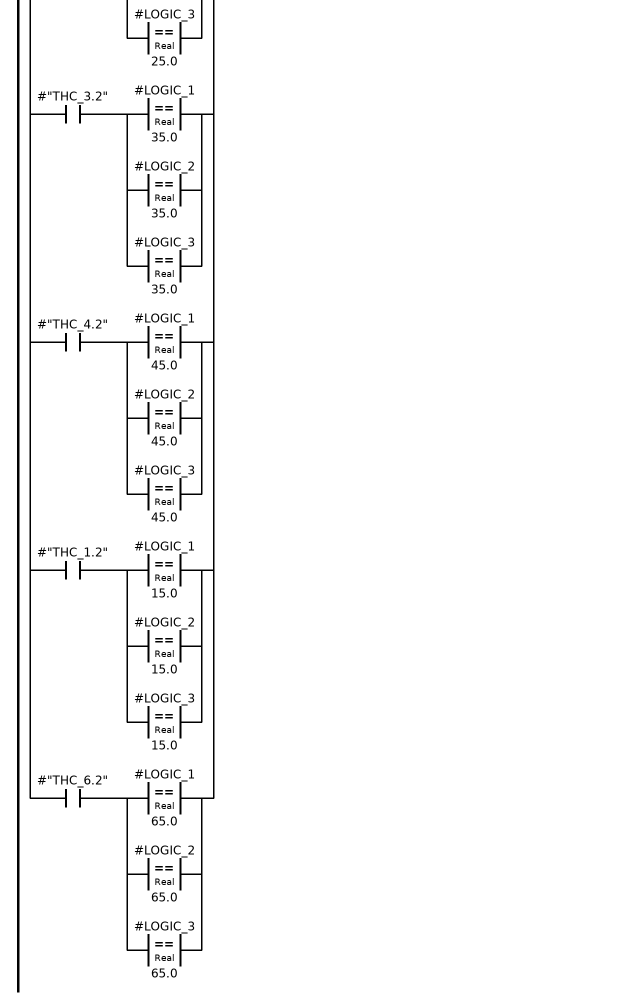
   RUNG wire#powerrail
      Contact( #"THC_2.1" )
      wire#w1
      { S7_Templates := "SrcType := Real" } EQ_Contact(in1 := #LOGIC_1, in2 := 25.0)
      wire#w2
      Coil( #"OUT_LGOIC_5.1" )
   END_RUNG
   RUNG wire#w1
      { S7_Templates := "SrcType := Real" } EQ_Contact(in1 := #LOGIC_2, in2 := 25.0)
   END_RUNG wire#w2
   RUNG wire#w1
      { S7_Templates := "SrcType := Real" } EQ_Contact(in1 := #LOGIC_3, in2 := 25.0)
   END_RUNG wire#w2
   RUNG wire#powerrail
      Contact( #"THC_3.1" )
      wire#w3
      { S7_Templates := "SrcType := Real" } EQ_Contact(in1 := #LOGIC_1, in2 := 35.0)
   END_RUNG wire#w2
   RUNG wire#w3
      { S7_Templates := "SrcType := Real" } EQ_Contact(in1 := #LOGIC_2, in2 := 35.0)
   END_RUNG wire#w2
   RUNG wire#w3
      { S7_Templates := "SrcType := Real" } EQ_Contact(in1 := #LOGIC_3, in2 := 35.0)
   END_RUNG wire#w2
   RUNG wire#powerrail
      Contact( #"THC_4.1" )
      wire#w4
      { S7_Templates := "SrcType := Real" } EQ_Contact(in1 := #LOGIC_1, in2 := 45.0)
   END_RUNG wire#w2
   RUNG wire#w4
      { S7_Templates := "SrcType := Real" } EQ_Contact(in1 := #LOGIC_2, in2 := 45.0)
   END_RUNG wire#w2
   RUNG wire#w4
      { S7_Templates := "SrcType := Real" } EQ_Contact(in1 := #LOGIC_3, in2 := 45.0)
   END_RUNG wire#w2
   RUNG wire#powerrail
      Contact( #"THC_1.1" )
      wire#w5
      { S7_Templates := "SrcType := Real" } EQ_Contact(in1 := #LOGIC_1, in2 := 15.0)
   END_RUNG wire#w2
   RUNG wire#w5
      { S7_Templates := "SrcType := Real" } EQ_Contact(in1 := #LOGIC_2, in2 := 15.0)
   END_RUNG wire#w2
   RUNG wire#w5
      { S7_Templates := "SrcType := Real" } EQ_Contact(in1 := #LOGIC_3, in2 := 15.0)
   END_RUNG wire#w2
   RUNG wire#powerrail
      Contact( #"THC_6.1" )
      wire#w6
      { S7_Templates := "SrcType := Real" } EQ_Contact(in1 := #LOGIC_1, in2 := 65.0)
   END_RUNG wire#w2
   RUNG wire#w6
      { S7_Templates := "SrcType := Real" } EQ_Contact(in1 := #LOGIC_2, in2 := 65.0)
   END_RUNG wire#w2
   RUNG wire#w6
      { S7_Templates := "SrcType := Real" } EQ_Contact(in1 := #LOGIC_3, in2 := 65.0)
   END_RUNG wire#w2
   RUNG wire#powerrail
      Contact( #"THC_2.2" )
      wire#w7
      { S7_Templates := "SrcType := Real" } EQ_Contact(in1 := #LOGIC_1, in2 := 25.0)
      wire#w8
      Coil( #"OUT_LGOIC_5.2" )
   END_RUNG
   RUNG wire#w7
      { S7_Templates := "SrcType := Real" } EQ_Contact(in1 := #LOGIC_2, in2 := 25.0)
   END_RUNG wire#w8
   RUNG wire#w7
      { S7_Templates := "SrcType := Real" } EQ_Contact(in1 := #LOGIC_3, in2 := 25.0)
   END_RUNG wire#w8
   RUNG wire#powerrail
      Contact( #"THC_3.2" )
      wire#w9
      { S7_Templates := "SrcType := Real" } EQ_Contact(in1 := #LOGIC_1, in2 := 35.0)
   END_RUNG wire#w8
   RUNG wire#w9
      { S7_Templates := "SrcType := Real" } EQ_Contact(in1 := #LOGIC_2, in2 := 35.0)
   END_RUNG wire#w8
   RUNG wire#w9
      { S7_Templates := "SrcType := Real" } EQ_Contact(in1 := #LOGIC_3, in2 := 35.0)
   END_RUNG wire#w8
   RUNG wire#powerrail
      Contact( #"THC_4.2" )
      wire#w10
      { S7_Templates := "SrcType := Real" } EQ_Contact(in1 := #LOGIC_1, in2 := 45.0)
   END_RUNG wire#w8
   RUNG wire#w10
      { S7_Templates := "SrcType := Real" } EQ_Contact(in1 := #LOGIC_2, in2 := 45.0)
   END_RUNG wire#w8
   RUNG wire#w10
      { S7_Templates := "SrcType := Real" } EQ_Contact(in1 := #LOGIC_3, in2 := 45.0)
   END_RUNG wire#w8
   RUNG wire#powerrail
      Contact( #"THC_1.2" )
      wire#w11
      { S7_Templates := "SrcType := Real" } EQ_Contact(in1 := #LOGIC_1, in2 := 15.0)
   END_RUNG wire#w8
   RUNG wire#w11
      { S7_Templates := "SrcType := Real" } EQ_Contact(in1 := #LOGIC_2, in2 := 15.0)
   END_RUNG wire#w8
   RUNG wire#w11
      { S7_Templates := "SrcType := Real" } EQ_Contact(in1 := #LOGIC_3, in2 := 15.0)
   END_RUNG wire#w8
   RUNG wire#powerrail
      Contact( #"THC_6.2" )
      wire#w12
      { S7_Templates := "SrcType := Real" } EQ_Contact(in1 := #LOGIC_1, in2 := 65.0)
   END_RUNG wire#w8
   RUNG wire#w12
      { S7_Templates := "SrcType := Real" } EQ_Contact(in1 := #LOGIC_2, in2 := 65.0)
   END_RUNG wire#w8
   RUNG wire#w12
      { S7_Templates := "SrcType := Real" } EQ_Contact(in1 := #LOGIC_3, in2 := 65.0)
   END_RUNG wire#w8
   // the same network as SCL:
   #"OUT_LGOIC_5.1" := (#"THC_2.1" AND ((#LOGIC_1 = 25.0) OR (#LOGIC_2 = 25.0) OR (#LOGIC_3 = 25.0))) OR (#"THC_3.1" AND ((#LOGIC_1 = 35.0) OR (#LOGIC_2 = 35.0) OR (#LOGIC_3 = 35.0))) OR (#"THC_4.1" AND ((#LOGIC_1 = 45.0) OR (#LOGIC_2 = 45.0) OR (#LOGIC_3 = 45.0))) OR (#"THC_1.1" AND ((#LOGIC_1 = 15.0) OR (#LOGIC_2 = 15.0) OR (#LOGIC_3 = 15.0))) OR (#"THC_6.1" AND ((#LOGIC_1 = 65.0) OR (#LOGIC_2 = 65.0) OR (#LOGIC_3 = 65.0)));
   #"OUT_LGOIC_5.2" := (#"THC_2.2" AND ((#LOGIC_1 = 25.0) OR (#LOGIC_2 = 25.0) OR (#LOGIC_3 = 25.0))) OR (#"THC_3.2" AND ((#LOGIC_1 = 35.0) OR (#LOGIC_2 = 35.0) OR (#LOGIC_3 = 35.0))) OR (#"THC_4.2" AND ((#LOGIC_1 = 45.0) OR (#LOGIC_2 = 45.0) OR (#LOGIC_3 = 45.0))) OR (#"THC_1.2" AND ((#LOGIC_1 = 15.0) OR (#LOGIC_2 = 15.0) OR (#LOGIC_3 = 15.0))) OR (#"THC_6.2" AND ((#LOGIC_1 = 65.0) OR (#LOGIC_2 = 65.0) OR (#LOGIC_3 = 65.0)));
END_REGION

REGION Network 6: OUT6
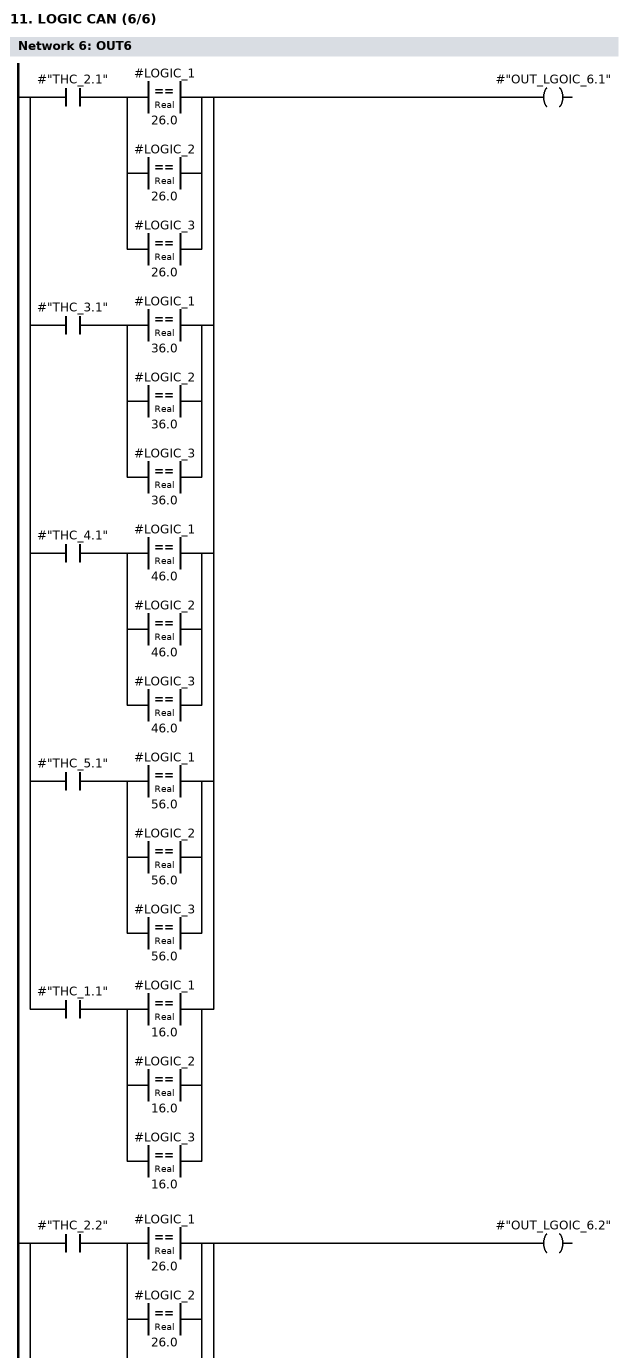
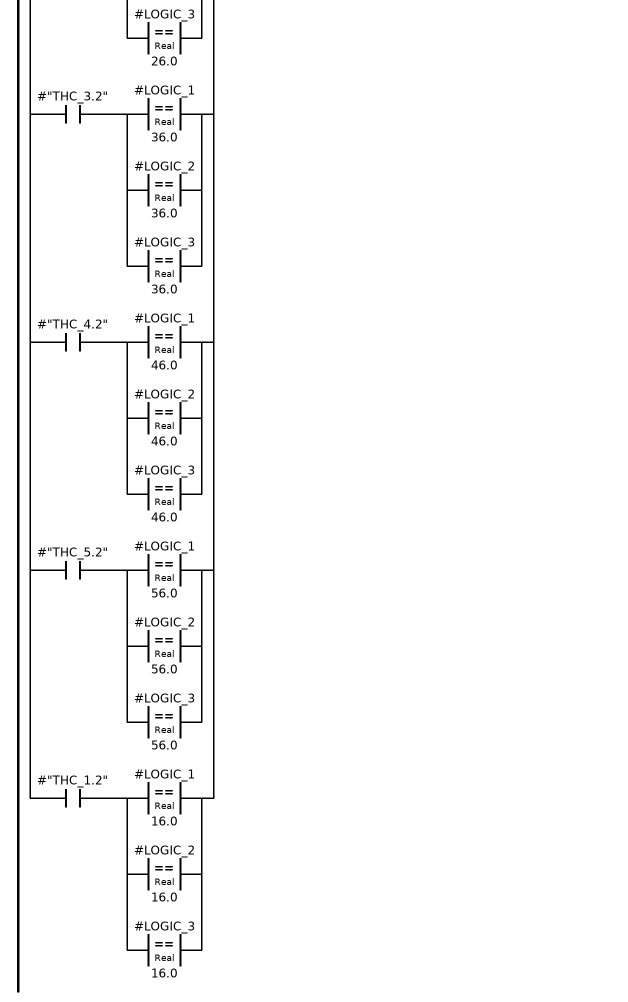
   RUNG wire#powerrail
      Contact( #"THC_2.1" )
      wire#w1
      { S7_Templates := "SrcType := Real" } EQ_Contact(in1 := #LOGIC_1, in2 := 26.0)
      wire#w2
      Coil( #"OUT_LGOIC_6.1" )
   END_RUNG
   RUNG wire#w1
      { S7_Templates := "SrcType := Real" } EQ_Contact(in1 := #LOGIC_2, in2 := 26.0)
   END_RUNG wire#w2
   RUNG wire#w1
      { S7_Templates := "SrcType := Real" } EQ_Contact(in1 := #LOGIC_3, in2 := 26.0)
   END_RUNG wire#w2
   RUNG wire#powerrail
      Contact( #"THC_3.1" )
      wire#w3
      { S7_Templates := "SrcType := Real" } EQ_Contact(in1 := #LOGIC_1, in2 := 36.0)
   END_RUNG wire#w2
   RUNG wire#w3
      { S7_Templates := "SrcType := Real" } EQ_Contact(in1 := #LOGIC_2, in2 := 36.0)
   END_RUNG wire#w2
   RUNG wire#w3
      { S7_Templates := "SrcType := Real" } EQ_Contact(in1 := #LOGIC_3, in2 := 36.0)
   END_RUNG wire#w2
   RUNG wire#powerrail
      Contact( #"THC_4.1" )
      wire#w4
      { S7_Templates := "SrcType := Real" } EQ_Contact(in1 := #LOGIC_1, in2 := 46.0)
   END_RUNG wire#w2
   RUNG wire#w4
      { S7_Templates := "SrcType := Real" } EQ_Contact(in1 := #LOGIC_2, in2 := 46.0)
   END_RUNG wire#w2
   RUNG wire#w4
      { S7_Templates := "SrcType := Real" } EQ_Contact(in1 := #LOGIC_3, in2 := 46.0)
   END_RUNG wire#w2
   RUNG wire#powerrail
      Contact( #"THC_5.1" )
      wire#w5
      { S7_Templates := "SrcType := Real" } EQ_Contact(in1 := #LOGIC_1, in2 := 56.0)
   END_RUNG wire#w2
   RUNG wire#w5
      { S7_Templates := "SrcType := Real" } EQ_Contact(in1 := #LOGIC_2, in2 := 56.0)
   END_RUNG wire#w2
   RUNG wire#w5
      { S7_Templates := "SrcType := Real" } EQ_Contact(in1 := #LOGIC_3, in2 := 56.0)
   END_RUNG wire#w2
   RUNG wire#powerrail
      Contact( #"THC_1.1" )
      wire#w6
      { S7_Templates := "SrcType := Real" } EQ_Contact(in1 := #LOGIC_1, in2 := 16.0)
   END_RUNG wire#w2
   RUNG wire#w6
      { S7_Templates := "SrcType := Real" } EQ_Contact(in1 := #LOGIC_2, in2 := 16.0)
   END_RUNG wire#w2
   RUNG wire#w6
      { S7_Templates := "SrcType := Real" } EQ_Contact(in1 := #LOGIC_3, in2 := 16.0)
   END_RUNG wire#w2
   RUNG wire#powerrail
      Contact( #"THC_2.2" )
      wire#w7
      { S7_Templates := "SrcType := Real" } EQ_Contact(in1 := #LOGIC_1, in2 := 26.0)
      wire#w8
      Coil( #"OUT_LGOIC_6.2" )
   END_RUNG
   RUNG wire#w7
      { S7_Templates := "SrcType := Real" } EQ_Contact(in1 := #LOGIC_2, in2 := 26.0)
   END_RUNG wire#w8
   RUNG wire#w7
      { S7_Templates := "SrcType := Real" } EQ_Contact(in1 := #LOGIC_3, in2 := 26.0)
   END_RUNG wire#w8
   RUNG wire#powerrail
      Contact( #"THC_3.2" )
      wire#w9
      { S7_Templates := "SrcType := Real" } EQ_Contact(in1 := #LOGIC_1, in2 := 36.0)
   END_RUNG wire#w8
   RUNG wire#w9
      { S7_Templates := "SrcType := Real" } EQ_Contact(in1 := #LOGIC_2, in2 := 36.0)
   END_RUNG wire#w8
   RUNG wire#w9
      { S7_Templates := "SrcType := Real" } EQ_Contact(in1 := #LOGIC_3, in2 := 36.0)
   END_RUNG wire#w8
   RUNG wire#powerrail
      Contact( #"THC_4.2" )
      wire#w10
      { S7_Templates := "SrcType := Real" } EQ_Contact(in1 := #LOGIC_1, in2 := 46.0)
   END_RUNG wire#w8
   RUNG wire#w10
      { S7_Templates := "SrcType := Real" } EQ_Contact(in1 := #LOGIC_2, in2 := 46.0)
   END_RUNG wire#w8
   RUNG wire#w10
      { S7_Templates := "SrcType := Real" } EQ_Contact(in1 := #LOGIC_3, in2 := 46.0)
   END_RUNG wire#w8
   RUNG wire#powerrail
      Contact( #"THC_5.2" )
      wire#w11
      { S7_Templates := "SrcType := Real" } EQ_Contact(in1 := #LOGIC_1, in2 := 56.0)
   END_RUNG wire#w8
   RUNG wire#w11
      { S7_Templates := "SrcType := Real" } EQ_Contact(in1 := #LOGIC_2, in2 := 56.0)
   END_RUNG wire#w8
   RUNG wire#w11
      { S7_Templates := "SrcType := Real" } EQ_Contact(in1 := #LOGIC_3, in2 := 56.0)
   END_RUNG wire#w8
   RUNG wire#powerrail
      Contact( #"THC_1.2" )
      wire#w12
      { S7_Templates := "SrcType := Real" } EQ_Contact(in1 := #LOGIC_1, in2 := 16.0)
   END_RUNG wire#w8
   RUNG wire#w12
      { S7_Templates := "SrcType := Real" } EQ_Contact(in1 := #LOGIC_2, in2 := 16.0)
   END_RUNG wire#w8
   RUNG wire#w12
      { S7_Templates := "SrcType := Real" } EQ_Contact(in1 := #LOGIC_3, in2 := 16.0)
   END_RUNG wire#w8
   // the same network as SCL:
   #"OUT_LGOIC_6.1" := (#"THC_2.1" AND ((#LOGIC_1 = 26.0) OR (#LOGIC_2 = 26.0) OR (#LOGIC_3 = 26.0))) OR (#"THC_3.1" AND ((#LOGIC_1 = 36.0) OR (#LOGIC_2 = 36.0) OR (#LOGIC_3 = 36.0))) OR (#"THC_4.1" AND ((#LOGIC_1 = 46.0) OR (#LOGIC_2 = 46.0) OR (#LOGIC_3 = 46.0))) OR (#"THC_5.1" AND ((#LOGIC_1 = 56.0) OR (#LOGIC_2 = 56.0) OR (#LOGIC_3 = 56.0))) OR (#"THC_1.1" AND ((#LOGIC_1 = 16.0) OR (#LOGIC_2 = 16.0) OR (#LOGIC_3 = 16.0)));
   #"OUT_LGOIC_6.2" := (#"THC_2.2" AND ((#LOGIC_1 = 26.0) OR (#LOGIC_2 = 26.0) OR (#LOGIC_3 = 26.0))) OR (#"THC_3.2" AND ((#LOGIC_1 = 36.0) OR (#LOGIC_2 = 36.0) OR (#LOGIC_3 = 36.0))) OR (#"THC_4.2" AND ((#LOGIC_1 = 46.0) OR (#LOGIC_2 = 46.0) OR (#LOGIC_3 = 46.0))) OR (#"THC_5.2" AND ((#LOGIC_1 = 56.0) OR (#LOGIC_2 = 56.0) OR (#LOGIC_3 = 56.0))) OR (#"THC_1.2" AND ((#LOGIC_1 = 16.0) OR (#LOGIC_2 = 16.0) OR (#LOGIC_3 = 16.0)));
END_REGION
END_FUNCTION_BLOCK

FUNCTION "3.OUTPUT_PLC" : Void   // FC3, LAD
{ S7_Optimized_Access := 'TRUE' }
VERSION : 0.1
// stored: AutoNumber false, CodeModifiedDate 2025-08-27T17:07:28.4518091Z, CompileDate 2026-01-15T16:25:55.7493553Z, CreationDate 2026-01-15T16:22:49.8270549Z, HandleErrorsWithinBlock false, InterfaceModifiedDate 2022-06-07T03:40:45.7898546Z, IsConsistent true, IsIECCheckEnabled false, IsKnowHowProtected false, IsWriteProtected false, LibraryConformanceStatus The object is library-conformant., ModifiedDate 2025-08-27T17:07:28.4518091Z, ParameterModified 2022-06-07T03:40:45.7898546Z, PLCSimAdvancedSupport false, SetENOAutomatically False, StructureModified 2022-06-07T03:40:45.7898546Z, UDAEnableTagReadback false
   VAR_INPUT
      A1 : Bool;
      M1 : Bool;
      A2 : Bool;
      M2 : Bool;
      A3 : Bool;
      M3 : Bool;
      A4 : Bool;
      M4 : Bool;
   END_VAR
   VAR_OUTPUT
      OUT1 : Bool;
      OUT2 : Bool;
      OUT3 : Bool;
      OUT4 : Bool;
   END_VAR
BEGIN

REGION Network 1
